(* Schneider Machine Expert - Basic project PLC_New_08_09, file version 2.7.0.0 *)
(* CompanyInformations: Name=Plast-O-Matick, Country=EEUU *)
(* ProjectInformations: Name=New project *)

HARDWARE
  Cpu 0: TM221CE16R
  ModuleExtensionObject 0: TM3AM6/G
  EthernetConfiguration: NetworkName=M221, IpAllocationMode=FixedAddress, IpAddress=192.168.1.235, SubnetMask=255.255.255.0
  SerialLineConfiguration: Baud=Baud19200, Parity=ParityNone, DataBits=DataBits8, StopBits=StopBits1, PhysicalMedium=PhysicalMediumRs485, TransmissionMode=TransmissionModeModbusRtu, SlaveId=1, Addressing=MasterAddressing
  MastTask: UsePeriodScanMode=false, PeriodScan=100
  FastTask: Period=255
  CpuBehavior: StartingMode=StartAsPreviousState, AutoSaveRamOnEeprom=true, WatchdogPeriod=250

SYMBOLS  (address, symbol, comment, settings)
  %MW432:X0 VLV03_04_POWER_ON
  %MW444:X0 VLV05_06_POWER_ON
  %MW117:X0 DATETIME_CHANGE
  %M0       VLV01_HMI_START
  %M1       VLV01_HMI_STP
  %M2       VLV01_CMD_OPN
  %M3       VLV01_TON_OPN_DN
  %M4       VLV01_COUNT_OPN_DN
  %M5       VLV01_RST_COUNT
  %M6       VLV01_ONS_STS_AUTOMATIC
  %M7       VLV01_CNF_OPN
  %M8       VLV01_CNF_CLS
  %M9       COPY_DATA
  %M10      VLV01_ONS_STP
  %M11      VLV01_SAVE_DATETIME
  %M12      VLV01_CMD_CLS
  %M13      VLV01_TON_CLS_DN
  %M14      VLV01_COUNT_CLS_DN
  %M15      VLV01_ALMD_CNF_OPN_DN
  %M16      VLV01_ALMD_CNF_CLS_DN
  %M17      VLV01_T_ALMD_CNF_OPN_DN
  %M19      VLV01_T_ALMD_CNF_CLS_DN
  %M20      PLC_HORARIOOFICINA
  %M21      HORARIOOFICINA_ACTIVE
  %M22      HMI_HORARIOOFICINA
  %M23      VLV01_STS_AUTOMATIC
  %M24      VLV01_HMI_STARTED
  %M25      VLV01_TON_SEG_RST
  %M26      VLV01_TON_SEG_DN
  %M27      VLV01_TON_MIN_DN
  %M28      VLV01_TON_HR_DN
  %M29      VLV2_ONS_STP
  %M30      VLV02_HMI_START
  %M31      VLV02_HMI_STP
  %M32      VLV02_CMD_OPN
  %M33      VLV02_TON_OPN_DN
  %M34      VLV02_COUNT_OPN_DN
  %M35      VLV02_RST_COUNT
  %M36      VLV02_ONS_STS_AUTOMATIC
  %M37      VLV02_CNF_OPN
  %M38      VLV02_CNF_CLS
  %M41      VLV02_SAVE_DATETIME
  %M42      VLV02_CMD_CLS
  %M43      VLV02_TON_CLS_DN
  %M44      VLV02_COUNT_CLS_DN
  %M45      VLV02_ALMD_CNF_OPN_DN
  %M46      VLV02_ALMD_CNF_CLS_DN
  %M47      VLV02_T_ALMD_CNF_OPN_DN
  %M49      VLV02_T_ALMD_CNF_CLS_DN
  %M50      VLV01_02_POWER_ON
  %M53      VLV02_STS_AUTOMATIC
  %M54      VLV02_HMI_STARTED
  %M55      VLV02_TON_SEG_RST
  %M56      VLV02_TON_SEG_DN
  %M57      VLV02_TON_MIN_DN
  %M58      VLV02_TON_HR_DN
  %M60      VLV03_HMI_START
  %M61      VLV03_HMI_STP
  %M62      VLV03_CMD_OPN
  %M63      VLV03_TON_OPN_DN
  %M64      VLV03_COUNT_OPN_DN
  %M65      VLV03_RST_COUNT
  %M66      VLV03_ONS_STR_AUTOMATIC
  %M67      VLV03_CNF_OPN
  %M68      VLV03_CNF_CLS
  %M70      VLV03_CLOSE_DATA1
  %M71      VLV03_SAVE_DATETIME
  %M72      VLV03_CMD_CLS
  %M73      VLV03_TON_CLS_DN
  %M74      VLV03_COUNT_CLS_DN
  %M75      VLV03_ALMD_CNF_OPN_DN
  %M76      VLV03_ALMD_CNF_CLS_DN
  %M77      VLV03_T_ALMD_CNF_OPN_DN
  %M78      VLV03_ONS_STP_AUTOMATIC
  %M79      VLV03_T_ALMD_CNF_CLS_DN
  %M83      VLV03_STS_AUTOMATIC
  %M84      VLV03_HMI_STARTED
  %M85      VLV03_TON_SEG_RST
  %M86      VLV03_TON_SEG_DN
  %M87      VLV03_TON_MIN_DN
  %M88      VLV03_TON_HR_DN
  %M90      VLV04_HMI_START
  %M91      VLV04_HMI_STP
  %M92      VLV04_CMD_OPN
  %M93      VLV04_TON_OPN_DN
  %M94      VLV04_COUNT_OPN_DN
  %M95      VLV04_RST_COUNT
  %M96      VLV04_ONS_STR_AUTOMATIC
  %M97      VLV04_CNF_OPN
  %M98      VLV04_CNF_CLS
  %M100     VLV04_CLOSE_DATA1
  %M101     VLV04_SAVE_DATETIME
  %M102     VLV04_CMD_CLS
  %M103     VLV04_TON_CLS_DN
  %M104     VLV04_COUNT_CLS_DN
  %M105     VLV04_ALMD_CNF_OPN_DN
  %M106     VLV04_ALMD_CNF_CLS_DN
  %M107     VLV04_T_ALMD_CNF_OPN_DN
  %M108     VLV04_ONS_STP_AUTOMATIC
  %M109     VLV04_T_ALMD_CNF_CLS_DN
  %M113     VLV04_STS_AUTOMATIC
  %M114     VLV04_HMI_STARTED
  %M115     VLV04_TON_SEG_RST
  %M116     VLV04_TON_SEG_DN
  %M117     VLV04_TON_MIN_DN
  %M118     VLV04_TON_HR_DN
  %M120     VLV05_HMI_START
  %M121     VLV05_HMI_STP
  %M122     VLV05_CMD_OPN
  %M123     VLV05_TON_OPN_DN
  %M124     VLV05_COUNT_OPN_DN
  %M125     VLV05_RST_COUNT
  %M126     VLV05_ONS_STS_AUTOMATIC
  %M127     VLV05_CNF_OPN
  %M128     VLV05_CNF_CLS
  %M131     VLV05_SAVE_DATETIME
  %M132     VLV05_CMD_CLS
  %M133     VLV05_TON_CLS_DN
  %M134     VLV05_COUNT_CLS_DN
  %M135     VLV05_ALMD_CNF_OPN_DN
  %M136     VLV05_ALMD_CNF_CLS_DN
  %M137     VLV05_T_ALMD_CNF_OPN_DN
  %M138     VLV05_ONS_STP_AUTOMATIC
  %M139     VLV05_T_ALMD_CNF_CLS_DN
  %M143     VLV05_STS_AUTOMATIC
  %M144     VLV05_HMI_STARTED
  %M145     VLV05_TON_SEG_RST
  %M146     VLV05_TON_SEG_DN
  %M147     VLV05_TON_MIN_DN
  %M148     VLV05_TON_HR_DN
  %M150     VLV06_HMI_START
  %M151     VLV06_HMI_STP
  %M152     VLV06_CMD_OPN
  %M153     VLV06_TON_OPN_DN
  %M154     VLV06_COUNT_OPN_DN
  %M155     VLV06_RST_COUNT
  %M156     VLV06_ONS_STS_AUTOMATIC
  %M157     VLV06_CNF_OPN
  %M158     VLV06_CNF_CLS
  %M161     VLV06_SAVE_DATETIME
  %M162     VLV06_CMD_CLS
  %M163     VLV06_TON_CLS_DN
  %M164     VLV06_COUNT_CLS_DN
  %M165     VLV06_ALMD_CNF_OPN_DN
  %M166     VLV06_ALMD_CNF_CLS_DN
  %M167     VLV06_T_ALMD_CNF_OPN_DN
  %M169     VLV06_T_ALMD_CNF_CLS_DN
  %M173     VLV06_STS_AUTOMATIC
  %M174     VLV06_HMI_STARTED
  %M175     VLV06_TON_SEG_RST
  %M176     VLV06_TON_SEG_DN
  %M177     VLV06_TON_MIN_DN
  %M178     VLV06_TON_HR_DN
  %M180     VLV07_HMI_START
  %M181     VLV07_HMI_STP
  %M182     VLV07_CMD_OPN
  %M183     VLV07_TON_OPN_DN
  %M184     VLV07_COUNT_OPN_DN
  %M185     VLV07_RST_COUNT
  %M186     VLV07_ONS_STS_AUTOMATIC
  %M187     VLV07_CNF_OPN
  %M188     VLV07_CNF_CLS
  %M191     VLV07_SAVE_DATETIME
  %M192     VLV07_CMD_CLS
  %M193     VLV07_TON_CLS_DN
  %M194     VLV07_COUNT_CLS_DN
  %M195     VLV07_ALMD_CNF_OPN_DN
  %M196     VLV07_ALMD_CNF_CLS_DN
  %M197     VLV07_T_ALMD_CNF_OPN_DN
  %M199     VLV07_T_ALMD_CNF_CLS_DN
  %M200     VLV07_SCHEDULE_ON
  %M203     VLV07_STS_AUTOMATIC
  %M204     VLV07_HMI_STARTED
  %M205     VLV07_TON_SEG_RST
  %M206     VLV07_TON_SEG_DN
  %M207     VLV07_TON_MIN_DN
  %M208     VLV07_TON_HR_DN
  %M220     VLV08_HMI_START
  %M221     VLV08_HMI_STP
  %M222     VLV08_HMI_STARTED
  %M223     VLV08_RST_COUNT
  %M224     VLV08_STS_AUTOMATIC
  %M225     VLV08_ONS_STR
  %M226     VLV08_ONS_STP_AUTOMATIC
  %M227     VLV08_ONS_STS_AUTOMATIC
  %M228     VLV08_ONS_01
  %M229     VLV08_CMD_OPN
  %M230     VLV08_CMD_CLS
  %M231     VLV08_CNF_OPN
  %M232     VLV08_CNF_CLS
  %M233     VLV08_TON_OPN_DN
  %M234     VLV08_TON_CLS_DN
  %M235     VLV08_TON_SEG_DN
  %M236     VLV08_TON_SEG_RST
  %M237     VLV08_TON_MIN_DN
  %M238     VLV08_TON_HR_DN
  %M239     VLV08_ALMD_CNF_OPN_DN
  %M240     VLV08_ALMD_CNF_CLS_DN
  %M241     VLV08_T_ALMD_CNF_OPN_DN
  %M242     VLV08_T_ALMD_CNF_CLS_DN
  %M243     VLV08_SAVE_DATETIME
  %M244     VLV08_T_CNF_OPN
  %M245     VLV08_T_CNF_CLS
  %M246     VLV08_MB_COMM_OK
  %M247     VLV08_MB_COMM_ERROR
  %M248     VLV08_MB_READ_ENABLE
  %M249     VLV08_MB_READ_TRIGGER
  %M250     VLV08_ONS_STR_AUTOMATIC
  %M251     VLV08_CLOSE_DATA1
  %M315     VLV09_HMI_START
  %M316     VLV09_HMI_STP
  %M317     VLV09_HMI_STARTED
  %M318     VLV09_RST_COUNT
  %M319     VLV09_STS_AUTOMATIC
  %M320     VLV09_ONS_STR
  %M321     VLV09_ONS_STP_AUTOMATIC
  %M322     VLV09_ONS_STS_AUTOMATIC
  %M323     VLV09_ONS_01
  %M324     VLV09_CMD_OPN
  %M325     VLV09_CMD_CLS
  %M326     VLV09_CNF_OPN
  %M327     VLV09_CNF_CLS
  %M328     VLV09_TON_OPN_DN
  %M329     VLV09_TON_CLS_DN
  %M330     VLV09_TON_SEG_DN
  %M331     VLV09_TON_SEG_RST
  %M332     VLV09_TON_MIN_DN
  %M333     VLV09_TON_HR_DN
  %M334     VLV09_ALMD_CNF_OPN_DN
  %M335     VLV09_ALMD_CNF_CLS_DN
  %M336     VLV09_T_ALMD_CNF_OPN_DN
  %M337     VLV09_T_ALMD_CNF_CLS_DN
  %M338     VLV09_SAVE_DATETIME
  %M339     VLV09_T_CNF_OPN
  %M340     VLV09_T_CNF_CLS
  %M341     VLV09_MB_COMM_OK
  %M342     VLV09_MB_COMM_ERROR
  %M343     VLV09_MB_READ_ENABLE
  %M344     VLV09_MB_READ_TRIGGER
  %S5       SB_TB100MS  "Time base of 100 ms generated by an internal clock"
  %S13      SB_FIRSTRUN  "Indicates the first controller cycle in RUN mode"
  %S50      SB_RTCUPDATE  "Set to 1, this bit allows to update the date and time"
  %SW51     SW_RTCHHMM  "RTC Function: contains in BCD HHMM: hour and minute"
  %SW52     SW_RTCMMDD  "RTC Function: contains in BCD MMDD: month and day"
  %SW53     SW_RTCCCYY  "RTC Function: contains in BCD CCYY: century and year"
  %MW0      VLV01_CNT_CLS_ACC
  %MW1      VLV01_CNT_OPN_ACC
  %MW2      VLV01_T_CNF_PRESET
  %MW3      VLV01_CNF_HR_PRESET
  %MW5      VLV01_RTC_HHMM
  %MW6      VLV01_RTC_MMDD
  %MW7      VLV01_RTC_YY
  %MW10     VLV02_CNT_CLS_ACC
  %MW11     VLV02_CNT_OPN_ACC
  %MW12     VLV02_T_CNF_PRESET  "timer1"
  %MW13     VLV02_CNF_HR_PRESET
  %MW15     VLV02_RTC_HHMM
  %MW16     VLV02_RTC_MMDD
  %MW17     VLV02_RTC_YY
  %MW18     VLV03_SP_ACTUAL
  %MW19     VLV03_CV_ACTUAL
  %MW20     VLV03_CNT_CLS_ACC
  %MW21     VLV03_CNT_OPN_ACC
  %MW22     VLV03_T_CNF_PRESET
  %MW23     VLV03_CNF_HR_PRESET
  %MW24     VLV03_SETPOINT_ALTO
  %MW25     VLV03_RTC_HHMM
  %MW26     VLV03_RTC_MMDD
  %MW27     VLV03_RTC_YY
  %MW28     VLV04_SP_ACTUAL
  %MW29     VLV04_CV_ACTUAL
  %MW30     VLV04_CNT_CLS_ACC
  %MW31     VLV04_CNT_OPN_ACC
  %MW32     VLV04_T_CNF_PRESET
  %MW33     VLV04_CNF_HR_PRESET
  %MW34     VLV04_SETPOINT_ALTO
  %MW35     VLV04_RTC_HHMM
  %MW36     VLV04_RTC_MMDD
  %MW37     VLV04_RTC_YY
  %MW40     VLV05_CNT_CLS_ACC
  %MW41     VLV05_CNT_OPN_ACC
  %MW42     VLV05_T_CNF_PRESET
  %MW43     VLV05_CNF_HR_PRESET
  %MW45     VLV05_RTC_HHMM
  %MW46     VLV05_RTC_MMDD
  %MW47     VLV05_RTC_YY
  %MW50     VLV06_CNT_CLS_ACC
  %MW51     VLV06_CNT_OPN_ACC
  %MW52     VLV06_T_CNF_PRESET
  %MW53     VLV06_CNF_HR_PRESET
  %MW55     VLV06_RTC_HHMM
  %MW56     VLV06_RTC_MMDD
  %MW57     VLV06_RTC_YY
  %MW60     VLV07_CNT_OPN_ACC
  %MW61     VLV07_CNT_CLS_ACC
  %MW63     VLV07_T_CICLO
  %MW64     VLV07_WORK_CICLE
  %MW68     VLV05_RTC_HHMM_OPEN
  %MW69     VLV05_RTC_MMDD_OPEN
  %MW70     VLV05_RTC_YY_OPEN
  %MW71     VLV05_RTC_HHMM_CLOSE
  %MW72     VLV05_RTC_MMDD_CLOSE
  %MW73     VLV05_RTC_YY_CLOSE
  %MW110    DAY
  %MW111    HOUR
  %MW112    MINUTES
  %MW113    MONTH
  %MW114    YEAR
  %MW115    SCRAP_MONTH
  %MW116    SCRAP_MINUTES
  %MW129    VLV07_SCHEDULE
  %MW130    VLV07_MONTH
  %MW131    VLV07_YR
  %MW132    VLV07_DY
  %MW133    VLV07_HR
  %MW134    VLV07_MIN
  %MW135    VLV07_OPEN_MONTH
  %MW136    VLV07_OPEN_YR
  %MW137    VLV07_OPEN_DY
  %MW138    VLV07_OPEN_HR
  %MW139    VLV07_OPEN_MIN
  %MW140    VLV07_CLOSE_MONTH
  %MW141    VLV07_CLOSE_YR
  %MW142    VLV07_CLOSE_DY
  %MW143    VLV07_CLOSE_HR
  %MW144    VLV07_CLOSE_MIN
  %MW145    VLV07_SCHED_HR
  %MW146    VLV07_SCHED_MIN
  %MW155    VLV01_CNF_OPN_W
  %MW156    VLV02_CNF_OPN_W
  %MW180    VLV08_SP_ACTUAL  "Setpoint actual VLV8"
  %MW181    VLV08_CV_ACTUAL  "Control value (salida analógica)"
  %MW182    VLV08_CNT_CLS_ACC  "Acumulador contador cierre"
  %MW183    VLV08_CNT_OPN_ACC  "Acumulador contador apertura"
  %MW184    VLV08_CNT_CLS_ACC2  "Acumulador cierre 2"
  %MW185    VLV08_CNT_OPN_ACC2  "Acumulador apertura 2"
  %MW186    VLV08_T_CNF_PRESET  "Tiempo configuración preset"
  %MW187    VLV08_CNF_HR_PRESET  "Horas configuración preset"
  %MW188    VLV08_RTC_HHMM  "RTC hora:minuto"
  %MW189    VLV08_RTC_MMDD  "RTC mes:día"
  %MW190    VLV08_RTC_YY  "RTC año"
  %MW191    VLV08_SETPOINT_ALTO  "Setpoint alto (límite superior)"
  %MW192      "Selector rango (0=0-20mA, 1=4-20mA)"
  %MW193    VLV08_WORK_CICLE  "Ciclo de trabajo (%)"
  %MW194    VLV08_T_CICLO  "Tiempo de ciclo (segundos)"
  %MW195    VLV08_MB_POSITION  "Posición Modbus (0-100%)"
  %MW196    VLV08_MB_COMM_OK_COUNT  "Contador comms exitosas"
  %MW197    VLV08_MB_ERROR_COUNT  "Contador errores comm"
  %MW210    VLV09_SP_ACTUAL
  %MW211    VLV09_CV_ACTUAL
  %MW212    VLV09_CNT_CLS_ACC
  %MW213    VLV09_CNT_OPN_ACC
  %MW214    VLV09_CNT_CLS_ACC2
  %MW215    VLV09_CNT_OPN_ACC2
  %MW216    VLV09_T_CNF_PRESET
  %MW217    VLV09_CNF_HR_PRESET
  %MW218    VLV09_RTC_HHMM
  %MW219    VLV09_RTC_MMDD
  %MW220    VLV09_RTC_YY
  %MW221    VLV09_SETPOINT_ALTO
  %MW222    VLV09_CLOSE_DATA1
  %MW223    VLV09_WORK_CICLE
  %MW224    VLV09_T_CICLO
  %MW225    VLV09_MB_POSITION
  %MW226    VLV09_MB_COMM_OK_COUNT
  %MW227    VLV09_MB_ERROR_COUNT
  %MD200    VLV01_CNT_OPN_ACC2
  %MD202    VLV01_CNT_CLS_ACC2
  %MD204    VLV02_CNT_OPN_ACC2
  %MD206    VLV02_CNT_CLS_ACC2
  %MD208    VLV03_CNT_OPN_ACC2
  %MD210    VLV03_CNT_CLS_ACC2
  %MD212    VLV04_CNT_OPN_ACC2
  %MD214    VLV04_CNT_CLS_ACC2
  %MD216    VLV05_CNT_OPN_ACC2
  %MD218    VLV05_CNT_CLS_ACC2
  %MD220    VLV06_CNT_OPN_ACC2
  %MD222    VLV06_CNT_CLS_ACC2
  %MD224    VLV07_CNT_OPN_ACC2
  %MD226    VLV07_CNT_CLS_ACC2
  %TM0      VLV01_TON_OPN  "timer1"  [Preset=600, Base=TenMilliSeconds]
  %TM1      VLV01_TON_SEG  [Preset=60, Base=OneSecond]
  %TM2      VLV01_TON_CLS  [Preset=600, Base=TenMilliSeconds]
  %TM3      VLV01_TON_ALMD_CNF_OPN  [Preset=400, Base=TenMilliSeconds]
  %TM4      VLV01_TON_ALMD_CNF_CLS  [Preset=500, Base=TenMilliSeconds]
  %TM5      VLV01_T_CNF_OPN  [Preset=400, Base=TenMilliSeconds]
  %TM6      VLV01_T_CNF_CLS  [Preset=400, Base=TenMilliSeconds]
  %TM7      VLV01_ONS_01  [Type=TP, Preset=50, Base=TenMilliSeconds]
  %TM8      NOVLV02_TON_SEG  [Preset=25, Base=TenMilliSeconds]
  %TM9      VLV03_ONS_STP  [Type=TP, Preset=100, Base=TenMilliSeconds]
  %TM10     VLV02_TON_OPN  [Preset=700, Base=TenMilliSeconds]
  %TM11     VLV02_TON_SEG  [Preset=60, Base=OneSecond, IsRetentive=true]
  %TM12     VLV02_TON_CLS  [Preset=500, Base=TenMilliSeconds]
  %TM13     VLV02_TON_ALMD_CNF_OPN  [Base=TenMilliSeconds]
  %TM14     VLV02_TON_ALMD_CNF_CLS  [Base=TenMilliSeconds]
  %TM15     VLV02_T_CNF_OPN  [Preset=250, Base=TenMilliSeconds]
  %TM16     VLV02_T_CNF_CLS  [Preset=250, Base=TenMilliSeconds]
  %TM17     VLV02_ONS  [Type=TP, Preset=50, Base=TenMilliSeconds]
  %TM18     VLV04_ONS_STP  [Type=TP, Preset=500, Base=TenMilliSeconds]
  %TM19     VLV05_ONS_STR  [Type=TP, Preset=500, Base=TenMilliSeconds]
  %TM20     VLV03_TON_OPN  [Preset=200, Base=TenMilliSeconds]
  %TM21     VLV03_TON_SEG  [Preset=60, Base=OneSecond]
  %TM22     VLV03_TON_CLS  [Preset=60, Base=TenMilliSeconds]
  %TM23     VLV03_TON_ALMD_CNF_OPN  [Preset=400, Base=TenMilliSeconds]
  %TM24     VLV03_TON_ALMD_CNF_CLS  [Preset=500, Base=TenMilliSeconds]
  %TM25     VLV03_T_CNF_OPN  [Preset=30, Base=TenMilliSeconds]
  %TM26     VLV03_T_CNF_CLS  [Preset=30, Base=TenMilliSeconds]
  %TM27     VLV03_ONS_01  [Type=TP, Preset=50, Base=TenMilliSeconds]
  %TM28       [Type=TP, Base=TenMilliSeconds]
  %TM29       [Preset=10, Base=OneSecond]
  %TM30     VLV04_TON_OPN  [Preset=300, Base=TenMilliSeconds]
  %TM31     VLV04_TON_SEG  [Preset=60, Base=OneSecond]
  %TM32     VLV04_TON_CLS  [Preset=300, Base=TenMilliSeconds]
  %TM33     VLV04_TON_ALMD_CNF_OPN  [Preset=300, Base=TenMilliSeconds]
  %TM34     VLV04_TON_ALMD_CNF_CLS  [Preset=300, Base=TenMilliSeconds]
  %TM35     VLV04_T_CNF_OPN  [Preset=10, Base=TenMilliSeconds]
  %TM36     VLV04_T_CNF_CLS  [Base=TenMilliSeconds]
  %TM37     VLV04_ONS  [Type=TP, Preset=50, Base=TenMilliSeconds]
  %TM38       [Type=TP, Preset=5, Base=OneSecond]
  %TM39       [Type=TP, Preset=6, Base=TenMilliSeconds]
  %TM40     VLV05_TON_OPN  [Preset=60, Base=TenMilliSeconds]
  %TM41     VLV05_TON_SEG  [Preset=60, Base=OneSecond]
  %TM42     VLV05_TON_CLS  [Preset=60, Base=TenMilliSeconds]
  %TM43     VLV05_TON_ALMD_CNF_OPN  [Preset=500, Base=TenMilliSeconds]
  %TM44     VLV05_TON_ALMD_CNF_CLS  [Preset=500, Base=TenMilliSeconds]
  %TM45     VLV05_T_CNF_OPN
  %TM46     VLV05_T_CNF_CLS
  %TM47     VLV05_ONS_01  [Type=TP, Preset=50, Base=TenMilliSeconds]
  %TM48       [Type=TP, Preset=50, Base=TenMilliSeconds]
  %TM49       [Type=TP, Preset=50, Base=TenMilliSeconds]
  %TM50     VLV06_TON_OPN  [Preset=200, Base=TenMilliSeconds]
  %TM51     VLV06_TON_SEG  [Preset=60, Base=OneSecond]
  %TM52     VLV06_TON_CLS  [Preset=300, Base=TenMilliSeconds]
  %TM53     VLV06_TON_ALMD_CNF_OPN  [Preset=300, Base=TenMilliSeconds]
  %TM54     VLV06_TON_ALMD_CNF_CLS  [Preset=300, Base=TenMilliSeconds]
  %TM55     VLV06_T_CNF_OPN
  %TM56     VLV06_T_CNF_CLS
  %TM57     VLV06_ONS  [Type=TP, Preset=50, Base=TenMilliSeconds]
  %TM58       [Preset=5, Base=OneSecond]
  %TM61       [Preset=60, Base=OneSecond]
  %TM76       [Preset=30, Base=TenMilliSeconds]
  %TM77       [Preset=30, Base=TenMilliSeconds]
  %TM78       [Preset=30, Base=TenMilliSeconds]
  %TM79       [Preset=30, Base=TenMilliSeconds]
  %TM80       [Type=TP, Preset=30, Base=TenMilliSeconds]
  %TM81       [Preset=30, Base=TenMilliSeconds]
  %TM87       [Type=TP, Preset=50, Base=TenMilliSeconds]
  %TM90       [Type=TP, Preset=50, Base=TenMilliSeconds]
  %TM91       [Type=TP, Preset=50, Base=TenMilliSeconds]
  %TM96       [Type=TP, Preset=50, Base=TenMilliSeconds]
  %TM100    VLV08_ONS_STP  [Type=TP, Preset=100, Base=TenMilliSeconds]
  %TM101    VLV08_ONS_02  [Type=TP, Preset=50, Base=TenMilliSeconds]
  %C0       VLV01_CNT_OPN
  %C1       VLV01_CNT_CLS
  %C2       VLV01_CNT_SEG  [Preset=1]
  %C3       VLV01_CNT_MIN  [Preset=60]
  %C4       VLV01_CNT_HR  [Preset=9]
  %C5       VLV02_CNT_SEG  [Preset=1]
  %C6       VLV02_CNT_MIN  [Preset=60]
  %C7       VLV02_CNT_HR  [Preset=8]
  %C8       VLV02_CNT_CLS
  %C9       VLV02_CNT_OPN
  %C10      VLV03_CNT_OPN  [Preset=60]
  %C11      VLV03_CNT_CLS
  %C12      VLV03_CNT_SEG  [Preset=1]
  %C13      VLV03_CNT_MIN  [Preset=60]
  %C14      VLV03_CNT_HR  [Preset=8]
  %C15      VLV04_CNT_SEG  [Preset=1]
  %C16      VLV04_CNT_MIN  [Preset=60]
  %C17      VLV04_CNT_HR  [Preset=60]
  %C18      VLV04_CNT_CLS  [Preset=60]
  %C19      VLV04_CNT_OPN
  %C20      VLV05_CNT_OPN
  %C21      VLV05_CNT_CLS
  %C22      VLV05_CNT_SEG  [Preset=1]
  %C23      VLV05_CNT_MIN  [Preset=60]
  %C24      VLV05_CNT_HR  [Preset=8]
  %C25      VLV06_CNT_SEG  [Preset=1]
  %C26      VLV06_CNT_MIN  [Preset=60]
  %C27      VLV06_CNT_HR  [Preset=9]
  %C28      VLV06_CNT_CLS
  %C29      VLV06_CNT_OPN
  %C30        [Preset=22]
  %C31        [Preset=20]
  %C32      VLV07_CNT_SEG  [Preset=1]
  %C33      VLV07_CNT_MIN  [Preset=60]
  %C34      VLV07_CNT_HR  [Preset=8]
  %C35        [Preset=5]
  %C36        [Preset=10]
  %C37        [Preset=10]
  %C40      VLV07_CNT_OPN
  %C41      VLV07_CNT_CLS
  %C50        [Preset=500]
  %C51        [Preset=500]
  %C52      VLV08_CNT_SEG  [Preset=500]
  %C53      VLV08_CNT_MIN
  %C54      VLV08_CNT_HR
  %C55      VLV08_CNT_OPN
  %C56      VLV08_CNT_CLS
  %C60      VLV09_CNT_OPN
  %C61      VLV09_CNT_CLS
  %C62      VLV09_CNT_SEG
  %C63      VLV09_CNT_MIN
  %C64      VLV09_CNT_HR
  %READ_VAR0   [Link(Value(FBComLinkParameterEnums=SerialLine1)), RemoteDeviceId(Value(int=1)), Timeout(Value(int=2)), ObjType(Value(FBComObjTypeParameterEnums=MW)), FirstObj(Value(int=1)), Quantity(Value(int=1)), IndexData(Value(int=59))]
  %READ_VAR1   [Link(Value(FBComLinkParameterEnums=SerialLine1)), RemoteDeviceId(Value(int=2)), Timeout(Value(int=2)), ObjType(Value(FBComObjTypeParameterEnums=MW)), FirstObj(Value(int=1)), Quantity(Value(int=1)), IndexData(Value(int=48))]
  %WRITE_VAR0   [Link(Value(FBComLinkParameterEnums=SerialLine1)), RemoteDeviceId(Value(int=1)), Timeout(Value(int=2)), ObjType(Value(FBComObjTypeParameterEnums=SINGLE_REG)), FirstObj(Value(int=2)), Quantity(Value(int=1)), IndexData(Value(int=90))]
  %WRITE_VAR1   [Link(Value(FBComLinkParameterEnums=SerialLine1)), RemoteDeviceId(Value(int=2)), Timeout(Value(int=2)), ObjType(Value(FBComObjTypeParameterEnums=SINGLE_REG)), FirstObj(Value(int=2)), Quantity(Value(int=1)), IndexData(Value(int=100))]
  %IW1.0    AI1  [Type=Type_0_10V, Scope=Scope_Customized, Minimum=0, Maximum=10000]
  %IW1.1    AI2  [Type=Type_0_20mA, Scope=Scope_Customized, Minimum=0, Maximum=20000]
  %QW1.0    AO1  [Type=Type_0_10V, Scope=Scope_Customized, Minimum=0, Maximum=10000]
  %QW1.1    AO2  [Type=Type_0_20mA, Scope=Scope_Customized, Minimum=0, Maximum=20000]

POU MAIN - TEST
  (* SectionNumber=1 *)

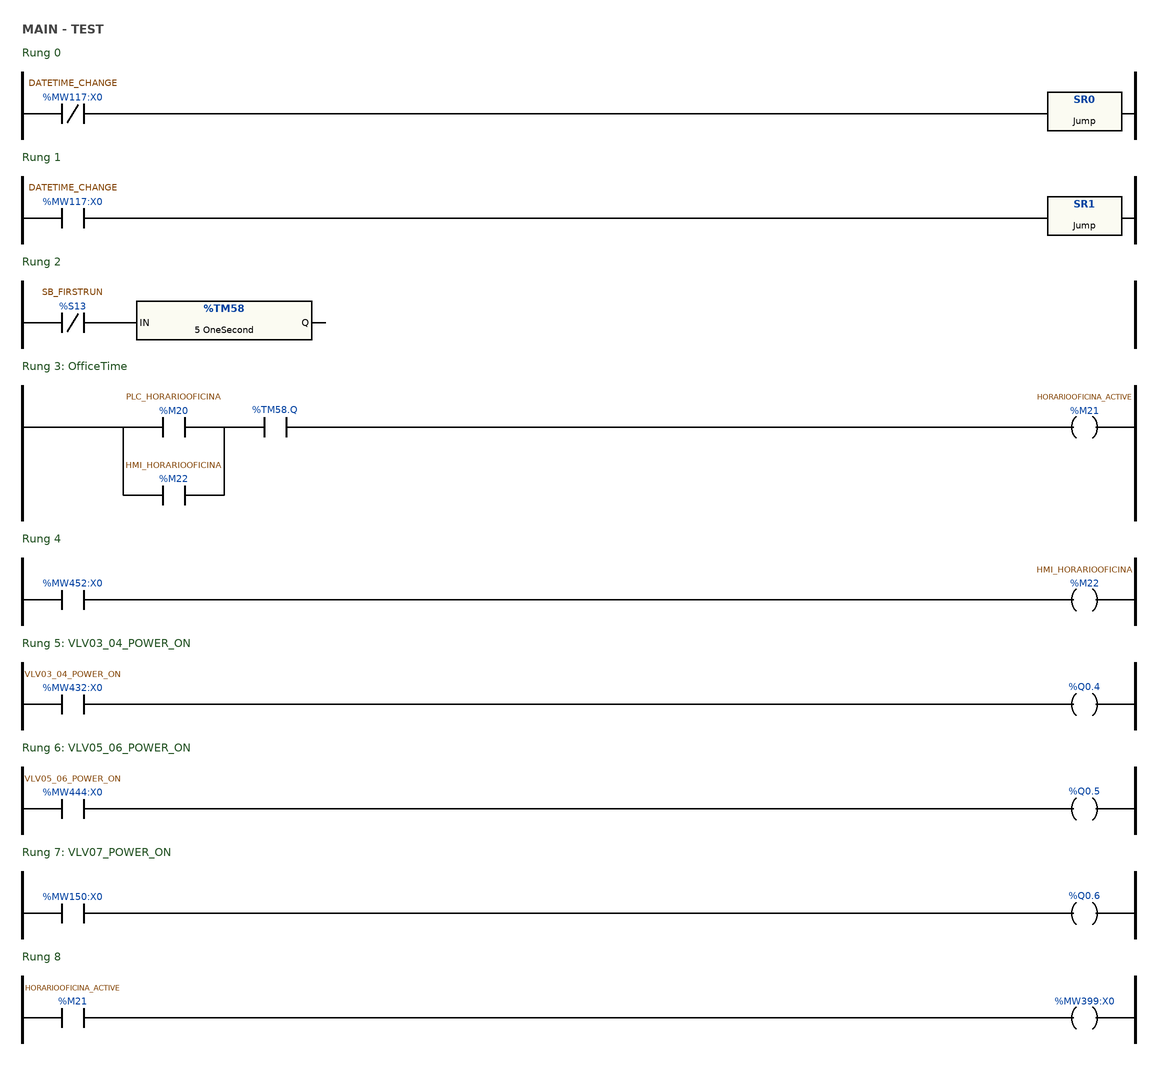

// Rung 0
  LDN %MW117:X0
  SR0
  // as ST:
  //   IF NOT %MW117:X0 THEN SR0(); END_IF;

// Rung 1
  LD %MW117:X0
  SR1
  // as ST:
  //   IF %MW117:X0 THEN SR1(); END_IF;

// Rung 2
  BLK %TM58
  LDN %S13                (* SB_FIRSTRUN *)
  IN
  END_BLK
  // as ST:
  //   %TM58(IN := NOT SB_FIRSTRUN);

// Rung 3: OfficeTime
  LD 1
  AND( %M20               (* PLC_HORARIOOFICINA *)
  OR %M22                 (* HMI_HORARIOOFICINA *)
  )
  AND %TM58.Q
  ST %M21                 (* HORARIOOFICINA_ACTIVE *)
  // as ST:
  //   HORARIOOFICINA_ACTIVE := (PLC_HORARIOOFICINA OR HMI_HORARIOOFICINA) AND %TM58.Q;

// Rung 4
  LD %MW452:X0
  ST %M22                 (* HMI_HORARIOOFICINA *)
  // as ST:
  //   HMI_HORARIOOFICINA := %MW452:X0;

// Rung 5: VLV03_04_POWER_ON
  LD %MW432:X0
  ST %Q0.4
  // as ST:
  //   %Q0.4 := %MW432:X0;

// Rung 6: VLV05_06_POWER_ON
  LD %MW444:X0
  ST %Q0.5
  // as ST:
  //   %Q0.5 := %MW444:X0;

// Rung 7: VLV07_POWER_ON
  LD %MW150:X0
  ST %Q0.6
  // as ST:
  //   %Q0.6 := %MW150:X0;

// Rung 8
  LD %M21                 (* HORARIOOFICINA_ACTIVE *)
  ST %MW399:X0
  // as ST:
  //   %MW399:X0 := HORARIOOFICINA_ACTIVE;

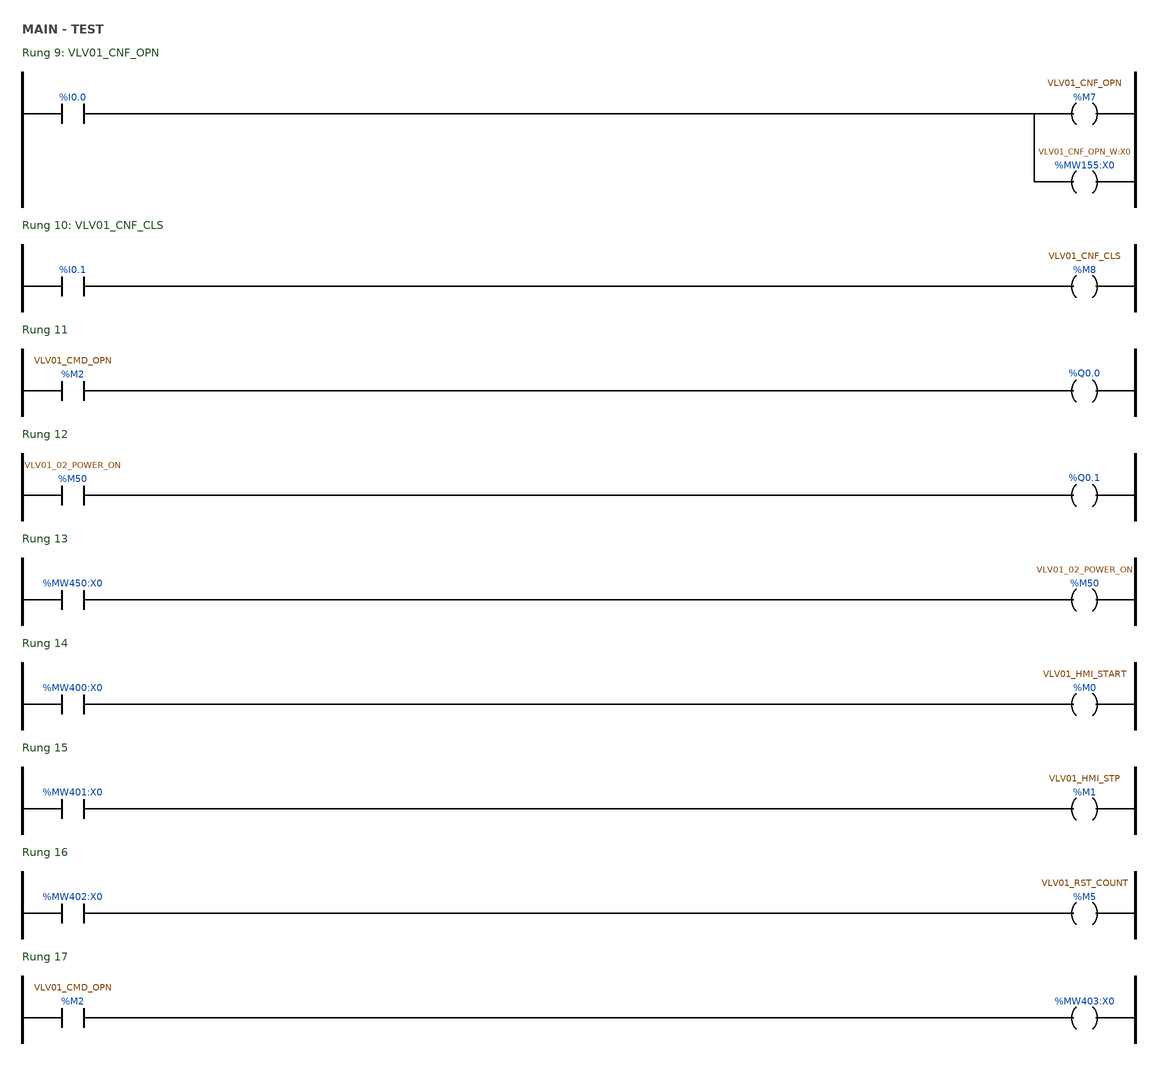

// Rung 9: VLV01_CNF_OPN
  LD %I0.0
  ST %M7                  (* VLV01_CNF_OPN *)
  ST %MW155:X0            (* VLV01_CNF_OPN_W *)
  // as ST:
  //   VLV01_CNF_OPN := %I0.0;
  //   VLV01_CNF_OPN_W:X0 := %I0.0;

// Rung 10: VLV01_CNF_CLS
  LD %I0.1
  ST %M8                  (* VLV01_CNF_CLS *)
  // as ST:
  //   VLV01_CNF_CLS := %I0.1;

// Rung 11
  LD %M2                  (* VLV01_CMD_OPN *)
  ST %Q0.0
  // as ST:
  //   %Q0.0 := VLV01_CMD_OPN;

// Rung 12
  LD %M50                 (* VLV01_02_POWER_ON *)
  ST %Q0.1
  // as ST:
  //   %Q0.1 := VLV01_02_POWER_ON;

// Rung 13
  LD %MW450:X0
  ST %M50                 (* VLV01_02_POWER_ON *)
  // as ST:
  //   VLV01_02_POWER_ON := %MW450:X0;

// Rung 14
  LD %MW400:X0
  ST %M0                  (* VLV01_HMI_START *)
  // as ST:
  //   VLV01_HMI_START := %MW400:X0;

// Rung 15
  LD %MW401:X0
  ST %M1                  (* VLV01_HMI_STP *)
  // as ST:
  //   VLV01_HMI_STP := %MW401:X0;

// Rung 16
  LD %MW402:X0
  ST %M5                  (* VLV01_RST_COUNT *)
  // as ST:
  //   VLV01_RST_COUNT := %MW402:X0;

// Rung 17
  LD %M2                  (* VLV01_CMD_OPN *)
  ST %MW403:X0
  // as ST:
  //   %MW403:X0 := VLV01_CMD_OPN;

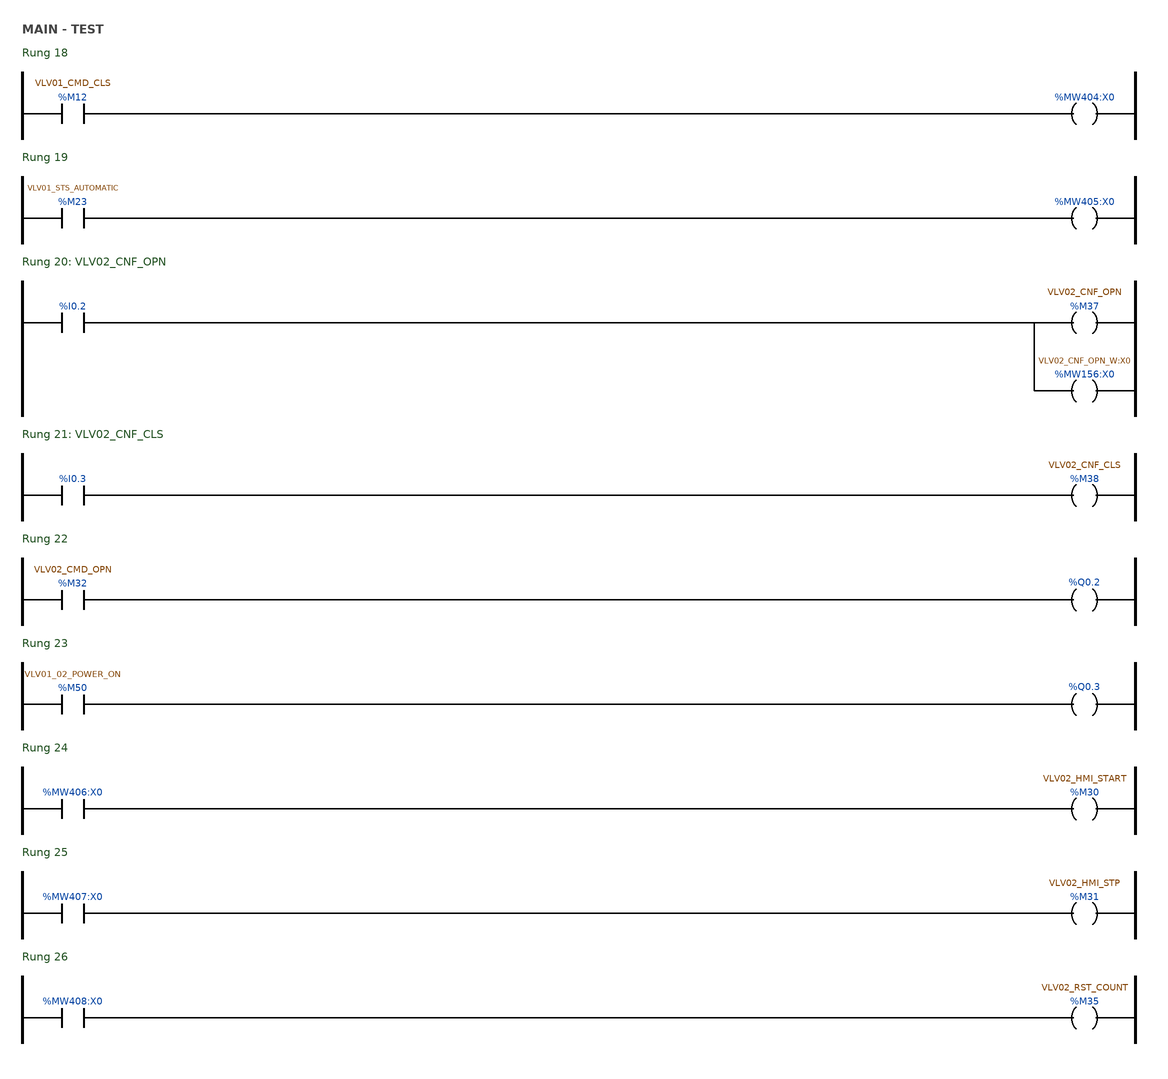

// Rung 18
  LD %M12                 (* VLV01_CMD_CLS *)
  ST %MW404:X0
  // as ST:
  //   %MW404:X0 := VLV01_CMD_CLS;

// Rung 19
  LD %M23                 (* VLV01_STS_AUTOMATIC *)
  ST %MW405:X0
  // as ST:
  //   %MW405:X0 := VLV01_STS_AUTOMATIC;

// Rung 20: VLV02_CNF_OPN
  LD %I0.2
  ST %M37                 (* VLV02_CNF_OPN *)
  ST %MW156:X0            (* VLV02_CNF_OPN_W *)
  // as ST:
  //   VLV02_CNF_OPN := %I0.2;
  //   VLV02_CNF_OPN_W:X0 := %I0.2;

// Rung 21: VLV02_CNF_CLS
  LD %I0.3
  ST %M38                 (* VLV02_CNF_CLS *)
  // as ST:
  //   VLV02_CNF_CLS := %I0.3;

// Rung 22
  LD %M32                 (* VLV02_CMD_OPN *)
  ST %Q0.2
  // as ST:
  //   %Q0.2 := VLV02_CMD_OPN;

// Rung 23
  LD %M50                 (* VLV01_02_POWER_ON *)
  ST %Q0.3
  // as ST:
  //   %Q0.3 := VLV01_02_POWER_ON;

// Rung 24
  LD %MW406:X0
  ST %M30                 (* VLV02_HMI_START *)
  // as ST:
  //   VLV02_HMI_START := %MW406:X0;

// Rung 25
  LD %MW407:X0
  ST %M31                 (* VLV02_HMI_STP *)
  // as ST:
  //   VLV02_HMI_STP := %MW407:X0;

// Rung 26
  LD %MW408:X0
  ST %M35                 (* VLV02_RST_COUNT *)
  // as ST:
  //   VLV02_RST_COUNT := %MW408:X0;

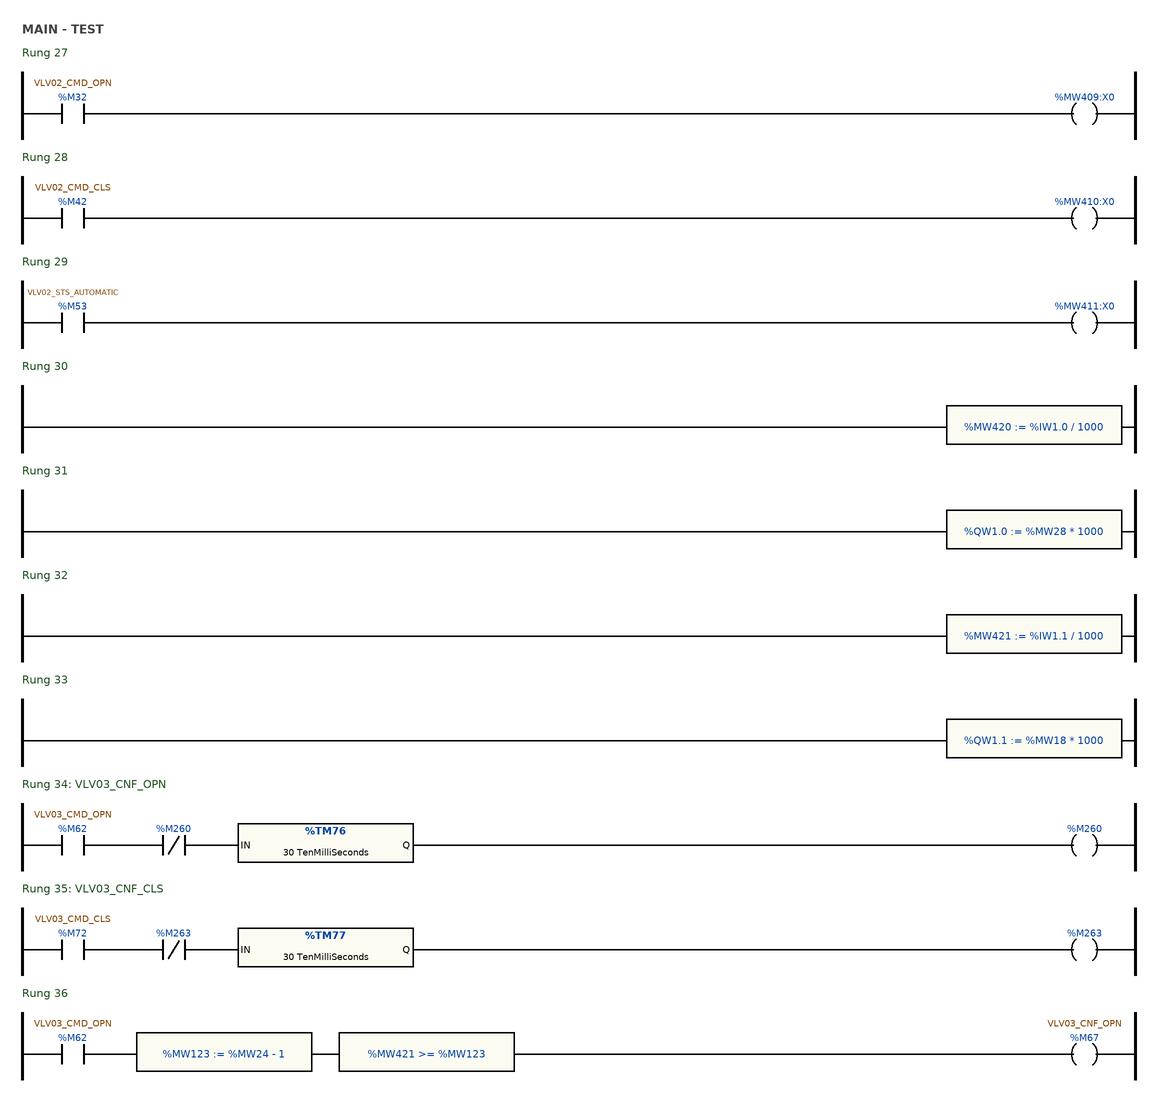

// Rung 27
  LD %M32                 (* VLV02_CMD_OPN *)
  ST %MW409:X0
  // as ST:
  //   %MW409:X0 := VLV02_CMD_OPN;

// Rung 28
  LD %M42                 (* VLV02_CMD_CLS *)
  ST %MW410:X0
  // as ST:
  //   %MW410:X0 := VLV02_CMD_CLS;

// Rung 29
  LD %M53                 (* VLV02_STS_AUTOMATIC *)
  ST %MW411:X0
  // as ST:
  //   %MW411:X0 := VLV02_STS_AUTOMATIC;

// Rung 30
  LD 1
  [ %MW420 := %IW1.0 / 1000 ](* AI1 *)
  // as ST:
  //   %MW420 := AI1 / 1000;

// Rung 31
  LD 1
  [ %QW1.0 := %MW28 * 1000 ](* AO1, VLV04_SP_ACTUAL *)
  // as ST:
  //   AO1 := VLV04_SP_ACTUAL * 1000;

// Rung 32
  LD 1
  [ %MW421 := %IW1.1 / 1000 ](* AI2 *)
  // as ST:
  //   %MW421 := AI2 / 1000;

// Rung 33
  LD 1
  [ %QW1.1 := %MW18 * 1000 ](* AO2, VLV03_SP_ACTUAL *)
  // as ST:
  //   AO2 := VLV03_SP_ACTUAL * 1000;

// Rung 34: VLV03_CNF_OPN
  BLK %TM76
  LD %M62                 (* VLV03_CMD_OPN *)
  ANDN %M260
  IN
  OUT_BLK
  LD Q
  ST %M260
  END_BLK
  // as ST:
  //   %TM76(IN := VLV03_CMD_OPN AND NOT %M260);
  //   %M260 := %TM76.Q;

// Rung 35: VLV03_CNF_CLS
  BLK %TM77
  LD %M72                 (* VLV03_CMD_CLS *)
  ANDN %M263
  IN
  OUT_BLK
  LD Q
  ST %M263
  END_BLK
  // as ST:
  //   %TM77(IN := VLV03_CMD_CLS AND NOT %M263);
  //   %M263 := %TM77.Q;

// Rung 36
  LD %M62                 (* VLV03_CMD_OPN *)
  OPER [ %MW123 := %MW24 - 1 ](* VLV03_SETPOINT_ALTO *)
  AND [ %MW421 >= %MW123 ]
  ST %M67                 (* VLV03_CNF_OPN *)
  // as ST:
  //   IF VLV03_CMD_OPN THEN %MW123 := VLV03_SETPOINT_ALTO - 1; END_IF;
  //   VLV03_CNF_OPN := VLV03_CMD_OPN AND %MW421 >= %MW123;

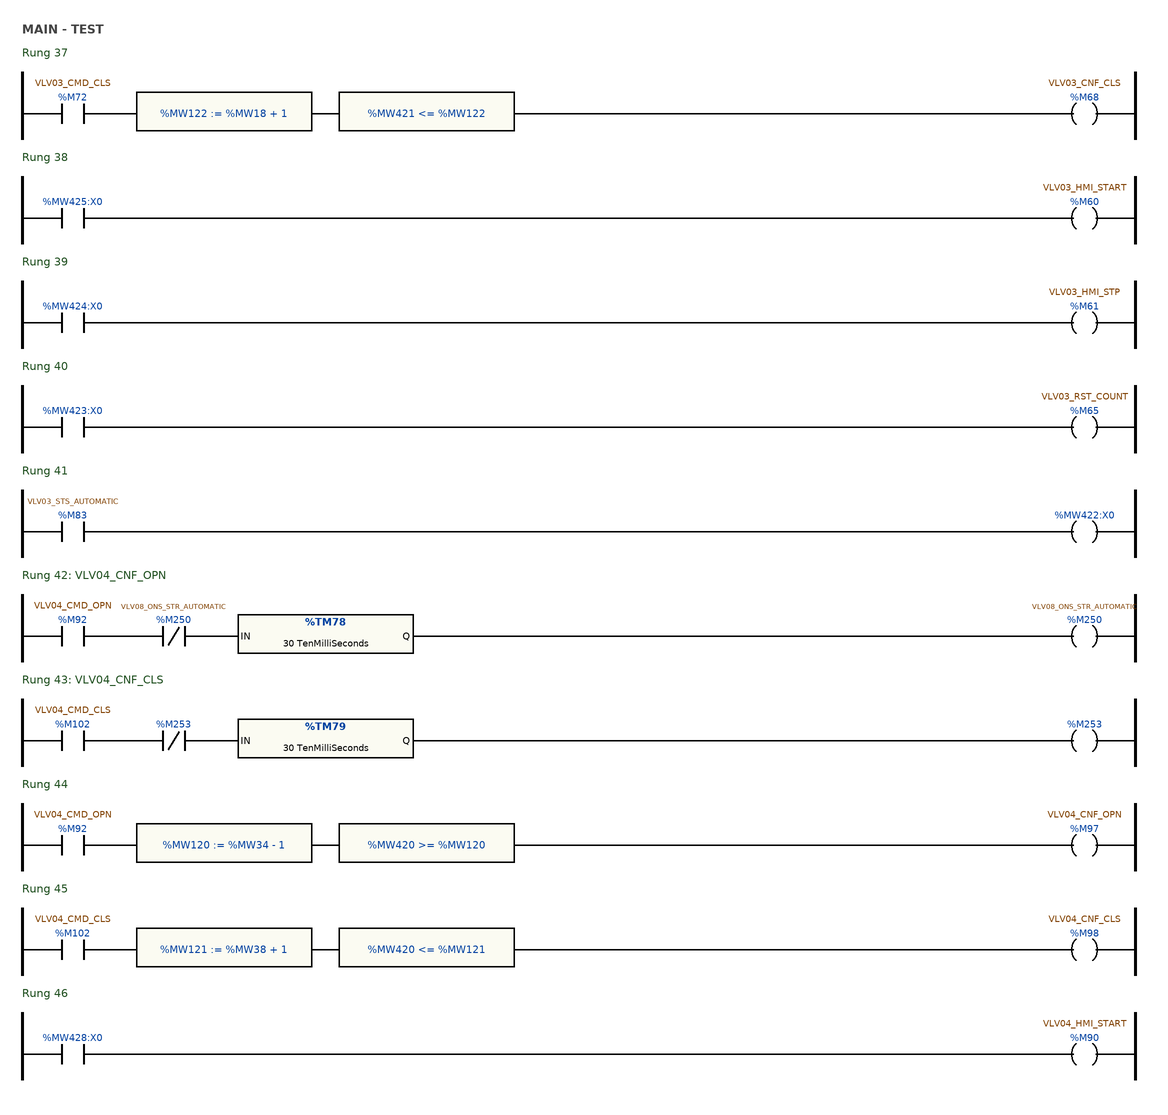

// Rung 37
  LD %M72                 (* VLV03_CMD_CLS *)
  OPER [ %MW122 := %MW18 + 1 ](* VLV03_SP_ACTUAL *)
  AND [ %MW421 <= %MW122 ]
  ST %M68                 (* VLV03_CNF_CLS *)
  // as ST:
  //   IF VLV03_CMD_CLS THEN %MW122 := VLV03_SP_ACTUAL + 1; END_IF;
  //   VLV03_CNF_CLS := VLV03_CMD_CLS AND %MW421 <= %MW122;

// Rung 38
  LD %MW425:X0
  ST %M60                 (* VLV03_HMI_START *)
  // as ST:
  //   VLV03_HMI_START := %MW425:X0;

// Rung 39
  LD %MW424:X0
  ST %M61                 (* VLV03_HMI_STP *)
  // as ST:
  //   VLV03_HMI_STP := %MW424:X0;

// Rung 40
  LD %MW423:X0
  ST %M65                 (* VLV03_RST_COUNT *)
  // as ST:
  //   VLV03_RST_COUNT := %MW423:X0;

// Rung 41
  LD %M83                 (* VLV03_STS_AUTOMATIC *)
  ST %MW422:X0
  // as ST:
  //   %MW422:X0 := VLV03_STS_AUTOMATIC;

// Rung 42: VLV04_CNF_OPN
  BLK %TM78
  LD %M92                 (* VLV04_CMD_OPN *)
  ANDN %M250              (* VLV08_ONS_STR_AUTOMATIC *)
  IN
  OUT_BLK
  LD Q
  ST %M250                (* VLV08_ONS_STR_AUTOMATIC *)
  END_BLK
  // as ST:
  //   %TM78(IN := VLV04_CMD_OPN AND NOT VLV08_ONS_STR_AUTOMATIC);
  //   VLV08_ONS_STR_AUTOMATIC := %TM78.Q;

// Rung 43: VLV04_CNF_CLS
  BLK %TM79
  LD %M102                (* VLV04_CMD_CLS *)
  ANDN %M253
  IN
  OUT_BLK
  LD Q
  ST %M253
  END_BLK
  // as ST:
  //   %TM79(IN := VLV04_CMD_CLS AND NOT %M253);
  //   %M253 := %TM79.Q;

// Rung 44
  LD %M92                 (* VLV04_CMD_OPN *)
  OPER [ %MW120 := %MW34 - 1 ](* VLV04_SETPOINT_ALTO *)
  AND [ %MW420 >= %MW120 ]
  ST %M97                 (* VLV04_CNF_OPN *)
  // as ST:
  //   IF VLV04_CMD_OPN THEN %MW120 := VLV04_SETPOINT_ALTO - 1; END_IF;
  //   VLV04_CNF_OPN := VLV04_CMD_OPN AND %MW420 >= %MW120;

// Rung 45
  LD %M102                (* VLV04_CMD_CLS *)
  OPER [ %MW121 := %MW38 + 1 ]
  AND [ %MW420 <= %MW121 ]
  ST %M98                 (* VLV04_CNF_CLS *)
  // as ST:
  //   IF VLV04_CMD_CLS THEN %MW121 := %MW38 + 1; END_IF;
  //   VLV04_CNF_CLS := VLV04_CMD_CLS AND %MW420 <= %MW121;

// Rung 46
  LD %MW428:X0
  ST %M90                 (* VLV04_HMI_START *)
  // as ST:
  //   VLV04_HMI_START := %MW428:X0;

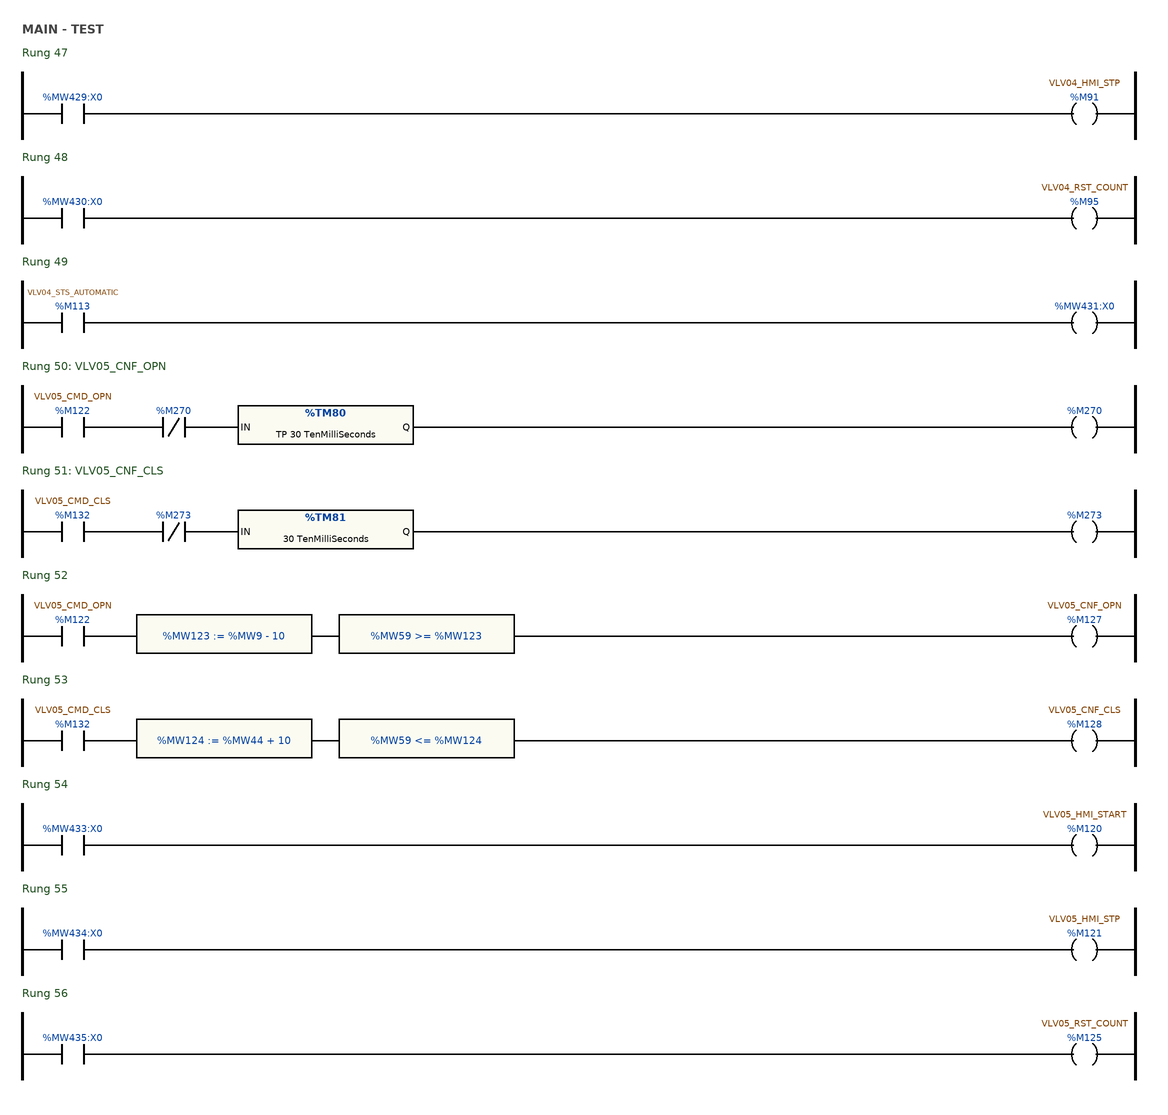

// Rung 47
  LD %MW429:X0
  ST %M91                 (* VLV04_HMI_STP *)
  // as ST:
  //   VLV04_HMI_STP := %MW429:X0;

// Rung 48
  LD %MW430:X0
  ST %M95                 (* VLV04_RST_COUNT *)
  // as ST:
  //   VLV04_RST_COUNT := %MW430:X0;

// Rung 49
  LD %M113                (* VLV04_STS_AUTOMATIC *)
  ST %MW431:X0
  // as ST:
  //   %MW431:X0 := VLV04_STS_AUTOMATIC;

// Rung 50: VLV05_CNF_OPN
  BLK %TM80
  LD %M122                (* VLV05_CMD_OPN *)
  ANDN %M270
  IN
  OUT_BLK
  LD Q
  ST %M270
  END_BLK
  // as ST:
  //   %TM80(IN := VLV05_CMD_OPN AND NOT %M270);
  //   %M270 := %TM80.Q;

// Rung 51: VLV05_CNF_CLS
  BLK %TM81
  LD %M132                (* VLV05_CMD_CLS *)
  ANDN %M273
  IN
  OUT_BLK
  LD Q
  ST %M273
  END_BLK
  // as ST:
  //   %TM81(IN := VLV05_CMD_CLS AND NOT %M273);
  //   %M273 := %TM81.Q;

// Rung 52
  LD %M122                (* VLV05_CMD_OPN *)
  OPER [ %MW123 := %MW9 - 10 ]
  AND [ %MW59 >= %MW123 ]
  ST %M127                (* VLV05_CNF_OPN *)
  // as ST:
  //   IF VLV05_CMD_OPN THEN %MW123 := %MW9 - 10; END_IF;
  //   VLV05_CNF_OPN := VLV05_CMD_OPN AND %MW59 >= %MW123;

// Rung 53
  LD %M132                (* VLV05_CMD_CLS *)
  OPER [ %MW124 := %MW44 + 10 ]
  AND [ %MW59 <= %MW124 ]
  ST %M128                (* VLV05_CNF_CLS *)
  // as ST:
  //   IF VLV05_CMD_CLS THEN %MW124 := %MW44 + 10; END_IF;
  //   VLV05_CNF_CLS := VLV05_CMD_CLS AND %MW59 <= %MW124;

// Rung 54
  LD %MW433:X0
  ST %M120                (* VLV05_HMI_START *)
  // as ST:
  //   VLV05_HMI_START := %MW433:X0;

// Rung 55
  LD %MW434:X0
  ST %M121                (* VLV05_HMI_STP *)
  // as ST:
  //   VLV05_HMI_STP := %MW434:X0;

// Rung 56
  LD %MW435:X0
  ST %M125                (* VLV05_RST_COUNT *)
  // as ST:
  //   VLV05_RST_COUNT := %MW435:X0;

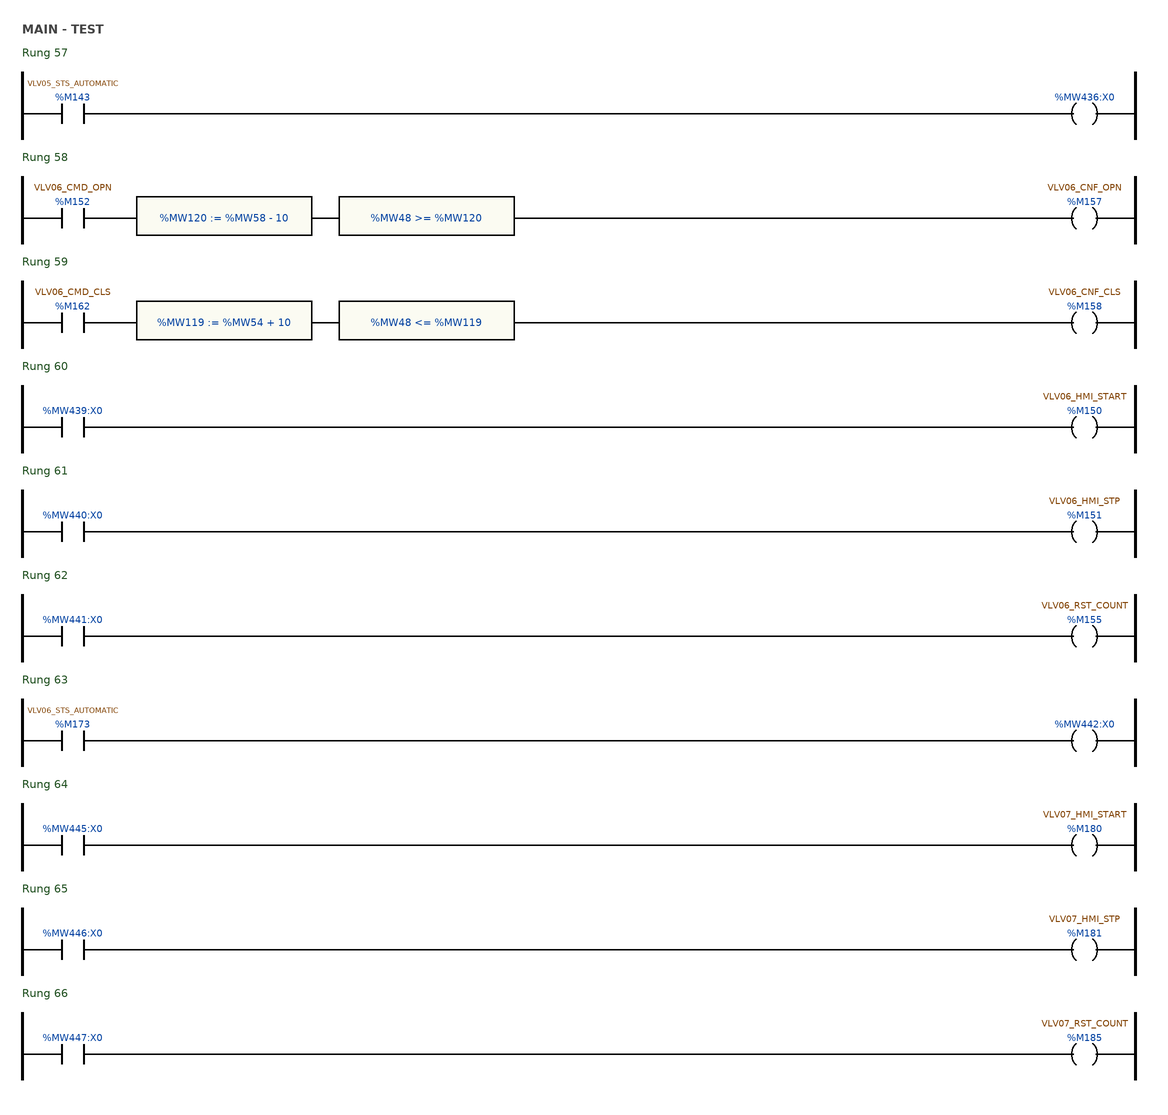

// Rung 57
  LD %M143                (* VLV05_STS_AUTOMATIC *)
  ST %MW436:X0
  // as ST:
  //   %MW436:X0 := VLV05_STS_AUTOMATIC;

// Rung 58
  LD %M152                (* VLV06_CMD_OPN *)
  OPER [ %MW120 := %MW58 - 10 ]
  AND [ %MW48 >= %MW120 ]
  ST %M157                (* VLV06_CNF_OPN *)
  // as ST:
  //   IF VLV06_CMD_OPN THEN %MW120 := %MW58 - 10; END_IF;
  //   VLV06_CNF_OPN := VLV06_CMD_OPN AND %MW48 >= %MW120;

// Rung 59
  LD %M162                (* VLV06_CMD_CLS *)
  OPER [ %MW119 := %MW54 + 10 ]
  AND [ %MW48 <= %MW119 ]
  ST %M158                (* VLV06_CNF_CLS *)
  // as ST:
  //   IF VLV06_CMD_CLS THEN %MW119 := %MW54 + 10; END_IF;
  //   VLV06_CNF_CLS := VLV06_CMD_CLS AND %MW48 <= %MW119;

// Rung 60
  LD %MW439:X0
  ST %M150                (* VLV06_HMI_START *)
  // as ST:
  //   VLV06_HMI_START := %MW439:X0;

// Rung 61
  LD %MW440:X0
  ST %M151                (* VLV06_HMI_STP *)
  // as ST:
  //   VLV06_HMI_STP := %MW440:X0;

// Rung 62
  LD %MW441:X0
  ST %M155                (* VLV06_RST_COUNT *)
  // as ST:
  //   VLV06_RST_COUNT := %MW441:X0;

// Rung 63
  LD %M173                (* VLV06_STS_AUTOMATIC *)
  ST %MW442:X0
  // as ST:
  //   %MW442:X0 := VLV06_STS_AUTOMATIC;

// Rung 64
  LD %MW445:X0
  ST %M180                (* VLV07_HMI_START *)
  // as ST:
  //   VLV07_HMI_START := %MW445:X0;

// Rung 65
  LD %MW446:X0
  ST %M181                (* VLV07_HMI_STP *)
  // as ST:
  //   VLV07_HMI_STP := %MW446:X0;

// Rung 66
  LD %MW447:X0
  ST %M185                (* VLV07_RST_COUNT *)
  // as ST:
  //   VLV07_RST_COUNT := %MW447:X0;

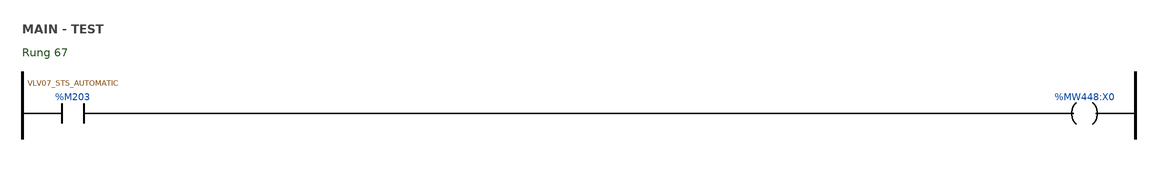

// Rung 67
  LD %M203                (* VLV07_STS_AUTOMATIC *)
  ST %MW448:X0
  // as ST:
  //   %MW448:X0 := VLV07_STS_AUTOMATIC;

POU VLV01_ON_OFF
  (* SectionNumber=2 *)

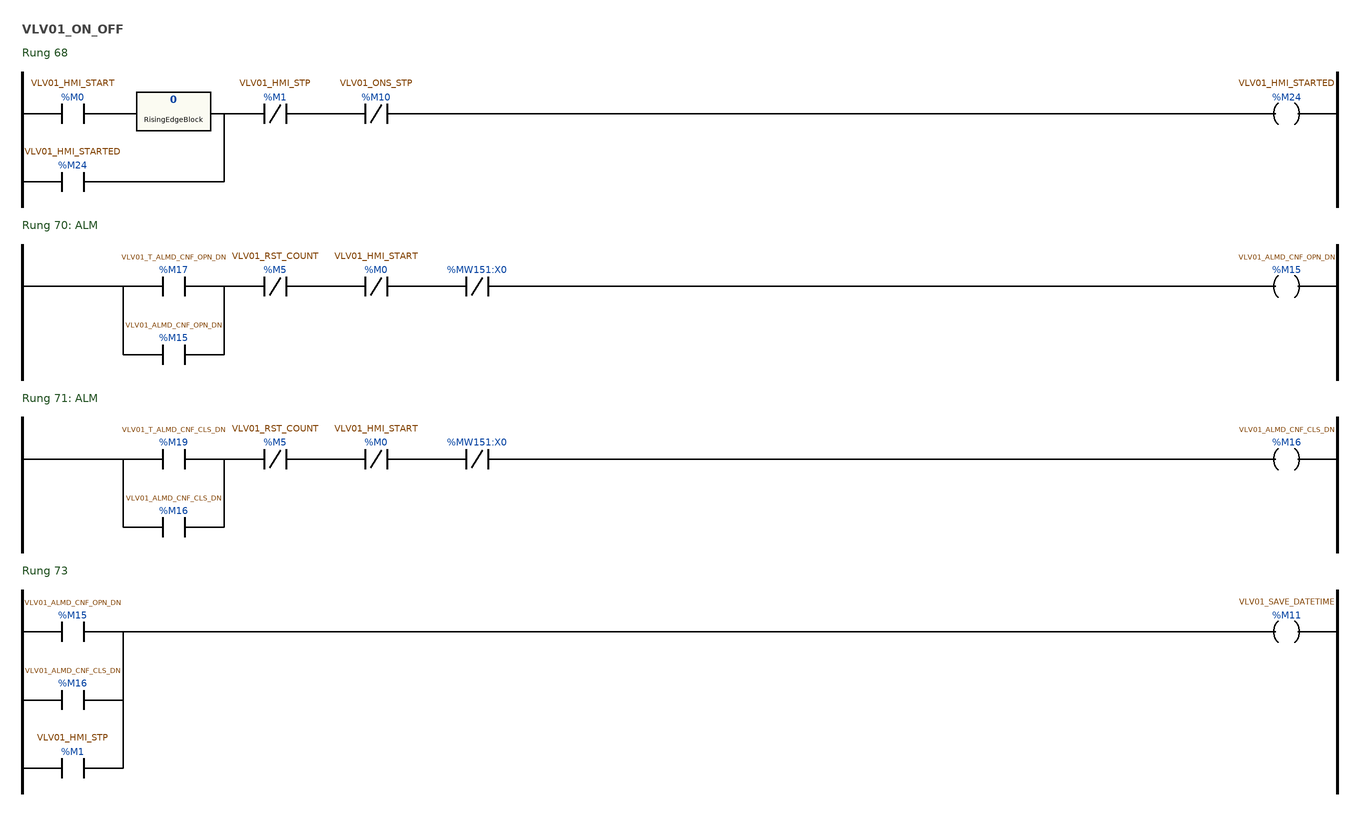

// Rung 68
  LD %M0                  (* VLV01_HMI_START *)
  RISING0
  OR %M24                 (* VLV01_HMI_STARTED *)
  ANDN %M1                (* VLV01_HMI_STP *)
  ANDN %M10               (* VLV01_ONS_STP *)
  ST %M24                 (* VLV01_HMI_STARTED *)
  // as ST:
  //   VLV01_HMI_STARTED := (RISING(VLV01_HMI_START) OR VLV01_HMI_STARTED) AND NOT VLV01_HMI_STP AND NOT VLV01_ONS_STP;

// Rung 69
  BLK %TM38
  LD %M1                  (* VLV01_HMI_STP *)
  OR(N %M23               (* VLV01_STS_AUTOMATIC *)
  RISING1
  )
  ANDN %M0                (* VLV01_HMI_START *)
  IN
  OUT_BLK
  LD Q
  ST %M10                 (* VLV01_ONS_STP *)
  END_BLK
  // as ST:
  //   %TM38(RISING1 := NOT VLV01_STS_AUTOMATIC, IN := (VLV01_HMI_STP OR NOT VLV01_STS_AUTOMATIC) AND NOT VLV01_HMI_START);
  //   VLV01_ONS_STP := %TM38.Q;
  (* the ladder stored for this rung does not match its IL; not drawn *)

// Rung 70: ALM
  LD 1
  AND( %M17               (* VLV01_T_ALMD_CNF_OPN_DN *)
  OR %M15                 (* VLV01_ALMD_CNF_OPN_DN *)
  )
  ANDN %M5                (* VLV01_RST_COUNT *)
  ANDN %M0                (* VLV01_HMI_START *)
  ANDN %MW151:X0
  ST %M15                 (* VLV01_ALMD_CNF_OPN_DN *)
  // as ST:
  //   VLV01_ALMD_CNF_OPN_DN := (VLV01_T_ALMD_CNF_OPN_DN OR VLV01_ALMD_CNF_OPN_DN) AND NOT VLV01_RST_COUNT AND NOT VLV01_HMI_START AND NOT %MW151:X0;

// Rung 71: ALM
  LD 1
  AND( %M19               (* VLV01_T_ALMD_CNF_CLS_DN *)
  OR %M16                 (* VLV01_ALMD_CNF_CLS_DN *)
  )
  ANDN %M5                (* VLV01_RST_COUNT *)
  ANDN %M0                (* VLV01_HMI_START *)
  ANDN %MW151:X0
  ST %M16                 (* VLV01_ALMD_CNF_CLS_DN *)
  // as ST:
  //   VLV01_ALMD_CNF_CLS_DN := (VLV01_T_ALMD_CNF_CLS_DN OR VLV01_ALMD_CNF_CLS_DN) AND NOT VLV01_RST_COUNT AND NOT VLV01_HMI_START AND NOT %MW151:X0;

// Rung 72: AUTM
  LD 1
  MULTIFB
  LD 1
  AND %M21                (* HORARIOOFICINA_ACTIVE *)
  AND %M24                (* VLV01_HMI_STARTED *)
  ANDN %M15               (* VLV01_ALMD_CNF_OPN_DN *)
  ANDN %M16               (* VLV01_ALMD_CNF_CLS_DN *)
  ANDN %M28               (* VLV01_TON_HR_DN *)
  ST %MW2509:X0
  LD %MW2509:X0
  ST %M23                 (* VLV01_STS_AUTOMATIC *)
  BLK %TM7                (* VLV01_ONS_01 *)
  LD %MW2509:X0
  IN
  OUT_BLK
  LD Q
  ST %M6                  (* VLV01_ONS_STS_AUTOMATIC *)
  END_BLK
  MULTIFB
  // as ST:
  //   %MW2509:X0 := HORARIOOFICINA_ACTIVE AND VLV01_HMI_STARTED AND NOT VLV01_ALMD_CNF_OPN_DN AND NOT VLV01_ALMD_CNF_CLS_DN AND NOT VLV01_TON_HR_DN;
  //   VLV01_STS_AUTOMATIC := %MW2509:X0;
  //   VLV01_ONS_01(IN := %MW2509:X0);
  //   VLV01_ONS_STS_AUTOMATIC := VLV01_ONS_01.Q;
  (* the ladder stored for this rung does not match its IL; not drawn *)

// Rung 73
  LD %M15                 (* VLV01_ALMD_CNF_OPN_DN *)
  OR %M16                 (* VLV01_ALMD_CNF_CLS_DN *)
  OR %M1                  (* VLV01_HMI_STP *)
  ST %M11                 (* VLV01_SAVE_DATETIME *)
  // as ST:
  //   VLV01_SAVE_DATETIME := VLV01_ALMD_CNF_OPN_DN OR VLV01_ALMD_CNF_CLS_DN OR VLV01_HMI_STP;

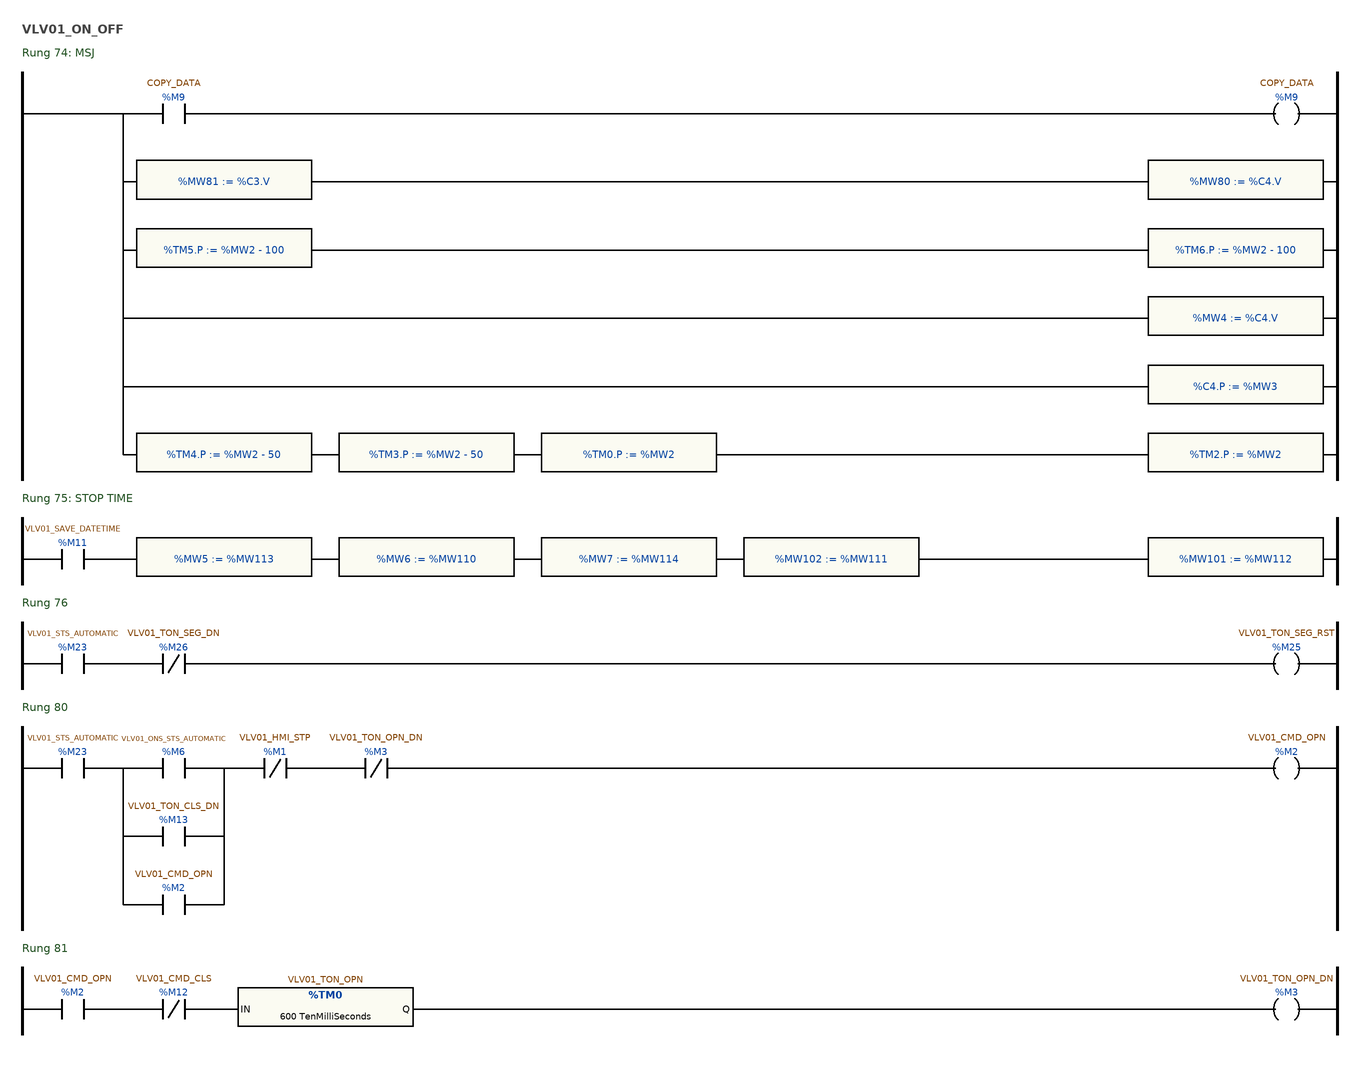

// Rung 74: MSJ
  LD 1
  MPS
  AND %M9                 (* COPY_DATA *)
  ST %M9                  (* COPY_DATA *)
  MRD
  OPER [ %MW81 := %C3.V ] (* VLV01_CNT_MIN *)
  [ %MW80 := %C4.V ]      (* VLV01_CNT_HR *)
  MRD
  OPER [ %TM5.P := %MW2 - 100 ](* VLV01_T_CNF_OPN, VLV01_T_CNF_PRESET *)
  [ %TM6.P := %MW2 - 100 ](* VLV01_T_CNF_CLS, VLV01_T_CNF_PRESET *)
  MRD
  [ %MW4 := %C4.V ]       (* VLV01_CNT_HR *)
  MRD
  [ %C4.P := %MW3 ]       (* VLV01_CNT_HR, VLV01_CNF_HR_PRESET *)
  MPP
  OPER [ %TM4.P := %MW2 - 50 ](* VLV01_TON_ALMD_CNF_CLS, VLV01_T_CNF_PRESET *)
  OPER [ %TM3.P := %MW2 - 50 ](* VLV01_TON_ALMD_CNF_OPN, VLV01_T_CNF_PRESET *)
  OPER [ %TM0.P := %MW2 ] (* VLV01_TON_OPN, VLV01_T_CNF_PRESET *)
  [ %TM2.P := %MW2 ]      (* VLV01_TON_CLS, VLV01_T_CNF_PRESET *)
  // as ST:
  //   COPY_DATA := COPY_DATA;
  //   %MW81 := VLV01_CNT_MIN.V;
  //   %MW80 := VLV01_CNT_HR.V;
  //   VLV01_T_CNF_OPN.P := VLV01_T_CNF_PRESET - 100;
  //   VLV01_T_CNF_CLS.P := VLV01_T_CNF_PRESET - 100;
  //   %MW4 := VLV01_CNT_HR.V;
  //   VLV01_CNT_HR.P := VLV01_CNF_HR_PRESET;
  //   VLV01_TON_ALMD_CNF_CLS.P := VLV01_T_CNF_PRESET - 50;
  //   VLV01_TON_ALMD_CNF_OPN.P := VLV01_T_CNF_PRESET - 50;
  //   VLV01_TON_OPN.P := VLV01_T_CNF_PRESET;
  //   VLV01_TON_CLS.P := VLV01_T_CNF_PRESET;

// Rung 75: STOP TIME
  LD %M11                 (* VLV01_SAVE_DATETIME *)
  OPER [ %MW5 := %MW113 ] (* VLV01_RTC_HHMM, MONTH *)
  OPER [ %MW6 := %MW110 ] (* VLV01_RTC_MMDD, DAY *)
  OPER [ %MW7 := %MW114 ] (* VLV01_RTC_YY, YEAR *)
  OPER [ %MW102 := %MW111 ](* HOUR *)
  [ %MW101 := %MW112 ]    (* MINUTES *)
  // as ST:
  //   IF VLV01_SAVE_DATETIME THEN VLV01_RTC_HHMM := MONTH; END_IF;
  //   IF VLV01_SAVE_DATETIME THEN VLV01_RTC_MMDD := DAY; END_IF;
  //   IF VLV01_SAVE_DATETIME THEN VLV01_RTC_YY := YEAR; END_IF;
  //   IF VLV01_SAVE_DATETIME THEN %MW102 := HOUR; END_IF;
  //   IF VLV01_SAVE_DATETIME THEN %MW101 := MINUTES; END_IF;

// Rung 76
  LD %M23                 (* VLV01_STS_AUTOMATIC *)
  ANDN %M26               (* VLV01_TON_SEG_DN *)
  ST %M25                 (* VLV01_TON_SEG_RST *)
  // as ST:
  //   VLV01_TON_SEG_RST := VLV01_STS_AUTOMATIC AND NOT VLV01_TON_SEG_DN;

// Rung 77
  BLK %C4                 (* VLV01_CNT_HR *)
  LD %M5                  (* VLV01_RST_COUNT *)
  OR( %M21                (* HORARIOOFICINA_ACTIVE *)
  RISING2
  )
  R
  LD %M27                 (* VLV01_TON_MIN_DN *)
  CU
  OUT_BLK
  LD D
  ST %M28                 (* VLV01_TON_HR_DN *)
  END_BLK
  // as ST:
  //   VLV01_CNT_HR(RISING2 := HORARIOOFICINA_ACTIVE, R := VLV01_RST_COUNT OR HORARIOOFICINA_ACTIVE, CU := VLV01_TON_MIN_DN);
  //   VLV01_TON_HR_DN := VLV01_CNT_HR.D;
  (* the ladder stored for this rung does not match its IL; not drawn *)

// Rung 78
  BLK %C3                 (* VLV01_CNT_MIN *)
  LD 1
  AND( %M5                (* VLV01_RST_COUNT *)
  OR %M27                 (* VLV01_TON_MIN_DN *)
  )
  OR( %M21                (* HORARIOOFICINA_ACTIVE *)
  RISING3
  )
  R
  LD %M26                 (* VLV01_TON_SEG_DN *)
  CU
  OUT_BLK
  LD D
  ST %M27                 (* VLV01_TON_MIN_DN *)
  END_BLK
  // as ST:
  //   VLV01_CNT_MIN(RISING3 := HORARIOOFICINA_ACTIVE, R := VLV01_RST_COUNT OR VLV01_TON_MIN_DN OR HORARIOOFICINA_ACTIVE, CU := VLV01_TON_SEG_DN);
  //   VLV01_TON_MIN_DN := VLV01_CNT_MIN.D;
  (* the ladder stored for this rung does not match its IL; not drawn *)

// Rung 79
  LD 1
  MULTIFB
  LD 1
  ST %MW2509:X1
  BLK %TM1                (* VLV01_TON_SEG *)
  LD %MW2509:X1
  AND %M23                (* VLV01_STS_AUTOMATIC *)
  AND %M25                (* VLV01_TON_SEG_RST *)
  IN
  OUT_BLK
  LD Q
  ST %MW2509:X0
  END_BLK
  BLK %C2                 (* VLV01_CNT_SEG *)
  LD %MW2509:X1
  AND( %M5                (* VLV01_RST_COUNT *)
  OR %M26                 (* VLV01_TON_SEG_DN *)
  )
  R
  LD %MW2509:X0
  CU
  OUT_BLK
  LD D
  ST %M26                 (* VLV01_TON_SEG_DN *)
  END_BLK
  MULTIFB
  // as ST:
  //   %MW2509:X1 := TRUE;
  //   VLV01_TON_SEG(IN := %MW2509:X1 AND VLV01_STS_AUTOMATIC AND VLV01_TON_SEG_RST);
  //   %MW2509:X0 := VLV01_TON_SEG.Q;
  //   VLV01_CNT_SEG(R := %MW2509:X1 AND (VLV01_RST_COUNT OR VLV01_TON_SEG_DN), CU := %MW2509:X0);
  //   VLV01_TON_SEG_DN := VLV01_CNT_SEG.D;
  (* the ladder stored for this rung does not match its IL; not drawn *)

// Rung 80
  LD %M23                 (* VLV01_STS_AUTOMATIC *)
  AND( %M6                (* VLV01_ONS_STS_AUTOMATIC *)
  OR %M13                 (* VLV01_TON_CLS_DN *)
  OR %M2                  (* VLV01_CMD_OPN *)
  )
  ANDN %M1                (* VLV01_HMI_STP *)
  ANDN %M3                (* VLV01_TON_OPN_DN *)
  ST %M2                  (* VLV01_CMD_OPN *)
  // as ST:
  //   VLV01_CMD_OPN := VLV01_STS_AUTOMATIC AND (VLV01_ONS_STS_AUTOMATIC OR VLV01_TON_CLS_DN OR VLV01_CMD_OPN) AND NOT VLV01_HMI_STP AND NOT VLV01_TON_OPN_DN;

// Rung 81
  BLK %TM0                (* VLV01_TON_OPN *)
  LD %M2                  (* VLV01_CMD_OPN *)
  ANDN %M12               (* VLV01_CMD_CLS *)
  IN
  OUT_BLK
  LD Q
  ST %M3                  (* VLV01_TON_OPN_DN *)
  END_BLK
  // as ST:
  //   VLV01_TON_OPN(IN := VLV01_CMD_OPN AND NOT VLV01_CMD_CLS);
  //   VLV01_TON_OPN_DN := VLV01_TON_OPN.Q;

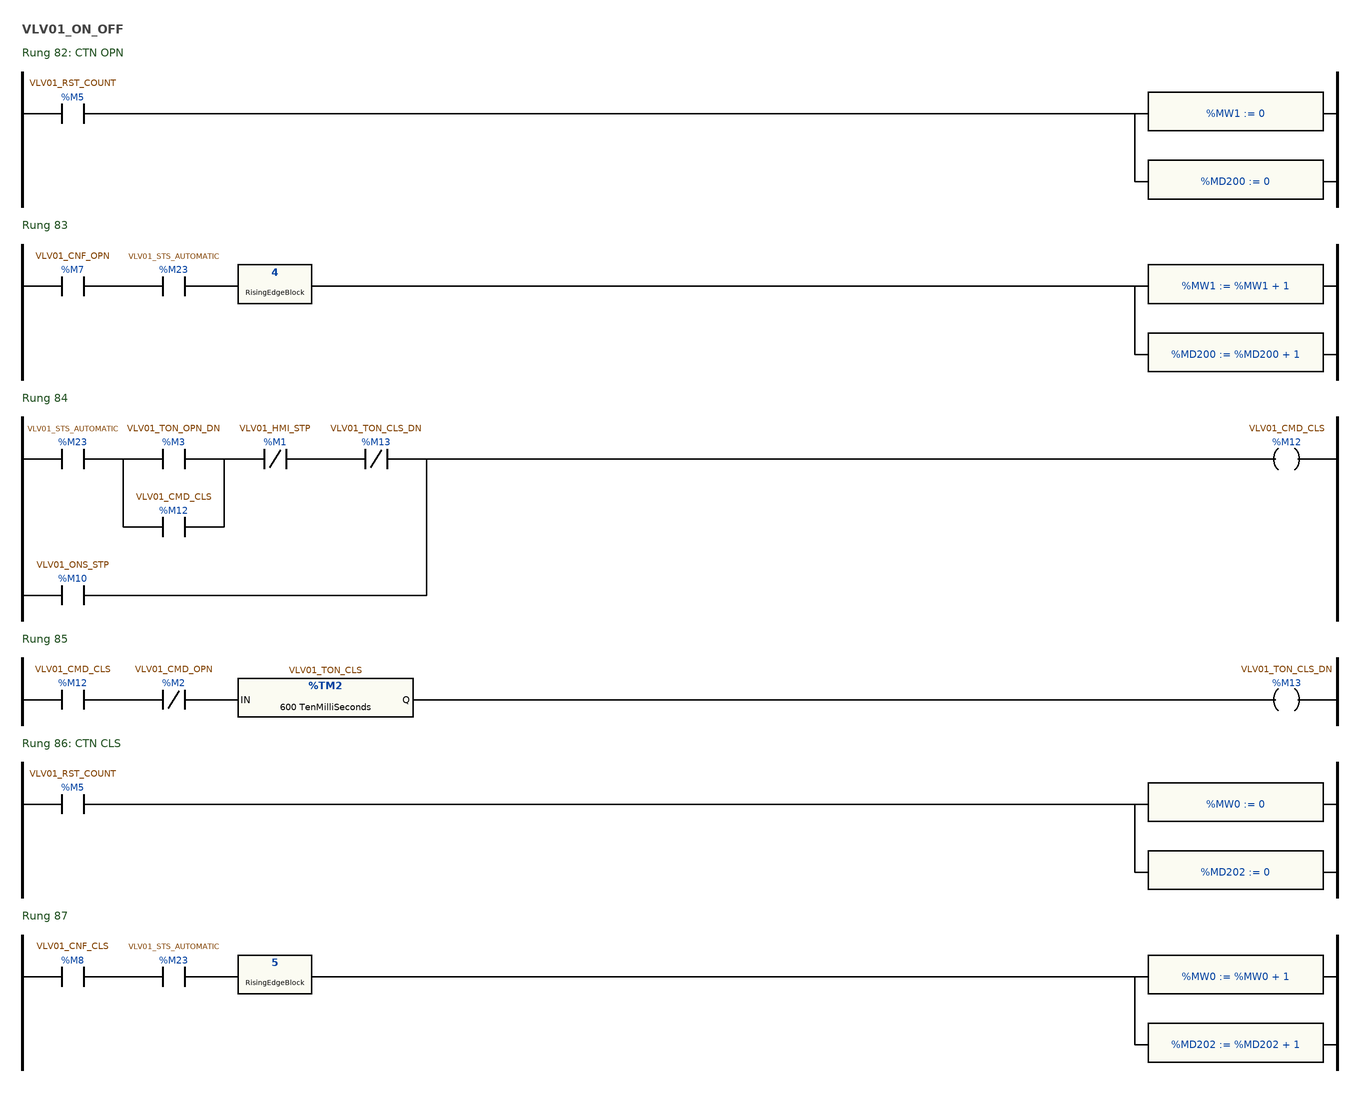

// Rung 82: CTN OPN
  LD %M5                  (* VLV01_RST_COUNT *)
  [ %MW1 := 0 ]           (* VLV01_CNT_OPN_ACC *)
  [ %MD200 := 0 ]         (* VLV01_CNT_OPN_ACC2 *)
  // as ST:
  //   IF VLV01_RST_COUNT THEN VLV01_CNT_OPN_ACC := 0; END_IF;
  //   IF VLV01_RST_COUNT THEN VLV01_CNT_OPN_ACC2 := 0; END_IF;

// Rung 83
  LD %M7                  (* VLV01_CNF_OPN *)
  AND %M23                (* VLV01_STS_AUTOMATIC *)
  RISING4
  [ %MW1 := %MW1 + 1 ]    (* VLV01_CNT_OPN_ACC, VLV01_CNT_OPN_ACC *)
  [ %MD200 := %MD200 + 1 ](* VLV01_CNT_OPN_ACC2, VLV01_CNT_OPN_ACC2 *)
  // as ST:
  //   IF RISING(VLV01_CNF_OPN AND VLV01_STS_AUTOMATIC) THEN VLV01_CNT_OPN_ACC := VLV01_CNT_OPN_ACC + 1; END_IF;
  //   IF RISING(VLV01_CNF_OPN AND VLV01_STS_AUTOMATIC) THEN VLV01_CNT_OPN_ACC2 := VLV01_CNT_OPN_ACC2 + 1; END_IF;

// Rung 84
  LD %M23                 (* VLV01_STS_AUTOMATIC *)
  AND( %M3                (* VLV01_TON_OPN_DN *)
  OR %M12                 (* VLV01_CMD_CLS *)
  )
  ANDN %M1                (* VLV01_HMI_STP *)
  ANDN %M13               (* VLV01_TON_CLS_DN *)
  OR %M10                 (* VLV01_ONS_STP *)
  ST %M12                 (* VLV01_CMD_CLS *)
  // as ST:
  //   VLV01_CMD_CLS := VLV01_STS_AUTOMATIC AND (VLV01_TON_OPN_DN OR VLV01_CMD_CLS) AND NOT VLV01_HMI_STP AND NOT VLV01_TON_CLS_DN OR VLV01_ONS_STP;

// Rung 85
  BLK %TM2                (* VLV01_TON_CLS *)
  LD %M12                 (* VLV01_CMD_CLS *)
  ANDN %M2                (* VLV01_CMD_OPN *)
  IN
  OUT_BLK
  LD Q
  ST %M13                 (* VLV01_TON_CLS_DN *)
  END_BLK
  // as ST:
  //   VLV01_TON_CLS(IN := VLV01_CMD_CLS AND NOT VLV01_CMD_OPN);
  //   VLV01_TON_CLS_DN := VLV01_TON_CLS.Q;

// Rung 86: CTN CLS
  LD %M5                  (* VLV01_RST_COUNT *)
  [ %MW0 := 0 ]           (* VLV01_CNT_CLS_ACC *)
  [ %MD202 := 0 ]         (* VLV01_CNT_CLS_ACC2 *)
  // as ST:
  //   IF VLV01_RST_COUNT THEN VLV01_CNT_CLS_ACC := 0; END_IF;
  //   IF VLV01_RST_COUNT THEN VLV01_CNT_CLS_ACC2 := 0; END_IF;

// Rung 87
  LD %M8                  (* VLV01_CNF_CLS *)
  AND %M23                (* VLV01_STS_AUTOMATIC *)
  RISING5
  [ %MW0 := %MW0 + 1 ]    (* VLV01_CNT_CLS_ACC, VLV01_CNT_CLS_ACC *)
  [ %MD202 := %MD202 + 1 ](* VLV01_CNT_CLS_ACC2, VLV01_CNT_CLS_ACC2 *)
  // as ST:
  //   IF RISING(VLV01_CNF_CLS AND VLV01_STS_AUTOMATIC) THEN VLV01_CNT_CLS_ACC := VLV01_CNT_CLS_ACC + 1; END_IF;
  //   IF RISING(VLV01_CNF_CLS AND VLV01_STS_AUTOMATIC) THEN VLV01_CNT_CLS_ACC2 := VLV01_CNT_CLS_ACC2 + 1; END_IF;

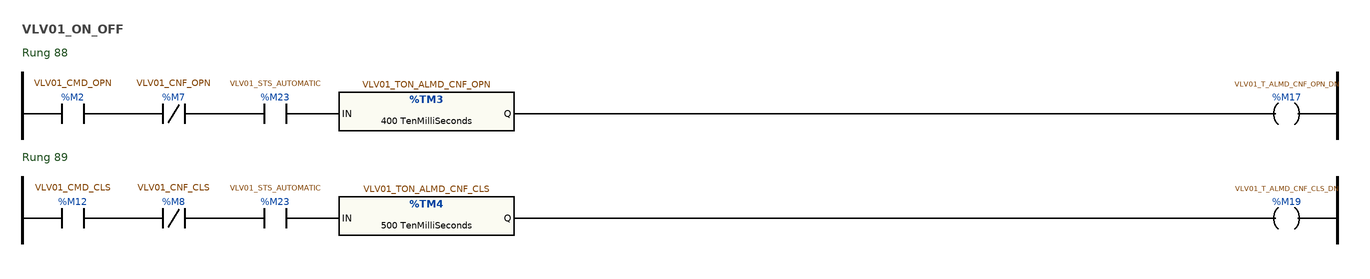

// Rung 88
  BLK %TM3                (* VLV01_TON_ALMD_CNF_OPN *)
  LD %M2                  (* VLV01_CMD_OPN *)
  ANDN %M7                (* VLV01_CNF_OPN *)
  AND %M23                (* VLV01_STS_AUTOMATIC *)
  IN
  OUT_BLK
  LD Q
  ST %M17                 (* VLV01_T_ALMD_CNF_OPN_DN *)
  END_BLK
  // as ST:
  //   VLV01_TON_ALMD_CNF_OPN(IN := VLV01_CMD_OPN AND NOT VLV01_CNF_OPN AND VLV01_STS_AUTOMATIC);
  //   VLV01_T_ALMD_CNF_OPN_DN := VLV01_TON_ALMD_CNF_OPN.Q;

// Rung 89
  BLK %TM4                (* VLV01_TON_ALMD_CNF_CLS *)
  LD %M12                 (* VLV01_CMD_CLS *)
  ANDN %M8                (* VLV01_CNF_CLS *)
  AND %M23                (* VLV01_STS_AUTOMATIC *)
  IN
  OUT_BLK
  LD Q
  ST %M19                 (* VLV01_T_ALMD_CNF_CLS_DN *)
  END_BLK
  // as ST:
  //   VLV01_TON_ALMD_CNF_CLS(IN := VLV01_CMD_CLS AND NOT VLV01_CNF_CLS AND VLV01_STS_AUTOMATIC);
  //   VLV01_T_ALMD_CNF_CLS_DN := VLV01_TON_ALMD_CNF_CLS.Q;

POU VLV02_ON_OFF
  (* SectionNumber=3 *)

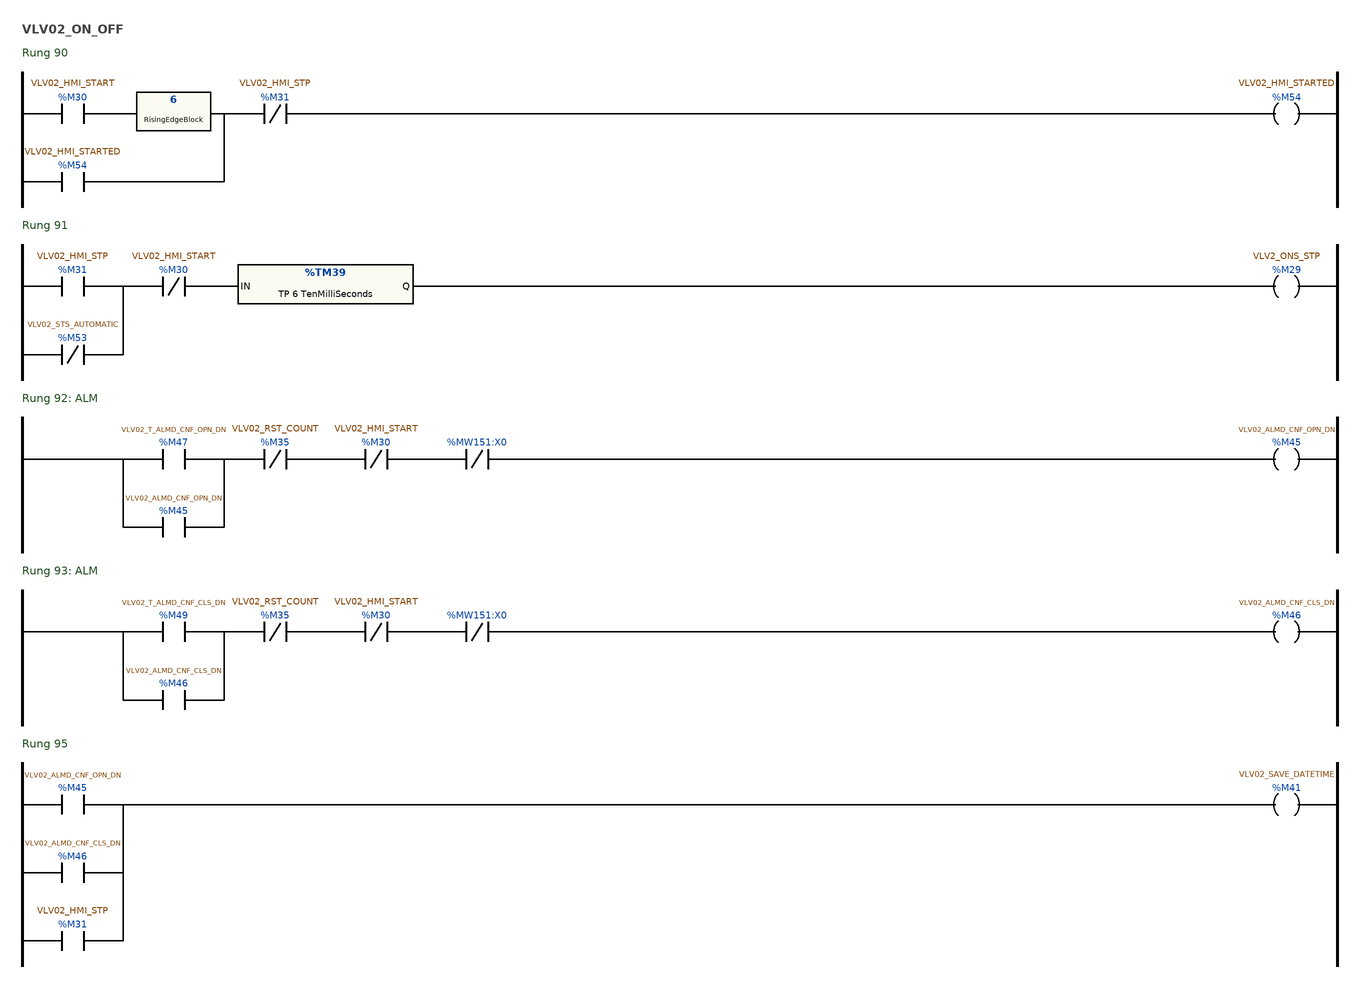

// Rung 90
  LD %M30                 (* VLV02_HMI_START *)
  RISING6
  OR %M54                 (* VLV02_HMI_STARTED *)
  ANDN %M31               (* VLV02_HMI_STP *)
  ST %M54                 (* VLV02_HMI_STARTED *)
  // as ST:
  //   VLV02_HMI_STARTED := (RISING(VLV02_HMI_START) OR VLV02_HMI_STARTED) AND NOT VLV02_HMI_STP;

// Rung 91
  BLK %TM39
  LD %M31                 (* VLV02_HMI_STP *)
  ORN %M53                (* VLV02_STS_AUTOMATIC *)
  ANDN %M30               (* VLV02_HMI_START *)
  IN
  OUT_BLK
  LD Q
  ST %M29                 (* VLV2_ONS_STP *)
  END_BLK
  // as ST:
  //   %TM39(IN := (VLV02_HMI_STP OR NOT VLV02_STS_AUTOMATIC) AND NOT VLV02_HMI_START);
  //   VLV2_ONS_STP := %TM39.Q;

// Rung 92: ALM
  LD 1
  AND( %M47               (* VLV02_T_ALMD_CNF_OPN_DN *)
  OR %M45                 (* VLV02_ALMD_CNF_OPN_DN *)
  )
  ANDN %M35               (* VLV02_RST_COUNT *)
  ANDN %M30               (* VLV02_HMI_START *)
  ANDN %MW151:X0
  ST %M45                 (* VLV02_ALMD_CNF_OPN_DN *)
  // as ST:
  //   VLV02_ALMD_CNF_OPN_DN := (VLV02_T_ALMD_CNF_OPN_DN OR VLV02_ALMD_CNF_OPN_DN) AND NOT VLV02_RST_COUNT AND NOT VLV02_HMI_START AND NOT %MW151:X0;

// Rung 93: ALM
  LD 1
  AND( %M49               (* VLV02_T_ALMD_CNF_CLS_DN *)
  OR %M46                 (* VLV02_ALMD_CNF_CLS_DN *)
  )
  ANDN %M35               (* VLV02_RST_COUNT *)
  ANDN %M30               (* VLV02_HMI_START *)
  ANDN %MW151:X0
  ST %M46                 (* VLV02_ALMD_CNF_CLS_DN *)
  // as ST:
  //   VLV02_ALMD_CNF_CLS_DN := (VLV02_T_ALMD_CNF_CLS_DN OR VLV02_ALMD_CNF_CLS_DN) AND NOT VLV02_RST_COUNT AND NOT VLV02_HMI_START AND NOT %MW151:X0;

// Rung 94
  LD 1
  MULTIFB
  LD 1
  AND %M21                (* HORARIOOFICINA_ACTIVE *)
  AND %M54                (* VLV02_HMI_STARTED *)
  ANDN %M45               (* VLV02_ALMD_CNF_OPN_DN *)
  ANDN %M46               (* VLV02_ALMD_CNF_CLS_DN *)
  ANDN %M58               (* VLV02_TON_HR_DN *)
  ST %MW2509:X0
  LD %MW2509:X0
  ST %M53                 (* VLV02_STS_AUTOMATIC *)
  BLK %TM17               (* VLV02_ONS *)
  LD %MW2509:X0
  IN
  OUT_BLK
  LD Q
  ST %M36                 (* VLV02_ONS_STS_AUTOMATIC *)
  END_BLK
  MULTIFB
  // as ST:
  //   %MW2509:X0 := HORARIOOFICINA_ACTIVE AND VLV02_HMI_STARTED AND NOT VLV02_ALMD_CNF_OPN_DN AND NOT VLV02_ALMD_CNF_CLS_DN AND NOT VLV02_TON_HR_DN;
  //   VLV02_STS_AUTOMATIC := %MW2509:X0;
  //   VLV02_ONS(IN := %MW2509:X0);
  //   VLV02_ONS_STS_AUTOMATIC := VLV02_ONS.Q;
  (* the ladder stored for this rung does not match its IL; not drawn *)

// Rung 95
  LD %M45                 (* VLV02_ALMD_CNF_OPN_DN *)
  OR %M46                 (* VLV02_ALMD_CNF_CLS_DN *)
  OR %M31                 (* VLV02_HMI_STP *)
  ST %M41                 (* VLV02_SAVE_DATETIME *)
  // as ST:
  //   VLV02_SAVE_DATETIME := VLV02_ALMD_CNF_OPN_DN OR VLV02_ALMD_CNF_CLS_DN OR VLV02_HMI_STP;

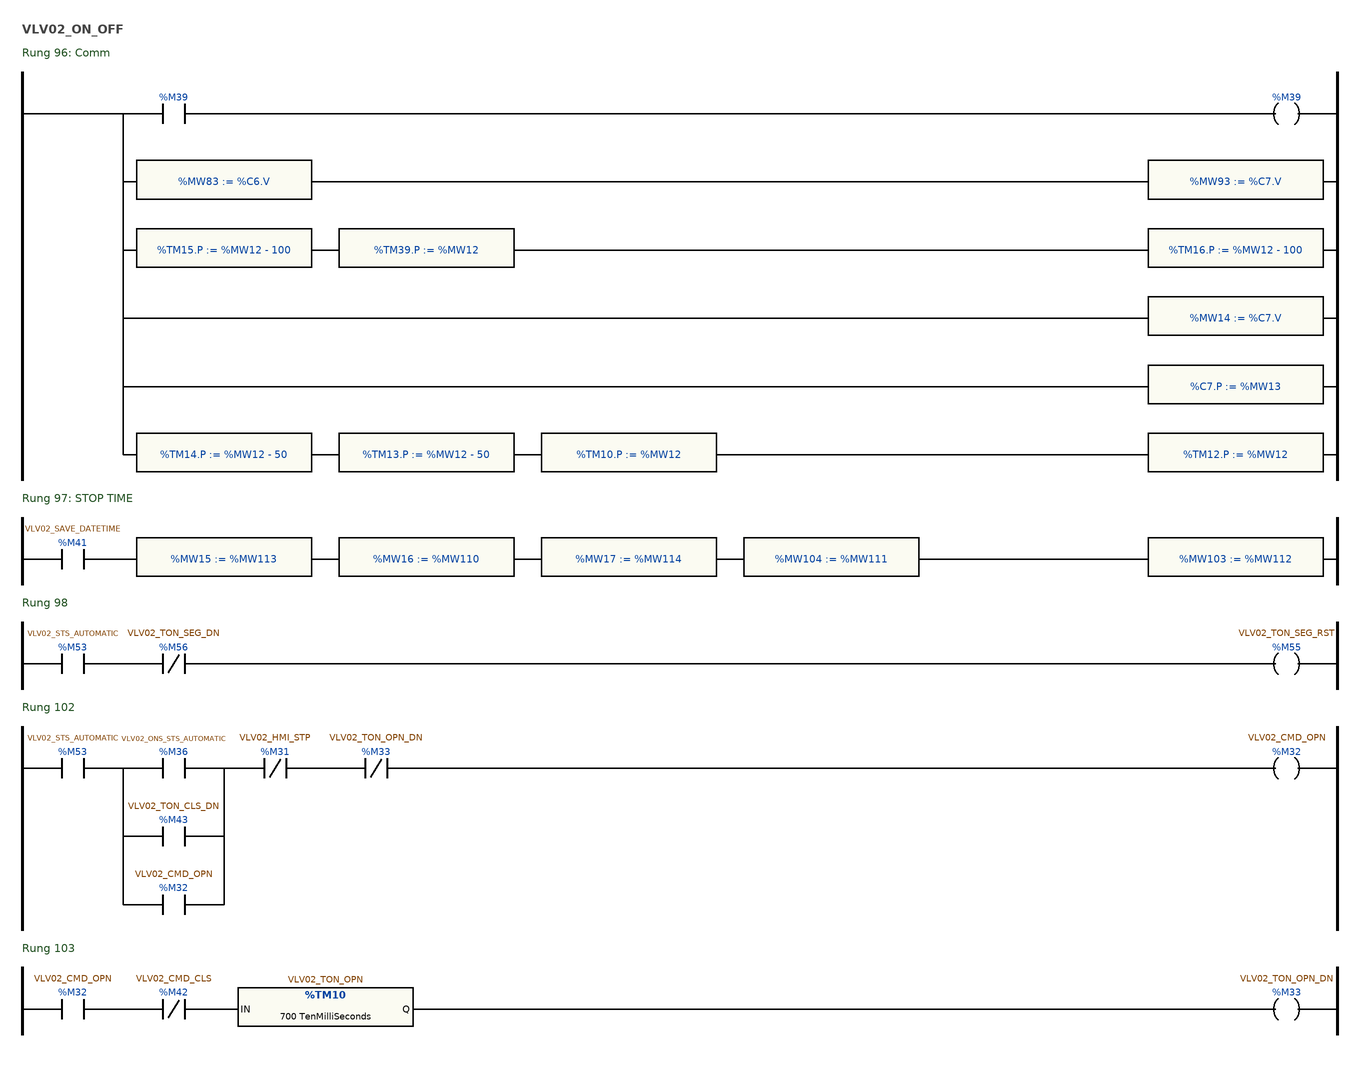

// Rung 96: Comm
  LD 1
  MPS
  AND %M39
  ST %M39
  MRD
  OPER [ %MW83 := %C6.V ] (* VLV02_CNT_MIN *)
  [ %MW93 := %C7.V ]      (* VLV02_CNT_HR *)
  MRD
  OPER [ %TM15.P := %MW12 - 100 ](* VLV02_T_CNF_OPN, VLV02_T_CNF_PRESET *)
  OPER [ %TM39.P := %MW12 ](* VLV02_T_CNF_PRESET *)
  [ %TM16.P := %MW12 - 100 ](* VLV02_T_CNF_CLS, VLV02_T_CNF_PRESET *)
  MRD
  [ %MW14 := %C7.V ]      (* VLV02_CNT_HR *)
  MRD
  [ %C7.P := %MW13 ]      (* VLV02_CNT_HR, VLV02_CNF_HR_PRESET *)
  MPP
  OPER [ %TM14.P := %MW12 - 50 ](* VLV02_TON_ALMD_CNF_CLS, VLV02_T_CNF_PRESET *)
  OPER [ %TM13.P := %MW12 - 50 ](* VLV02_TON_ALMD_CNF_OPN, VLV02_T_CNF_PRESET *)
  OPER [ %TM10.P := %MW12 ](* VLV02_TON_OPN, VLV02_T_CNF_PRESET *)
  [ %TM12.P := %MW12 ]    (* VLV02_TON_CLS, VLV02_T_CNF_PRESET *)
  // as ST:
  //   %M39 := %M39;
  //   %MW83 := VLV02_CNT_MIN.V;
  //   %MW93 := VLV02_CNT_HR.V;
  //   VLV02_T_CNF_OPN.P := VLV02_T_CNF_PRESET - 100;
  //   %TM39.P := VLV02_T_CNF_PRESET;
  //   VLV02_T_CNF_CLS.P := VLV02_T_CNF_PRESET - 100;
  //   %MW14 := VLV02_CNT_HR.V;
  //   VLV02_CNT_HR.P := VLV02_CNF_HR_PRESET;
  //   VLV02_TON_ALMD_CNF_CLS.P := VLV02_T_CNF_PRESET - 50;
  //   VLV02_TON_ALMD_CNF_OPN.P := VLV02_T_CNF_PRESET - 50;
  //   VLV02_TON_OPN.P := VLV02_T_CNF_PRESET;
  //   VLV02_TON_CLS.P := VLV02_T_CNF_PRESET;

// Rung 97: STOP TIME
  LD %M41                 (* VLV02_SAVE_DATETIME *)
  OPER [ %MW15 := %MW113 ](* VLV02_RTC_HHMM, MONTH *)
  OPER [ %MW16 := %MW110 ](* VLV02_RTC_MMDD, DAY *)
  OPER [ %MW17 := %MW114 ](* VLV02_RTC_YY, YEAR *)
  OPER [ %MW104 := %MW111 ](* HOUR *)
  [ %MW103 := %MW112 ]    (* MINUTES *)
  // as ST:
  //   IF VLV02_SAVE_DATETIME THEN VLV02_RTC_HHMM := MONTH; END_IF;
  //   IF VLV02_SAVE_DATETIME THEN VLV02_RTC_MMDD := DAY; END_IF;
  //   IF VLV02_SAVE_DATETIME THEN VLV02_RTC_YY := YEAR; END_IF;
  //   IF VLV02_SAVE_DATETIME THEN %MW104 := HOUR; END_IF;
  //   IF VLV02_SAVE_DATETIME THEN %MW103 := MINUTES; END_IF;

// Rung 98
  LD %M53                 (* VLV02_STS_AUTOMATIC *)
  ANDN %M56               (* VLV02_TON_SEG_DN *)
  ST %M55                 (* VLV02_TON_SEG_RST *)
  // as ST:
  //   VLV02_TON_SEG_RST := VLV02_STS_AUTOMATIC AND NOT VLV02_TON_SEG_DN;

// Rung 99
  BLK %C7                 (* VLV02_CNT_HR *)
  LD %M35                 (* VLV02_RST_COUNT *)
  OR( %M21                (* HORARIOOFICINA_ACTIVE *)
  RISING7
  )
  R
  LD %M57                 (* VLV02_TON_MIN_DN *)
  CU
  OUT_BLK
  LD D
  ST %M58                 (* VLV02_TON_HR_DN *)
  END_BLK
  // as ST:
  //   VLV02_CNT_HR(RISING7 := HORARIOOFICINA_ACTIVE, R := VLV02_RST_COUNT OR HORARIOOFICINA_ACTIVE, CU := VLV02_TON_MIN_DN);
  //   VLV02_TON_HR_DN := VLV02_CNT_HR.D;
  (* the ladder stored for this rung does not match its IL; not drawn *)

// Rung 100
  BLK %C6                 (* VLV02_CNT_MIN *)
  LD 1
  AND( %M35               (* VLV02_RST_COUNT *)
  OR %M57                 (* VLV02_TON_MIN_DN *)
  )
  OR( %M21                (* HORARIOOFICINA_ACTIVE *)
  RISING8
  )
  R
  LD %M56                 (* VLV02_TON_SEG_DN *)
  CU
  OUT_BLK
  LD D
  ST %M57                 (* VLV02_TON_MIN_DN *)
  END_BLK
  // as ST:
  //   VLV02_CNT_MIN(RISING8 := HORARIOOFICINA_ACTIVE, R := VLV02_RST_COUNT OR VLV02_TON_MIN_DN OR HORARIOOFICINA_ACTIVE, CU := VLV02_TON_SEG_DN);
  //   VLV02_TON_MIN_DN := VLV02_CNT_MIN.D;
  (* the ladder stored for this rung does not match its IL; not drawn *)

// Rung 101
  LD 1
  MULTIFB
  LD 1
  ST %MW2509:X1
  BLK %TM11               (* VLV02_TON_SEG *)
  LD %MW2509:X1
  AND %M53                (* VLV02_STS_AUTOMATIC *)
  AND %M55                (* VLV02_TON_SEG_RST *)
  IN
  OUT_BLK
  LD Q
  ST %MW2509:X0
  END_BLK
  BLK %C5                 (* VLV02_CNT_SEG *)
  LD %MW2509:X1
  AND( %M35               (* VLV02_RST_COUNT *)
  OR %M56                 (* VLV02_TON_SEG_DN *)
  )
  R
  LD %MW2509:X0
  CU
  OUT_BLK
  LD D
  ST %M56                 (* VLV02_TON_SEG_DN *)
  END_BLK
  MULTIFB
  // as ST:
  //   %MW2509:X1 := TRUE;
  //   VLV02_TON_SEG(IN := %MW2509:X1 AND VLV02_STS_AUTOMATIC AND VLV02_TON_SEG_RST);
  //   %MW2509:X0 := VLV02_TON_SEG.Q;
  //   VLV02_CNT_SEG(R := %MW2509:X1 AND (VLV02_RST_COUNT OR VLV02_TON_SEG_DN), CU := %MW2509:X0);
  //   VLV02_TON_SEG_DN := VLV02_CNT_SEG.D;
  (* the ladder stored for this rung does not match its IL; not drawn *)

// Rung 102
  LD %M53                 (* VLV02_STS_AUTOMATIC *)
  AND( %M36               (* VLV02_ONS_STS_AUTOMATIC *)
  OR %M43                 (* VLV02_TON_CLS_DN *)
  OR %M32                 (* VLV02_CMD_OPN *)
  )
  ANDN %M31               (* VLV02_HMI_STP *)
  ANDN %M33               (* VLV02_TON_OPN_DN *)
  ST %M32                 (* VLV02_CMD_OPN *)
  // as ST:
  //   VLV02_CMD_OPN := VLV02_STS_AUTOMATIC AND (VLV02_ONS_STS_AUTOMATIC OR VLV02_TON_CLS_DN OR VLV02_CMD_OPN) AND NOT VLV02_HMI_STP AND NOT VLV02_TON_OPN_DN;

// Rung 103
  BLK %TM10               (* VLV02_TON_OPN *)
  LD %M32                 (* VLV02_CMD_OPN *)
  ANDN %M42               (* VLV02_CMD_CLS *)
  IN
  OUT_BLK
  LD Q
  ST %M33                 (* VLV02_TON_OPN_DN *)
  END_BLK
  // as ST:
  //   VLV02_TON_OPN(IN := VLV02_CMD_OPN AND NOT VLV02_CMD_CLS);
  //   VLV02_TON_OPN_DN := VLV02_TON_OPN.Q;

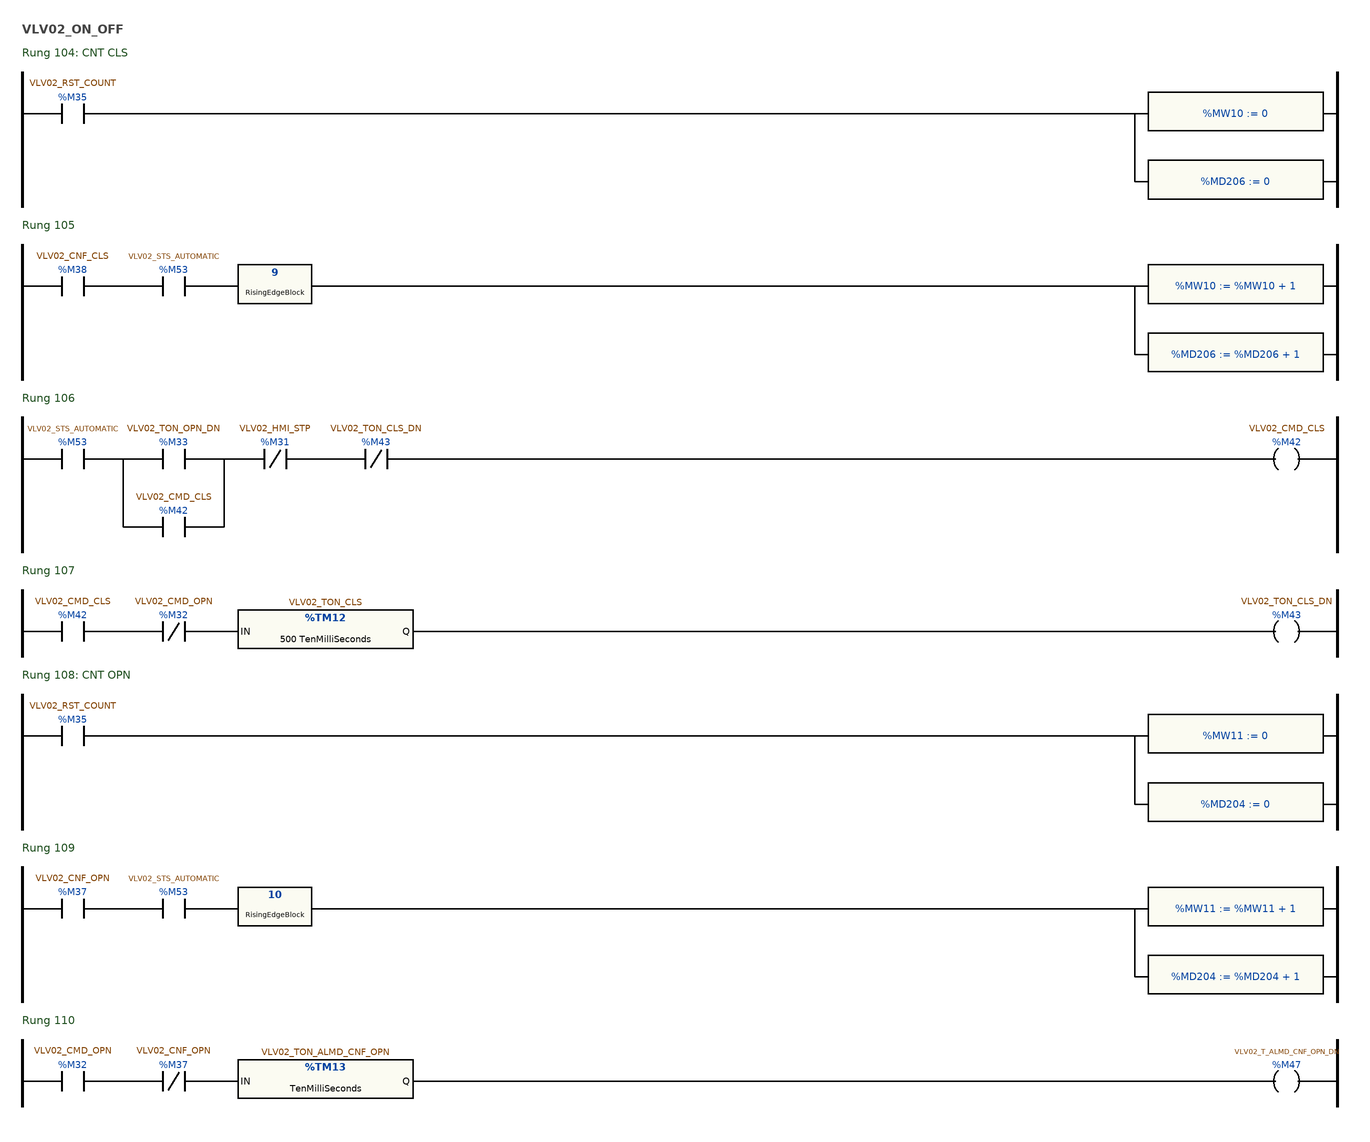

// Rung 104: CNT CLS
  LD %M35                 (* VLV02_RST_COUNT *)
  [ %MW10 := 0 ]          (* VLV02_CNT_CLS_ACC *)
  [ %MD206 := 0 ]         (* VLV02_CNT_CLS_ACC2 *)
  // as ST:
  //   IF VLV02_RST_COUNT THEN VLV02_CNT_CLS_ACC := 0; END_IF;
  //   IF VLV02_RST_COUNT THEN VLV02_CNT_CLS_ACC2 := 0; END_IF;

// Rung 105
  LD %M38                 (* VLV02_CNF_CLS *)
  AND %M53                (* VLV02_STS_AUTOMATIC *)
  RISING9
  [ %MW10 := %MW10 + 1 ]  (* VLV02_CNT_CLS_ACC, VLV02_CNT_CLS_ACC *)
  [ %MD206 := %MD206 + 1 ](* VLV02_CNT_CLS_ACC2, VLV02_CNT_CLS_ACC2 *)
  // as ST:
  //   IF RISING(VLV02_CNF_CLS AND VLV02_STS_AUTOMATIC) THEN VLV02_CNT_CLS_ACC := VLV02_CNT_CLS_ACC + 1; END_IF;
  //   IF RISING(VLV02_CNF_CLS AND VLV02_STS_AUTOMATIC) THEN VLV02_CNT_CLS_ACC2 := VLV02_CNT_CLS_ACC2 + 1; END_IF;

// Rung 106
  LD %M53                 (* VLV02_STS_AUTOMATIC *)
  AND( %M33               (* VLV02_TON_OPN_DN *)
  OR %M42                 (* VLV02_CMD_CLS *)
  )
  ANDN %M31               (* VLV02_HMI_STP *)
  ANDN %M43               (* VLV02_TON_CLS_DN *)
  ST %M42                 (* VLV02_CMD_CLS *)
  // as ST:
  //   VLV02_CMD_CLS := VLV02_STS_AUTOMATIC AND (VLV02_TON_OPN_DN OR VLV02_CMD_CLS) AND NOT VLV02_HMI_STP AND NOT VLV02_TON_CLS_DN;

// Rung 107
  BLK %TM12               (* VLV02_TON_CLS *)
  LD %M42                 (* VLV02_CMD_CLS *)
  ANDN %M32               (* VLV02_CMD_OPN *)
  IN
  OUT_BLK
  LD Q
  ST %M43                 (* VLV02_TON_CLS_DN *)
  END_BLK
  // as ST:
  //   VLV02_TON_CLS(IN := VLV02_CMD_CLS AND NOT VLV02_CMD_OPN);
  //   VLV02_TON_CLS_DN := VLV02_TON_CLS.Q;

// Rung 108: CNT OPN
  LD %M35                 (* VLV02_RST_COUNT *)
  [ %MW11 := 0 ]          (* VLV02_CNT_OPN_ACC *)
  [ %MD204 := 0 ]         (* VLV02_CNT_OPN_ACC2 *)
  // as ST:
  //   IF VLV02_RST_COUNT THEN VLV02_CNT_OPN_ACC := 0; END_IF;
  //   IF VLV02_RST_COUNT THEN VLV02_CNT_OPN_ACC2 := 0; END_IF;

// Rung 109
  LD %M37                 (* VLV02_CNF_OPN *)
  AND %M53                (* VLV02_STS_AUTOMATIC *)
  RISING10
  [ %MW11 := %MW11 + 1 ]  (* VLV02_CNT_OPN_ACC, VLV02_CNT_OPN_ACC *)
  [ %MD204 := %MD204 + 1 ](* VLV02_CNT_OPN_ACC2, VLV02_CNT_OPN_ACC2 *)
  // as ST:
  //   IF RISING(VLV02_CNF_OPN AND VLV02_STS_AUTOMATIC) THEN VLV02_CNT_OPN_ACC := VLV02_CNT_OPN_ACC + 1; END_IF;
  //   IF RISING(VLV02_CNF_OPN AND VLV02_STS_AUTOMATIC) THEN VLV02_CNT_OPN_ACC2 := VLV02_CNT_OPN_ACC2 + 1; END_IF;

// Rung 110
  BLK %TM13               (* VLV02_TON_ALMD_CNF_OPN *)
  LD %M32                 (* VLV02_CMD_OPN *)
  ANDN %M37               (* VLV02_CNF_OPN *)
  IN
  OUT_BLK
  LD Q
  ST %M47                 (* VLV02_T_ALMD_CNF_OPN_DN *)
  END_BLK
  // as ST:
  //   VLV02_TON_ALMD_CNF_OPN(IN := VLV02_CMD_OPN AND NOT VLV02_CNF_OPN);
  //   VLV02_T_ALMD_CNF_OPN_DN := VLV02_TON_ALMD_CNF_OPN.Q;

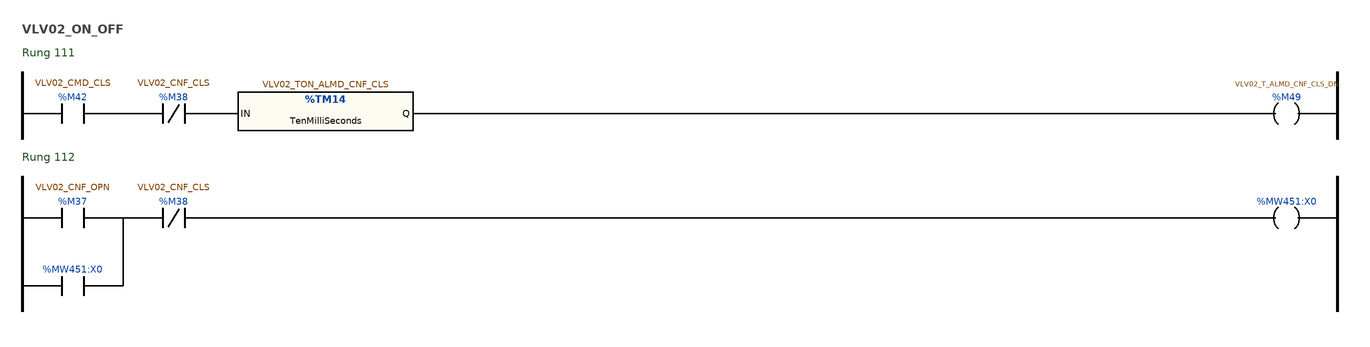

// Rung 111
  BLK %TM14               (* VLV02_TON_ALMD_CNF_CLS *)
  LD %M42                 (* VLV02_CMD_CLS *)
  ANDN %M38               (* VLV02_CNF_CLS *)
  IN
  OUT_BLK
  LD Q
  ST %M49                 (* VLV02_T_ALMD_CNF_CLS_DN *)
  END_BLK
  // as ST:
  //   VLV02_TON_ALMD_CNF_CLS(IN := VLV02_CMD_CLS AND NOT VLV02_CNF_CLS);
  //   VLV02_T_ALMD_CNF_CLS_DN := VLV02_TON_ALMD_CNF_CLS.Q;

// Rung 112
  LD %M37                 (* VLV02_CNF_OPN *)
  OR %MW451:X0
  ANDN %M38               (* VLV02_CNF_CLS *)
  ST %MW451:X0
  // as ST:
  //   %MW451:X0 := (VLV02_CNF_OPN OR %MW451:X0) AND NOT VLV02_CNF_CLS;

POU VLV03_ANALOG
  (* SectionNumber=4 *)

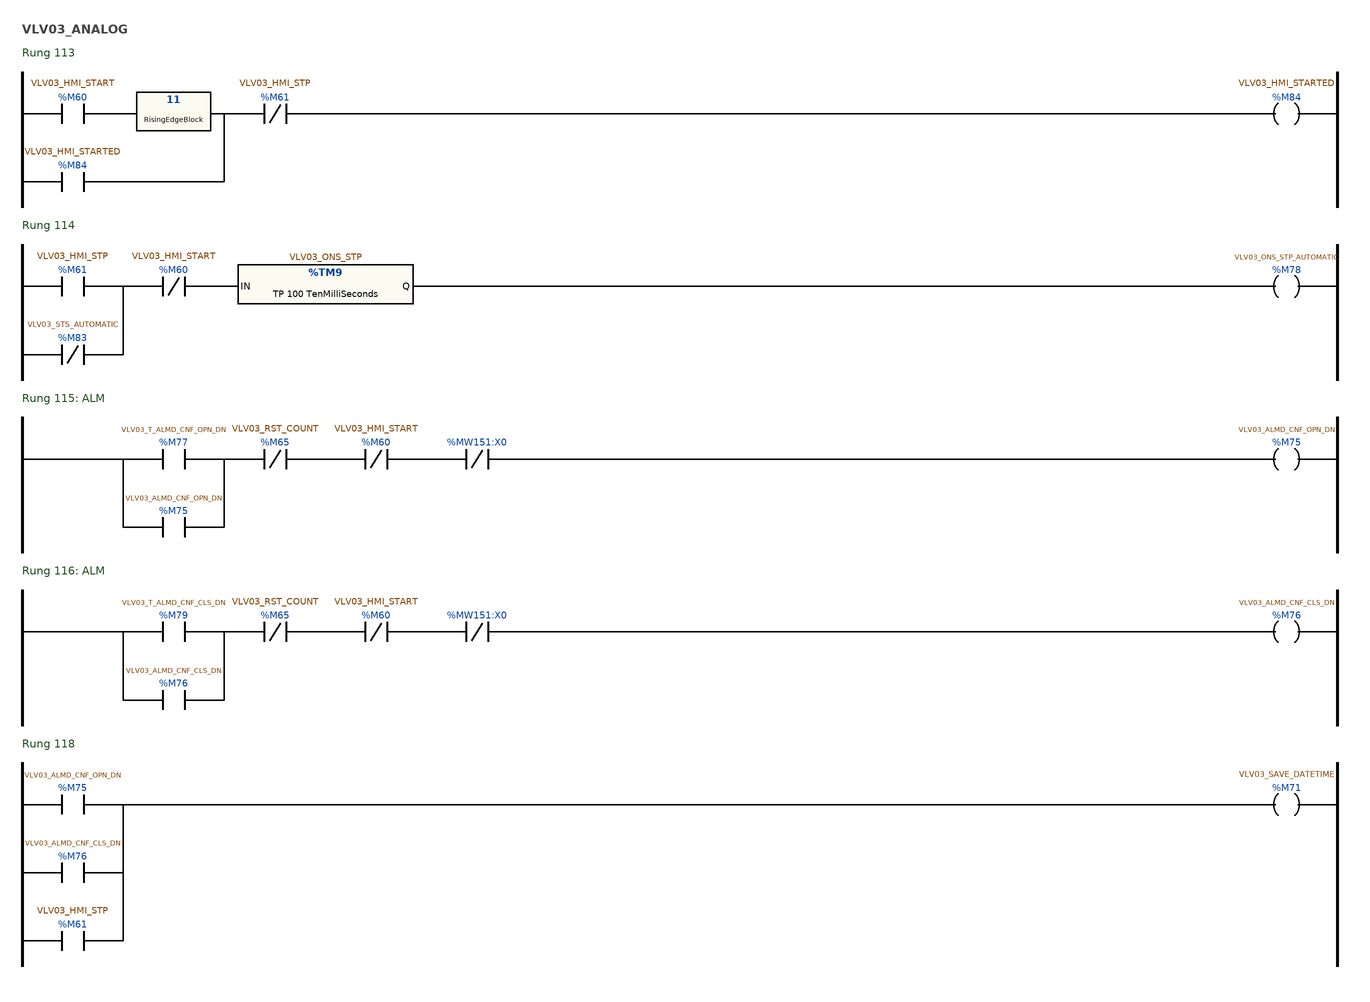

// Rung 113
  LD %M60                 (* VLV03_HMI_START *)
  RISING11
  OR %M84                 (* VLV03_HMI_STARTED *)
  ANDN %M61               (* VLV03_HMI_STP *)
  ST %M84                 (* VLV03_HMI_STARTED *)
  // as ST:
  //   VLV03_HMI_STARTED := (RISING(VLV03_HMI_START) OR VLV03_HMI_STARTED) AND NOT VLV03_HMI_STP;

// Rung 114
  BLK %TM9                (* VLV03_ONS_STP *)
  LD %M61                 (* VLV03_HMI_STP *)
  ORN %M83                (* VLV03_STS_AUTOMATIC *)
  ANDN %M60               (* VLV03_HMI_START *)
  IN
  OUT_BLK
  LD Q
  ST %M78                 (* VLV03_ONS_STP_AUTOMATIC *)
  END_BLK
  // as ST:
  //   VLV03_ONS_STP(IN := (VLV03_HMI_STP OR NOT VLV03_STS_AUTOMATIC) AND NOT VLV03_HMI_START);
  //   VLV03_ONS_STP_AUTOMATIC := VLV03_ONS_STP.Q;

// Rung 115: ALM
  LD 1
  AND( %M77               (* VLV03_T_ALMD_CNF_OPN_DN *)
  OR %M75                 (* VLV03_ALMD_CNF_OPN_DN *)
  )
  ANDN %M65               (* VLV03_RST_COUNT *)
  ANDN %M60               (* VLV03_HMI_START *)
  ANDN %MW151:X0
  ST %M75                 (* VLV03_ALMD_CNF_OPN_DN *)
  // as ST:
  //   VLV03_ALMD_CNF_OPN_DN := (VLV03_T_ALMD_CNF_OPN_DN OR VLV03_ALMD_CNF_OPN_DN) AND NOT VLV03_RST_COUNT AND NOT VLV03_HMI_START AND NOT %MW151:X0;

// Rung 116: ALM
  LD 1
  AND( %M79               (* VLV03_T_ALMD_CNF_CLS_DN *)
  OR %M76                 (* VLV03_ALMD_CNF_CLS_DN *)
  )
  ANDN %M65               (* VLV03_RST_COUNT *)
  ANDN %M60               (* VLV03_HMI_START *)
  ANDN %MW151:X0
  ST %M76                 (* VLV03_ALMD_CNF_CLS_DN *)
  // as ST:
  //   VLV03_ALMD_CNF_CLS_DN := (VLV03_T_ALMD_CNF_CLS_DN OR VLV03_ALMD_CNF_CLS_DN) AND NOT VLV03_RST_COUNT AND NOT VLV03_HMI_START AND NOT %MW151:X0;

// Rung 117
  LD 1
  MULTIFB
  LD 1
  AND %M21                (* HORARIOOFICINA_ACTIVE *)
  AND %M84                (* VLV03_HMI_STARTED *)
  ANDN %M75               (* VLV03_ALMD_CNF_OPN_DN *)
  ANDN %M76               (* VLV03_ALMD_CNF_CLS_DN *)
  AND %MW432:X0
  ANDN %M88               (* VLV03_TON_HR_DN *)
  ST %MW2509:X0
  LD %MW2509:X0
  ST %M83                 (* VLV03_STS_AUTOMATIC *)
  BLK %TM27               (* VLV03_ONS_01 *)
  LD %MW2509:X0
  IN
  OUT_BLK
  LD Q
  ST %M66                 (* VLV03_ONS_STR_AUTOMATIC *)
  END_BLK
  MULTIFB
  // as ST:
  //   %MW2509:X0 := HORARIOOFICINA_ACTIVE AND VLV03_HMI_STARTED AND NOT VLV03_ALMD_CNF_OPN_DN AND NOT VLV03_ALMD_CNF_CLS_DN AND %MW432:X0 AND NOT VLV03_TON_HR_DN;
  //   VLV03_STS_AUTOMATIC := %MW2509:X0;
  //   VLV03_ONS_01(IN := %MW2509:X0);
  //   VLV03_ONS_STR_AUTOMATIC := VLV03_ONS_01.Q;
  (* the ladder stored for this rung does not match its IL; not drawn *)

// Rung 118
  LD %M75                 (* VLV03_ALMD_CNF_OPN_DN *)
  OR %M76                 (* VLV03_ALMD_CNF_CLS_DN *)
  OR %M61                 (* VLV03_HMI_STP *)
  ST %M71                 (* VLV03_SAVE_DATETIME *)
  // as ST:
  //   VLV03_SAVE_DATETIME := VLV03_ALMD_CNF_OPN_DN OR VLV03_ALMD_CNF_CLS_DN OR VLV03_HMI_STP;

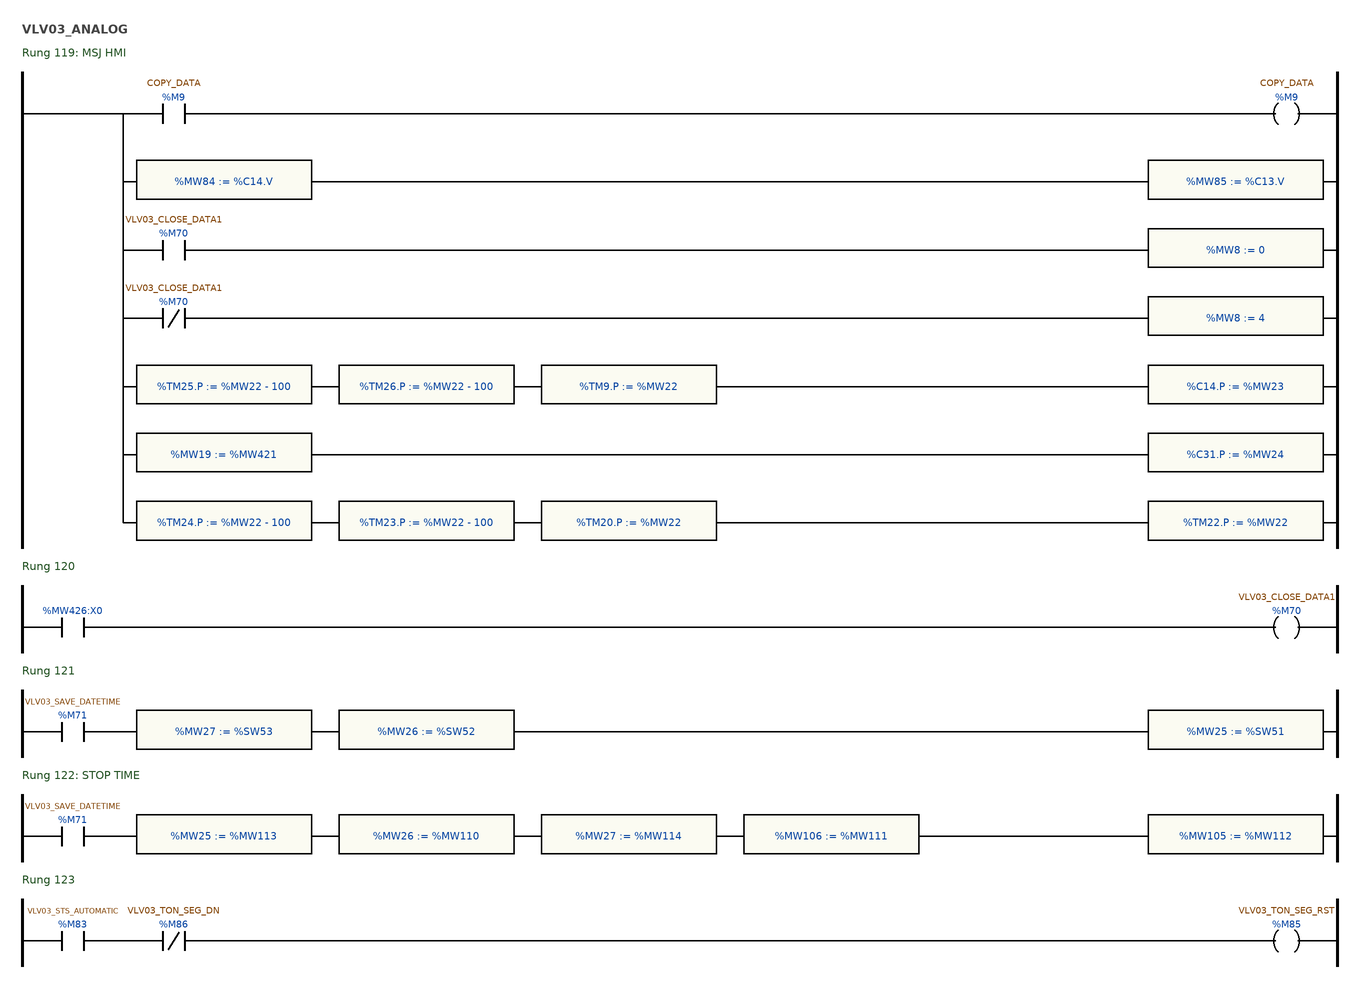

// Rung 119: MSJ HMI
  LD 1
  MPS
  AND %M9                 (* COPY_DATA *)
  ST %M9                  (* COPY_DATA *)
  MRD
  OPER [ %MW84 := %C14.V ](* VLV03_CNT_HR *)
  [ %MW85 := %C13.V ]     (* VLV03_CNT_MIN *)
  MRD
  AND %M70                (* VLV03_CLOSE_DATA1 *)
  [ %MW8 := 0 ]
  MRD
  ANDN %M70               (* VLV03_CLOSE_DATA1 *)
  [ %MW8 := 4 ]
  MRD
  OPER [ %TM25.P := %MW22 - 100 ](* VLV03_T_CNF_OPN, VLV03_T_CNF_PRESET *)
  OPER [ %TM26.P := %MW22 - 100 ](* VLV03_T_CNF_CLS, VLV03_T_CNF_PRESET *)
  OPER [ %TM9.P := %MW22 ](* VLV03_ONS_STP, VLV03_T_CNF_PRESET *)
  [ %C14.P := %MW23 ]     (* VLV03_CNT_HR, VLV03_CNF_HR_PRESET *)
  MRD
  OPER [ %MW19 := %MW421 ](* VLV03_CV_ACTUAL *)
  [ %C31.P := %MW24 ]     (* VLV03_SETPOINT_ALTO *)
  MPP
  OPER [ %TM24.P := %MW22 - 100 ](* VLV03_TON_ALMD_CNF_CLS, VLV03_T_CNF_PRESET *)
  OPER [ %TM23.P := %MW22 - 100 ](* VLV03_TON_ALMD_CNF_OPN, VLV03_T_CNF_PRESET *)
  OPER [ %TM20.P := %MW22 ](* VLV03_TON_OPN, VLV03_T_CNF_PRESET *)
  [ %TM22.P := %MW22 ]    (* VLV03_TON_CLS, VLV03_T_CNF_PRESET *)
  // as ST:
  //   COPY_DATA := COPY_DATA;
  //   %MW84 := VLV03_CNT_HR.V;
  //   %MW85 := VLV03_CNT_MIN.V;
  //   IF VLV03_CLOSE_DATA1 THEN %MW8 := 0; END_IF;
  //   IF NOT VLV03_CLOSE_DATA1 THEN %MW8 := 4; END_IF;
  //   VLV03_T_CNF_OPN.P := VLV03_T_CNF_PRESET - 100;
  //   VLV03_T_CNF_CLS.P := VLV03_T_CNF_PRESET - 100;
  //   VLV03_ONS_STP.P := VLV03_T_CNF_PRESET;
  //   VLV03_CNT_HR.P := VLV03_CNF_HR_PRESET;
  //   VLV03_CV_ACTUAL := %MW421;
  //   %C31.P := VLV03_SETPOINT_ALTO;
  //   VLV03_TON_ALMD_CNF_CLS.P := VLV03_T_CNF_PRESET - 100;
  //   VLV03_TON_ALMD_CNF_OPN.P := VLV03_T_CNF_PRESET - 100;
  //   VLV03_TON_OPN.P := VLV03_T_CNF_PRESET;
  //   VLV03_TON_CLS.P := VLV03_T_CNF_PRESET;

// Rung 120
  LD %MW426:X0
  ST %M70                 (* VLV03_CLOSE_DATA1 *)
  // as ST:
  //   VLV03_CLOSE_DATA1 := %MW426:X0;

// Rung 121
  LD %M71                 (* VLV03_SAVE_DATETIME *)
  OPER [ %MW27 := %SW53 ] (* VLV03_RTC_YY, SW_RTCCCYY *)
  OPER [ %MW26 := %SW52 ] (* VLV03_RTC_MMDD, SW_RTCMMDD *)
  [ %MW25 := %SW51 ]      (* VLV03_RTC_HHMM, SW_RTCHHMM *)
  // as ST:
  //   IF VLV03_SAVE_DATETIME THEN VLV03_RTC_YY := SW_RTCCCYY; END_IF;
  //   IF VLV03_SAVE_DATETIME THEN VLV03_RTC_MMDD := SW_RTCMMDD; END_IF;
  //   IF VLV03_SAVE_DATETIME THEN VLV03_RTC_HHMM := SW_RTCHHMM; END_IF;

// Rung 122: STOP TIME
  LD %M71                 (* VLV03_SAVE_DATETIME *)
  OPER [ %MW25 := %MW113 ](* VLV03_RTC_HHMM, MONTH *)
  OPER [ %MW26 := %MW110 ](* VLV03_RTC_MMDD, DAY *)
  OPER [ %MW27 := %MW114 ](* VLV03_RTC_YY, YEAR *)
  OPER [ %MW106 := %MW111 ](* HOUR *)
  [ %MW105 := %MW112 ]    (* MINUTES *)
  // as ST:
  //   IF VLV03_SAVE_DATETIME THEN VLV03_RTC_HHMM := MONTH; END_IF;
  //   IF VLV03_SAVE_DATETIME THEN VLV03_RTC_MMDD := DAY; END_IF;
  //   IF VLV03_SAVE_DATETIME THEN VLV03_RTC_YY := YEAR; END_IF;
  //   IF VLV03_SAVE_DATETIME THEN %MW106 := HOUR; END_IF;
  //   IF VLV03_SAVE_DATETIME THEN %MW105 := MINUTES; END_IF;

// Rung 123
  LD %M83                 (* VLV03_STS_AUTOMATIC *)
  ANDN %M86               (* VLV03_TON_SEG_DN *)
  ST %M85                 (* VLV03_TON_SEG_RST *)
  // as ST:
  //   VLV03_TON_SEG_RST := VLV03_STS_AUTOMATIC AND NOT VLV03_TON_SEG_DN;

// Rung 124
  BLK %C14                (* VLV03_CNT_HR *)
  LD %M65                 (* VLV03_RST_COUNT *)
  OR( %M21                (* HORARIOOFICINA_ACTIVE *)
  RISING12
  )
  R
  LD %M87                 (* VLV03_TON_MIN_DN *)
  CU
  OUT_BLK
  LD D
  ST %M88                 (* VLV03_TON_HR_DN *)
  END_BLK
  // as ST:
  //   VLV03_CNT_HR(RISING12 := HORARIOOFICINA_ACTIVE, R := VLV03_RST_COUNT OR HORARIOOFICINA_ACTIVE, CU := VLV03_TON_MIN_DN);
  //   VLV03_TON_HR_DN := VLV03_CNT_HR.D;
  (* the ladder stored for this rung does not match its IL; not drawn *)

// Rung 125
  BLK %C13                (* VLV03_CNT_MIN *)
  LD 1
  AND( %M65               (* VLV03_RST_COUNT *)
  OR %M87                 (* VLV03_TON_MIN_DN *)
  )
  OR( %M21                (* HORARIOOFICINA_ACTIVE *)
  RISING13
  )
  R
  LD %M86                 (* VLV03_TON_SEG_DN *)
  CU
  OUT_BLK
  LD D
  ST %M87                 (* VLV03_TON_MIN_DN *)
  END_BLK
  // as ST:
  //   VLV03_CNT_MIN(RISING13 := HORARIOOFICINA_ACTIVE, R := VLV03_RST_COUNT OR VLV03_TON_MIN_DN OR HORARIOOFICINA_ACTIVE, CU := VLV03_TON_SEG_DN);
  //   VLV03_TON_MIN_DN := VLV03_CNT_MIN.D;
  (* the ladder stored for this rung does not match its IL; not drawn *)

// Rung 126
  LD 1
  MULTIFB
  LD 1
  ST %MW2509:X1
  BLK %TM21               (* VLV03_TON_SEG *)
  LD %MW2509:X1
  AND %M83                (* VLV03_STS_AUTOMATIC *)
  AND %M85                (* VLV03_TON_SEG_RST *)
  IN
  OUT_BLK
  LD Q
  ST %MW2509:X0
  END_BLK
  BLK %C12                (* VLV03_CNT_SEG *)
  LD %MW2509:X1
  AND( %M65               (* VLV03_RST_COUNT *)
  OR %M86                 (* VLV03_TON_SEG_DN *)
  )
  R
  LD %MW2509:X0
  CU
  OUT_BLK
  LD D
  ST %M86                 (* VLV03_TON_SEG_DN *)
  END_BLK
  MULTIFB
  // as ST:
  //   %MW2509:X1 := TRUE;
  //   VLV03_TON_SEG(IN := %MW2509:X1 AND VLV03_STS_AUTOMATIC AND VLV03_TON_SEG_RST);
  //   %MW2509:X0 := VLV03_TON_SEG.Q;
  //   VLV03_CNT_SEG(R := %MW2509:X1 AND (VLV03_RST_COUNT OR VLV03_TON_SEG_DN), CU := %MW2509:X0);
  //   VLV03_TON_SEG_DN := VLV03_CNT_SEG.D;
  (* the ladder stored for this rung does not match its IL; not drawn *)

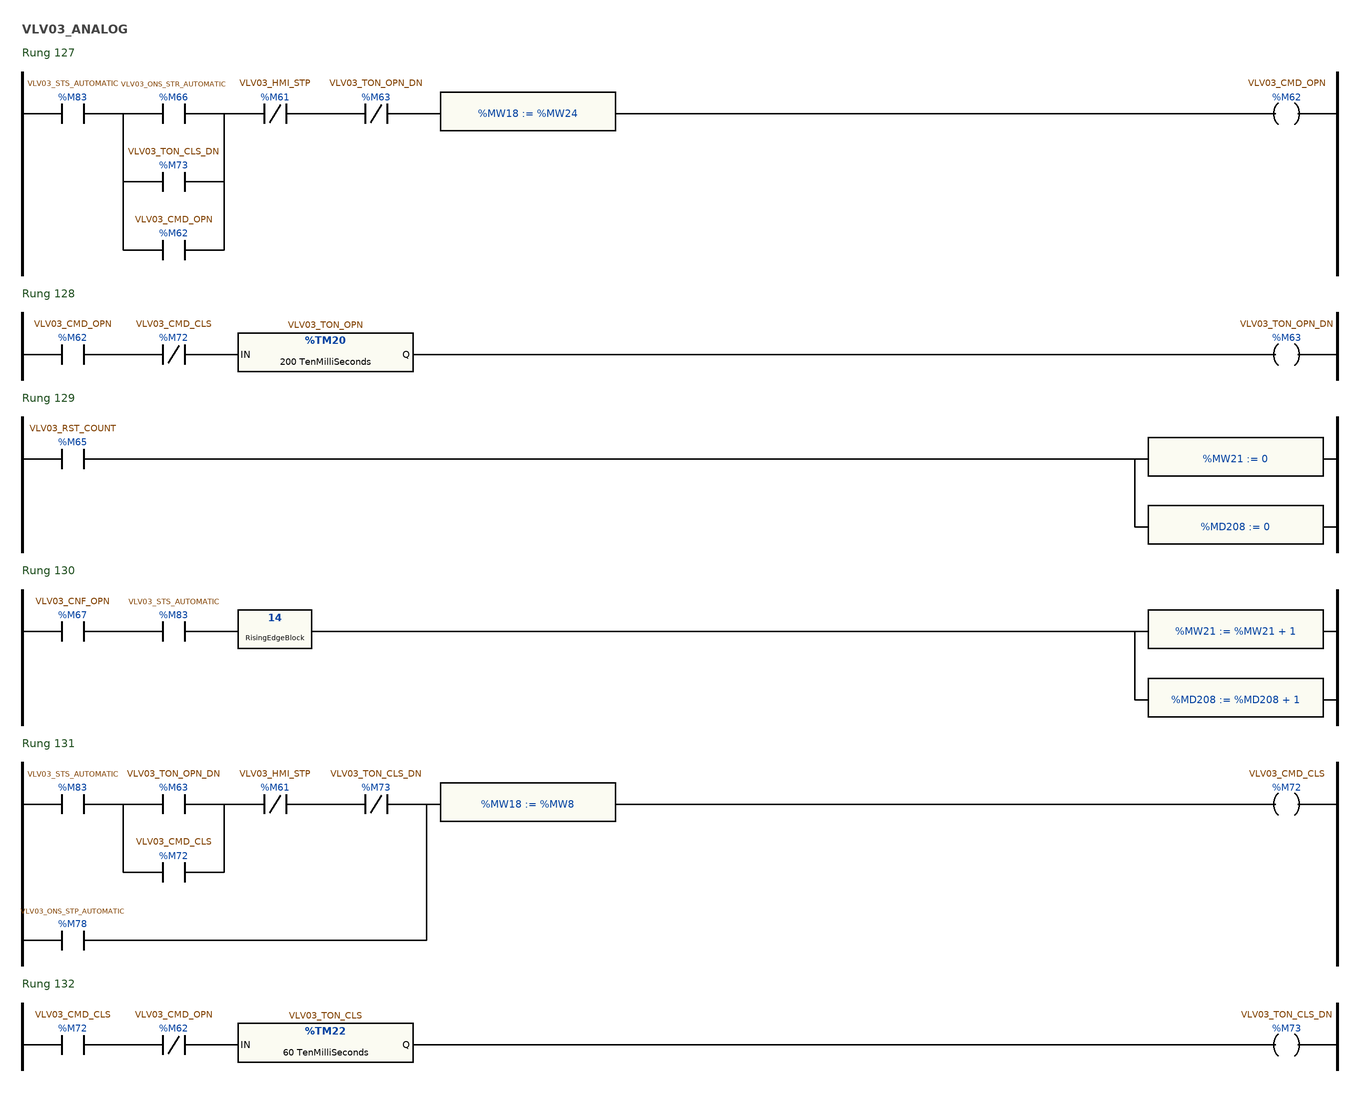

// Rung 127
  LD %M83                 (* VLV03_STS_AUTOMATIC *)
  AND( %M66               (* VLV03_ONS_STR_AUTOMATIC *)
  OR %M73                 (* VLV03_TON_CLS_DN *)
  OR %M62                 (* VLV03_CMD_OPN *)
  )
  ANDN %M61               (* VLV03_HMI_STP *)
  ANDN %M63               (* VLV03_TON_OPN_DN *)
  OPER [ %MW18 := %MW24 ] (* VLV03_SP_ACTUAL, VLV03_SETPOINT_ALTO *)
  ST %M62                 (* VLV03_CMD_OPN *)
  // as ST:
  //   IF VLV03_STS_AUTOMATIC AND (VLV03_ONS_STR_AUTOMATIC OR VLV03_TON_CLS_DN OR VLV03_CMD_OPN) AND NOT VLV03_HMI_STP AND NOT VLV03_TON_OPN_DN THEN VLV03_SP_ACTUAL := VLV03_SETPOINT_ALTO; END_IF;
  //   VLV03_CMD_OPN := VLV03_STS_AUTOMATIC AND (VLV03_ONS_STR_AUTOMATIC OR VLV03_TON_CLS_DN OR VLV03_CMD_OPN) AND NOT VLV03_HMI_STP AND NOT VLV03_TON_OPN_DN;

// Rung 128
  BLK %TM20               (* VLV03_TON_OPN *)
  LD %M62                 (* VLV03_CMD_OPN *)
  ANDN %M72               (* VLV03_CMD_CLS *)
  IN
  OUT_BLK
  LD Q
  ST %M63                 (* VLV03_TON_OPN_DN *)
  END_BLK
  // as ST:
  //   VLV03_TON_OPN(IN := VLV03_CMD_OPN AND NOT VLV03_CMD_CLS);
  //   VLV03_TON_OPN_DN := VLV03_TON_OPN.Q;

// Rung 129
  LD %M65                 (* VLV03_RST_COUNT *)
  [ %MW21 := 0 ]          (* VLV03_CNT_OPN_ACC *)
  [ %MD208 := 0 ]         (* VLV03_CNT_OPN_ACC2 *)
  // as ST:
  //   IF VLV03_RST_COUNT THEN VLV03_CNT_OPN_ACC := 0; END_IF;
  //   IF VLV03_RST_COUNT THEN VLV03_CNT_OPN_ACC2 := 0; END_IF;

// Rung 130
  LD %M67                 (* VLV03_CNF_OPN *)
  AND %M83                (* VLV03_STS_AUTOMATIC *)
  RISING14
  [ %MW21 := %MW21 + 1 ]  (* VLV03_CNT_OPN_ACC, VLV03_CNT_OPN_ACC *)
  [ %MD208 := %MD208 + 1 ](* VLV03_CNT_OPN_ACC2, VLV03_CNT_OPN_ACC2 *)
  // as ST:
  //   IF RISING(VLV03_CNF_OPN AND VLV03_STS_AUTOMATIC) THEN VLV03_CNT_OPN_ACC := VLV03_CNT_OPN_ACC + 1; END_IF;
  //   IF RISING(VLV03_CNF_OPN AND VLV03_STS_AUTOMATIC) THEN VLV03_CNT_OPN_ACC2 := VLV03_CNT_OPN_ACC2 + 1; END_IF;

// Rung 131
  LD %M83                 (* VLV03_STS_AUTOMATIC *)
  AND( %M63               (* VLV03_TON_OPN_DN *)
  OR %M72                 (* VLV03_CMD_CLS *)
  )
  ANDN %M61               (* VLV03_HMI_STP *)
  ANDN %M73               (* VLV03_TON_CLS_DN *)
  OR %M78                 (* VLV03_ONS_STP_AUTOMATIC *)
  OPER [ %MW18 := %MW8 ]  (* VLV03_SP_ACTUAL *)
  ST %M72                 (* VLV03_CMD_CLS *)
  // as ST:
  //   IF VLV03_STS_AUTOMATIC AND (VLV03_TON_OPN_DN OR VLV03_CMD_CLS) AND NOT VLV03_HMI_STP AND NOT VLV03_TON_CLS_DN OR VLV03_ONS_STP_AUTOMATIC THEN VLV03_SP_ACTUAL := %MW8; END_IF;
  //   VLV03_CMD_CLS := VLV03_STS_AUTOMATIC AND (VLV03_TON_OPN_DN OR VLV03_CMD_CLS) AND NOT VLV03_HMI_STP AND NOT VLV03_TON_CLS_DN OR VLV03_ONS_STP_AUTOMATIC;

// Rung 132
  BLK %TM22               (* VLV03_TON_CLS *)
  LD %M72                 (* VLV03_CMD_CLS *)
  ANDN %M62               (* VLV03_CMD_OPN *)
  IN
  OUT_BLK
  LD Q
  ST %M73                 (* VLV03_TON_CLS_DN *)
  END_BLK
  // as ST:
  //   VLV03_TON_CLS(IN := VLV03_CMD_CLS AND NOT VLV03_CMD_OPN);
  //   VLV03_TON_CLS_DN := VLV03_TON_CLS.Q;

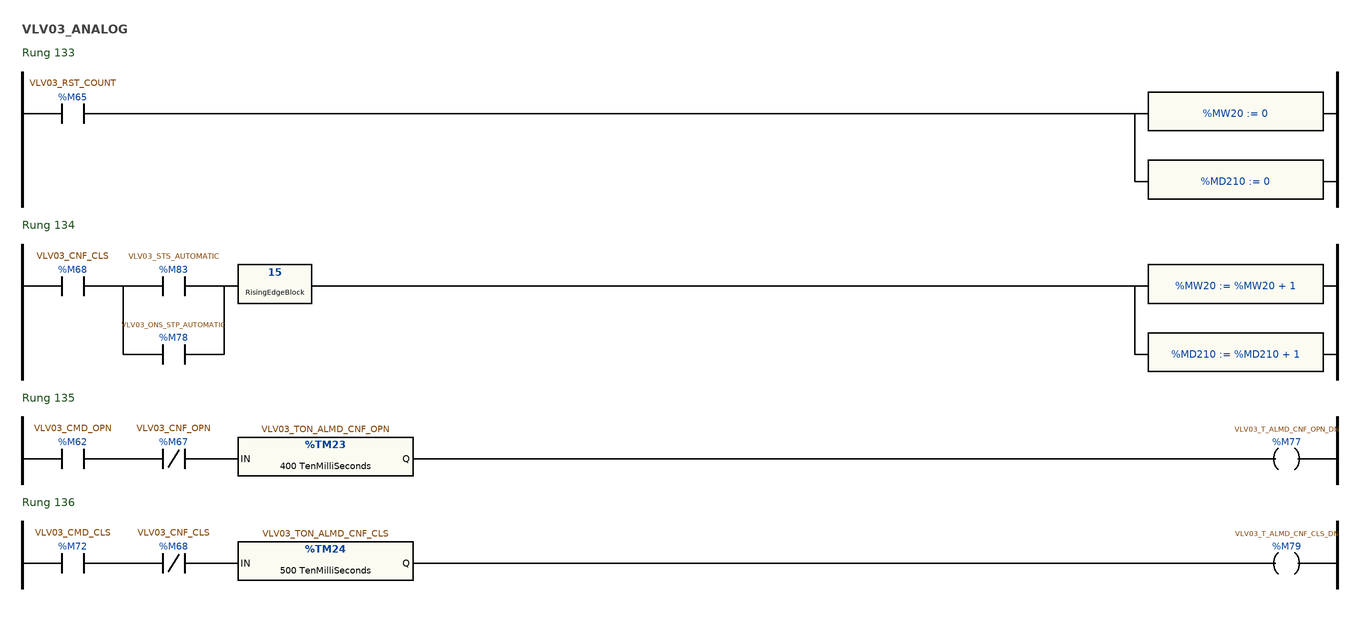

// Rung 133
  LD %M65                 (* VLV03_RST_COUNT *)
  [ %MW20 := 0 ]          (* VLV03_CNT_CLS_ACC *)
  [ %MD210 := 0 ]         (* VLV03_CNT_CLS_ACC2 *)
  // as ST:
  //   IF VLV03_RST_COUNT THEN VLV03_CNT_CLS_ACC := 0; END_IF;
  //   IF VLV03_RST_COUNT THEN VLV03_CNT_CLS_ACC2 := 0; END_IF;

// Rung 134
  LD %M68                 (* VLV03_CNF_CLS *)
  AND( %M83               (* VLV03_STS_AUTOMATIC *)
  OR %M78                 (* VLV03_ONS_STP_AUTOMATIC *)
  )
  RISING15
  [ %MW20 := %MW20 + 1 ]  (* VLV03_CNT_CLS_ACC, VLV03_CNT_CLS_ACC *)
  [ %MD210 := %MD210 + 1 ](* VLV03_CNT_CLS_ACC2, VLV03_CNT_CLS_ACC2 *)
  // as ST:
  //   IF RISING(VLV03_CNF_CLS AND (VLV03_STS_AUTOMATIC OR VLV03_ONS_STP_AUTOMATIC)) THEN VLV03_CNT_CLS_ACC := VLV03_CNT_CLS_ACC + 1; END_IF;
  //   IF RISING(VLV03_CNF_CLS AND (VLV03_STS_AUTOMATIC OR VLV03_ONS_STP_AUTOMATIC)) THEN VLV03_CNT_CLS_ACC2 := VLV03_CNT_CLS_ACC2 + 1; END_IF;

// Rung 135
  BLK %TM23               (* VLV03_TON_ALMD_CNF_OPN *)
  LD %M62                 (* VLV03_CMD_OPN *)
  ANDN %M67               (* VLV03_CNF_OPN *)
  IN
  OUT_BLK
  LD Q
  ST %M77                 (* VLV03_T_ALMD_CNF_OPN_DN *)
  END_BLK
  // as ST:
  //   VLV03_TON_ALMD_CNF_OPN(IN := VLV03_CMD_OPN AND NOT VLV03_CNF_OPN);
  //   VLV03_T_ALMD_CNF_OPN_DN := VLV03_TON_ALMD_CNF_OPN.Q;

// Rung 136
  BLK %TM24               (* VLV03_TON_ALMD_CNF_CLS *)
  LD %M72                 (* VLV03_CMD_CLS *)
  ANDN %M68               (* VLV03_CNF_CLS *)
  IN
  OUT_BLK
  LD Q
  ST %M79                 (* VLV03_T_ALMD_CNF_CLS_DN *)
  END_BLK
  // as ST:
  //   VLV03_TON_ALMD_CNF_CLS(IN := VLV03_CMD_CLS AND NOT VLV03_CNF_CLS);
  //   VLV03_T_ALMD_CNF_CLS_DN := VLV03_TON_ALMD_CNF_CLS.Q;

POU VLV04_ANALOG
  (* SectionNumber=5 *)

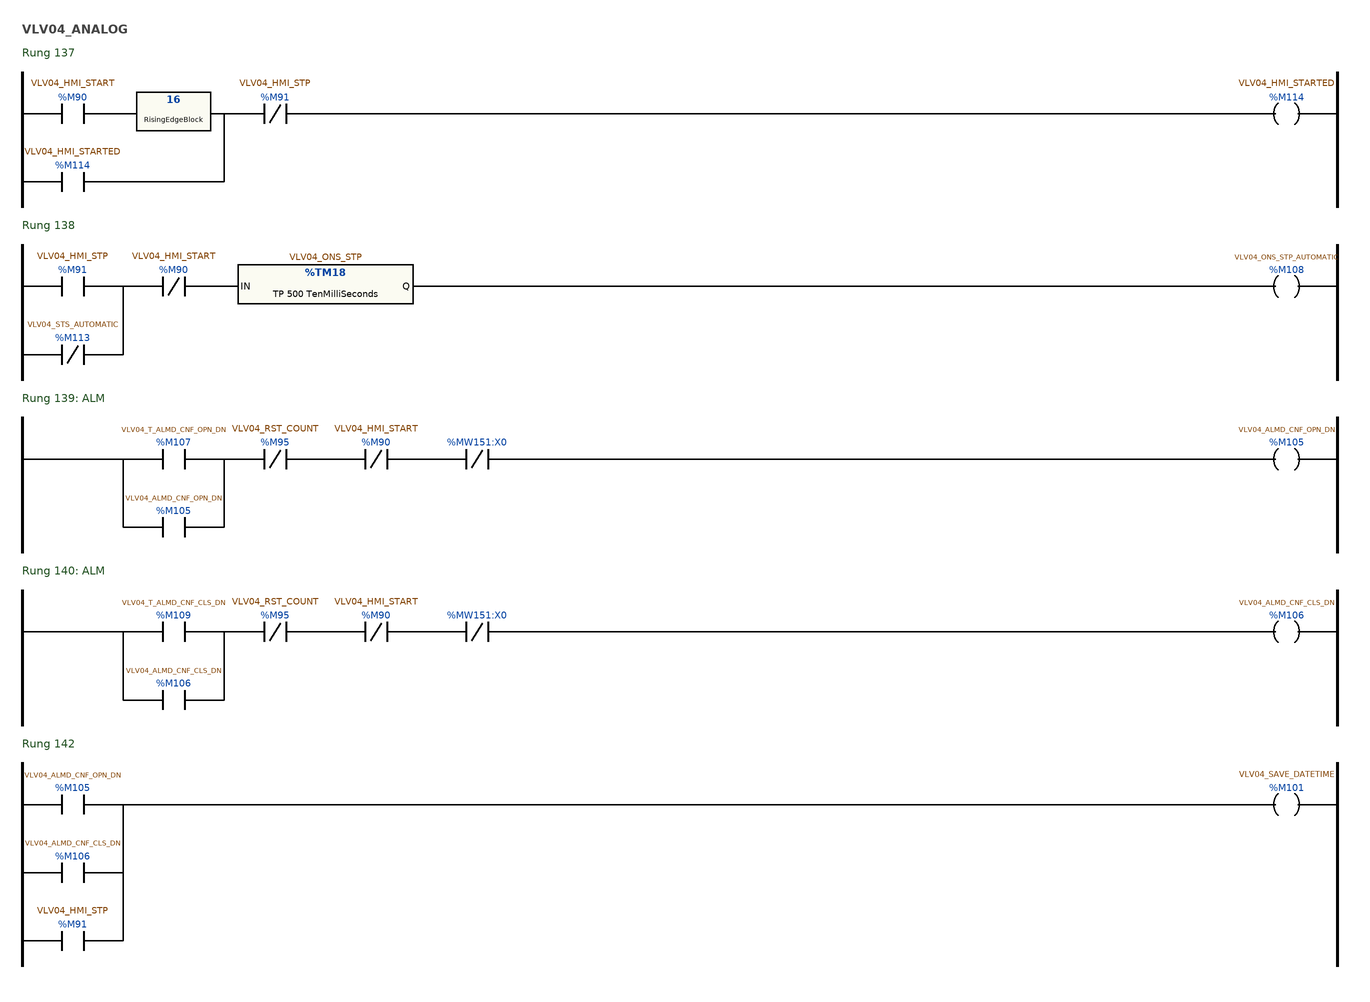

// Rung 137
  LD %M90                 (* VLV04_HMI_START *)
  RISING16
  OR %M114                (* VLV04_HMI_STARTED *)
  ANDN %M91               (* VLV04_HMI_STP *)
  ST %M114                (* VLV04_HMI_STARTED *)
  // as ST:
  //   VLV04_HMI_STARTED := (RISING(VLV04_HMI_START) OR VLV04_HMI_STARTED) AND NOT VLV04_HMI_STP;

// Rung 138
  BLK %TM18               (* VLV04_ONS_STP *)
  LD %M91                 (* VLV04_HMI_STP *)
  ORN %M113               (* VLV04_STS_AUTOMATIC *)
  ANDN %M90               (* VLV04_HMI_START *)
  IN
  OUT_BLK
  LD Q
  ST %M108                (* VLV04_ONS_STP_AUTOMATIC *)
  END_BLK
  // as ST:
  //   VLV04_ONS_STP(IN := (VLV04_HMI_STP OR NOT VLV04_STS_AUTOMATIC) AND NOT VLV04_HMI_START);
  //   VLV04_ONS_STP_AUTOMATIC := VLV04_ONS_STP.Q;

// Rung 139: ALM
  LD 1
  AND( %M107              (* VLV04_T_ALMD_CNF_OPN_DN *)
  OR %M105                (* VLV04_ALMD_CNF_OPN_DN *)
  )
  ANDN %M95               (* VLV04_RST_COUNT *)
  ANDN %M90               (* VLV04_HMI_START *)
  ANDN %MW151:X0
  ST %M105                (* VLV04_ALMD_CNF_OPN_DN *)
  // as ST:
  //   VLV04_ALMD_CNF_OPN_DN := (VLV04_T_ALMD_CNF_OPN_DN OR VLV04_ALMD_CNF_OPN_DN) AND NOT VLV04_RST_COUNT AND NOT VLV04_HMI_START AND NOT %MW151:X0;

// Rung 140: ALM
  LD 1
  AND( %M109              (* VLV04_T_ALMD_CNF_CLS_DN *)
  OR %M106                (* VLV04_ALMD_CNF_CLS_DN *)
  )
  ANDN %M95               (* VLV04_RST_COUNT *)
  ANDN %M90               (* VLV04_HMI_START *)
  ANDN %MW151:X0
  ST %M106                (* VLV04_ALMD_CNF_CLS_DN *)
  // as ST:
  //   VLV04_ALMD_CNF_CLS_DN := (VLV04_T_ALMD_CNF_CLS_DN OR VLV04_ALMD_CNF_CLS_DN) AND NOT VLV04_RST_COUNT AND NOT VLV04_HMI_START AND NOT %MW151:X0;

// Rung 141
  LD 1
  MULTIFB
  LD 1
  AND %M21                (* HORARIOOFICINA_ACTIVE *)
  AND %M114               (* VLV04_HMI_STARTED *)
  ANDN %M105              (* VLV04_ALMD_CNF_OPN_DN *)
  ANDN %M106              (* VLV04_ALMD_CNF_CLS_DN *)
  AND %MW432:X0
  ANDN %M118              (* VLV04_TON_HR_DN *)
  ST %MW2509:X0
  LD %MW2509:X0
  ST %M113                (* VLV04_STS_AUTOMATIC *)
  BLK %TM37               (* VLV04_ONS *)
  LD %MW2509:X0
  IN
  OUT_BLK
  LD Q
  ST %M96                 (* VLV04_ONS_STR_AUTOMATIC *)
  END_BLK
  MULTIFB
  // as ST:
  //   %MW2509:X0 := HORARIOOFICINA_ACTIVE AND VLV04_HMI_STARTED AND NOT VLV04_ALMD_CNF_OPN_DN AND NOT VLV04_ALMD_CNF_CLS_DN AND %MW432:X0 AND NOT VLV04_TON_HR_DN;
  //   VLV04_STS_AUTOMATIC := %MW2509:X0;
  //   VLV04_ONS(IN := %MW2509:X0);
  //   VLV04_ONS_STR_AUTOMATIC := VLV04_ONS.Q;
  (* the ladder stored for this rung does not match its IL; not drawn *)

// Rung 142
  LD %M105                (* VLV04_ALMD_CNF_OPN_DN *)
  OR %M106                (* VLV04_ALMD_CNF_CLS_DN *)
  OR %M91                 (* VLV04_HMI_STP *)
  ST %M101                (* VLV04_SAVE_DATETIME *)
  // as ST:
  //   VLV04_SAVE_DATETIME := VLV04_ALMD_CNF_OPN_DN OR VLV04_ALMD_CNF_CLS_DN OR VLV04_HMI_STP;

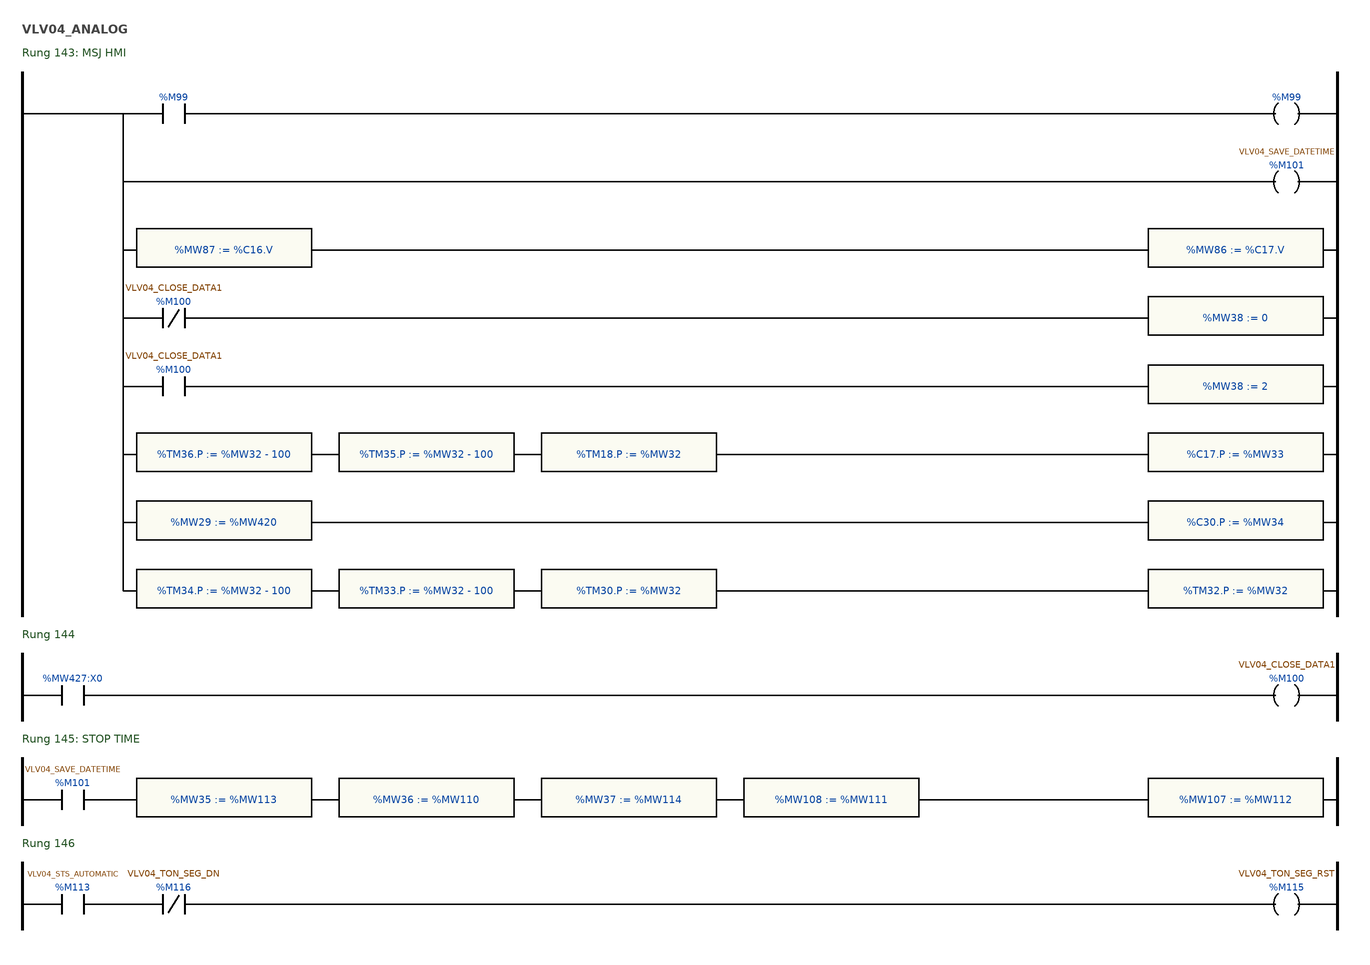

// Rung 143: MSJ HMI
  LD 1
  MPS
  AND %M99
  ST %M99
  MRD
  ST %M101                (* VLV04_SAVE_DATETIME *)
  MRD
  OPER [ %MW87 := %C16.V ](* VLV04_CNT_MIN *)
  [ %MW86 := %C17.V ]     (* VLV04_CNT_HR *)
  MRD
  ANDN %M100              (* VLV04_CLOSE_DATA1 *)
  [ %MW38 := 0 ]
  MRD
  AND %M100               (* VLV04_CLOSE_DATA1 *)
  [ %MW38 := 2 ]
  MRD
  OPER [ %TM36.P := %MW32 - 100 ](* VLV04_T_CNF_CLS, VLV04_T_CNF_PRESET *)
  OPER [ %TM35.P := %MW32 - 100 ](* VLV04_T_CNF_OPN, VLV04_T_CNF_PRESET *)
  OPER [ %TM18.P := %MW32 ](* VLV04_ONS_STP, VLV04_T_CNF_PRESET *)
  [ %C17.P := %MW33 ]     (* VLV04_CNT_HR, VLV04_CNF_HR_PRESET *)
  MRD
  OPER [ %MW29 := %MW420 ](* VLV04_CV_ACTUAL *)
  [ %C30.P := %MW34 ]     (* VLV04_SETPOINT_ALTO *)
  MPP
  OPER [ %TM34.P := %MW32 - 100 ](* VLV04_TON_ALMD_CNF_CLS, VLV04_T_CNF_PRESET *)
  OPER [ %TM33.P := %MW32 - 100 ](* VLV04_TON_ALMD_CNF_OPN, VLV04_T_CNF_PRESET *)
  OPER [ %TM30.P := %MW32 ](* VLV04_TON_OPN, VLV04_T_CNF_PRESET *)
  [ %TM32.P := %MW32 ]    (* VLV04_TON_CLS, VLV04_T_CNF_PRESET *)
  // as ST:
  //   %M99 := %M99;
  //   VLV04_SAVE_DATETIME := TRUE;
  //   %MW87 := VLV04_CNT_MIN.V;
  //   %MW86 := VLV04_CNT_HR.V;
  //   IF NOT VLV04_CLOSE_DATA1 THEN %MW38 := 0; END_IF;
  //   IF VLV04_CLOSE_DATA1 THEN %MW38 := 2; END_IF;
  //   VLV04_T_CNF_CLS.P := VLV04_T_CNF_PRESET - 100;
  //   VLV04_T_CNF_OPN.P := VLV04_T_CNF_PRESET - 100;
  //   VLV04_ONS_STP.P := VLV04_T_CNF_PRESET;
  //   VLV04_CNT_HR.P := VLV04_CNF_HR_PRESET;
  //   VLV04_CV_ACTUAL := %MW420;
  //   %C30.P := VLV04_SETPOINT_ALTO;
  //   VLV04_TON_ALMD_CNF_CLS.P := VLV04_T_CNF_PRESET - 100;
  //   VLV04_TON_ALMD_CNF_OPN.P := VLV04_T_CNF_PRESET - 100;
  //   VLV04_TON_OPN.P := VLV04_T_CNF_PRESET;
  //   VLV04_TON_CLS.P := VLV04_T_CNF_PRESET;

// Rung 144
  LD %MW427:X0
  ST %M100                (* VLV04_CLOSE_DATA1 *)
  // as ST:
  //   VLV04_CLOSE_DATA1 := %MW427:X0;

// Rung 145: STOP TIME
  LD %M101                (* VLV04_SAVE_DATETIME *)
  OPER [ %MW35 := %MW113 ](* VLV04_RTC_HHMM, MONTH *)
  OPER [ %MW36 := %MW110 ](* VLV04_RTC_MMDD, DAY *)
  OPER [ %MW37 := %MW114 ](* VLV04_RTC_YY, YEAR *)
  OPER [ %MW108 := %MW111 ](* HOUR *)
  [ %MW107 := %MW112 ]    (* MINUTES *)
  // as ST:
  //   IF VLV04_SAVE_DATETIME THEN VLV04_RTC_HHMM := MONTH; END_IF;
  //   IF VLV04_SAVE_DATETIME THEN VLV04_RTC_MMDD := DAY; END_IF;
  //   IF VLV04_SAVE_DATETIME THEN VLV04_RTC_YY := YEAR; END_IF;
  //   IF VLV04_SAVE_DATETIME THEN %MW108 := HOUR; END_IF;
  //   IF VLV04_SAVE_DATETIME THEN %MW107 := MINUTES; END_IF;

// Rung 146
  LD %M113                (* VLV04_STS_AUTOMATIC *)
  ANDN %M116              (* VLV04_TON_SEG_DN *)
  ST %M115                (* VLV04_TON_SEG_RST *)
  // as ST:
  //   VLV04_TON_SEG_RST := VLV04_STS_AUTOMATIC AND NOT VLV04_TON_SEG_DN;

// Rung 147
  BLK %C17                (* VLV04_CNT_HR *)
  LD %M95                 (* VLV04_RST_COUNT *)
  OR( %M21                (* HORARIOOFICINA_ACTIVE *)
  RISING17
  )
  R
  LD %M117                (* VLV04_TON_MIN_DN *)
  CU
  OUT_BLK
  LD D
  ST %M118                (* VLV04_TON_HR_DN *)
  END_BLK
  // as ST:
  //   VLV04_CNT_HR(RISING17 := HORARIOOFICINA_ACTIVE, R := VLV04_RST_COUNT OR HORARIOOFICINA_ACTIVE, CU := VLV04_TON_MIN_DN);
  //   VLV04_TON_HR_DN := VLV04_CNT_HR.D;
  (* the ladder stored for this rung does not match its IL; not drawn *)

// Rung 148
  BLK %C16                (* VLV04_CNT_MIN *)
  LD 1
  AND( %M95               (* VLV04_RST_COUNT *)
  OR %M117                (* VLV04_TON_MIN_DN *)
  )
  OR( %M21                (* HORARIOOFICINA_ACTIVE *)
  RISING18
  )
  R
  LD %M116                (* VLV04_TON_SEG_DN *)
  CU
  OUT_BLK
  LD D
  ST %M117                (* VLV04_TON_MIN_DN *)
  END_BLK
  // as ST:
  //   VLV04_CNT_MIN(RISING18 := HORARIOOFICINA_ACTIVE, R := VLV04_RST_COUNT OR VLV04_TON_MIN_DN OR HORARIOOFICINA_ACTIVE, CU := VLV04_TON_SEG_DN);
  //   VLV04_TON_MIN_DN := VLV04_CNT_MIN.D;
  (* the ladder stored for this rung does not match its IL; not drawn *)

// Rung 149
  LD 1
  MULTIFB
  LD 1
  ST %MW2509:X1
  BLK %TM31               (* VLV04_TON_SEG *)
  LD %MW2509:X1
  AND %M113               (* VLV04_STS_AUTOMATIC *)
  AND %M115               (* VLV04_TON_SEG_RST *)
  IN
  OUT_BLK
  LD Q
  ST %MW2509:X0
  END_BLK
  BLK %C15                (* VLV04_CNT_SEG *)
  LD %MW2509:X1
  AND( %M95               (* VLV04_RST_COUNT *)
  OR %M116                (* VLV04_TON_SEG_DN *)
  )
  R
  LD %MW2509:X0
  CU
  OUT_BLK
  LD D
  ST %M116                (* VLV04_TON_SEG_DN *)
  END_BLK
  MULTIFB
  // as ST:
  //   %MW2509:X1 := TRUE;
  //   VLV04_TON_SEG(IN := %MW2509:X1 AND VLV04_STS_AUTOMATIC AND VLV04_TON_SEG_RST);
  //   %MW2509:X0 := VLV04_TON_SEG.Q;
  //   VLV04_CNT_SEG(R := %MW2509:X1 AND (VLV04_RST_COUNT OR VLV04_TON_SEG_DN), CU := %MW2509:X0);
  //   VLV04_TON_SEG_DN := VLV04_CNT_SEG.D;
  (* the ladder stored for this rung does not match its IL; not drawn *)

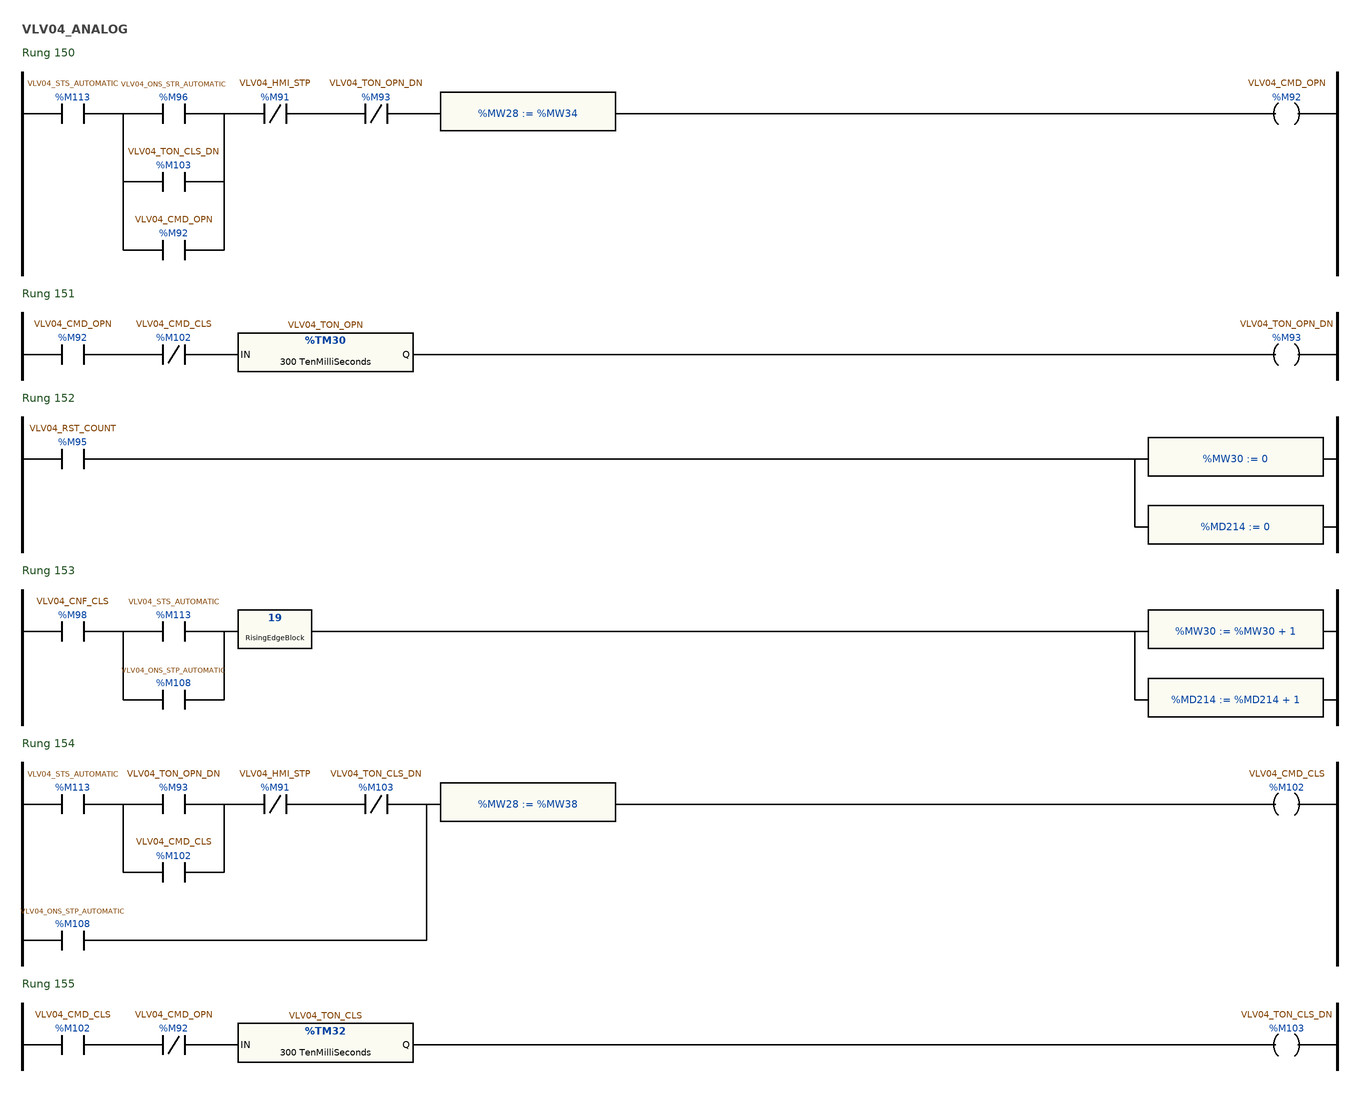

// Rung 150
  LD %M113                (* VLV04_STS_AUTOMATIC *)
  AND( %M96               (* VLV04_ONS_STR_AUTOMATIC *)
  OR %M103                (* VLV04_TON_CLS_DN *)
  OR %M92                 (* VLV04_CMD_OPN *)
  )
  ANDN %M91               (* VLV04_HMI_STP *)
  ANDN %M93               (* VLV04_TON_OPN_DN *)
  OPER [ %MW28 := %MW34 ] (* VLV04_SP_ACTUAL, VLV04_SETPOINT_ALTO *)
  ST %M92                 (* VLV04_CMD_OPN *)
  // as ST:
  //   IF VLV04_STS_AUTOMATIC AND (VLV04_ONS_STR_AUTOMATIC OR VLV04_TON_CLS_DN OR VLV04_CMD_OPN) AND NOT VLV04_HMI_STP AND NOT VLV04_TON_OPN_DN THEN VLV04_SP_ACTUAL := VLV04_SETPOINT_ALTO; END_IF;
  //   VLV04_CMD_OPN := VLV04_STS_AUTOMATIC AND (VLV04_ONS_STR_AUTOMATIC OR VLV04_TON_CLS_DN OR VLV04_CMD_OPN) AND NOT VLV04_HMI_STP AND NOT VLV04_TON_OPN_DN;

// Rung 151
  BLK %TM30               (* VLV04_TON_OPN *)
  LD %M92                 (* VLV04_CMD_OPN *)
  ANDN %M102              (* VLV04_CMD_CLS *)
  IN
  OUT_BLK
  LD Q
  ST %M93                 (* VLV04_TON_OPN_DN *)
  END_BLK
  // as ST:
  //   VLV04_TON_OPN(IN := VLV04_CMD_OPN AND NOT VLV04_CMD_CLS);
  //   VLV04_TON_OPN_DN := VLV04_TON_OPN.Q;

// Rung 152
  LD %M95                 (* VLV04_RST_COUNT *)
  [ %MW30 := 0 ]          (* VLV04_CNT_CLS_ACC *)
  [ %MD214 := 0 ]         (* VLV04_CNT_CLS_ACC2 *)
  // as ST:
  //   IF VLV04_RST_COUNT THEN VLV04_CNT_CLS_ACC := 0; END_IF;
  //   IF VLV04_RST_COUNT THEN VLV04_CNT_CLS_ACC2 := 0; END_IF;

// Rung 153
  LD %M98                 (* VLV04_CNF_CLS *)
  AND( %M113              (* VLV04_STS_AUTOMATIC *)
  OR %M108                (* VLV04_ONS_STP_AUTOMATIC *)
  )
  RISING19
  [ %MW30 := %MW30 + 1 ]  (* VLV04_CNT_CLS_ACC, VLV04_CNT_CLS_ACC *)
  [ %MD214 := %MD214 + 1 ](* VLV04_CNT_CLS_ACC2, VLV04_CNT_CLS_ACC2 *)
  // as ST:
  //   IF RISING(VLV04_CNF_CLS AND (VLV04_STS_AUTOMATIC OR VLV04_ONS_STP_AUTOMATIC)) THEN VLV04_CNT_CLS_ACC := VLV04_CNT_CLS_ACC + 1; END_IF;
  //   IF RISING(VLV04_CNF_CLS AND (VLV04_STS_AUTOMATIC OR VLV04_ONS_STP_AUTOMATIC)) THEN VLV04_CNT_CLS_ACC2 := VLV04_CNT_CLS_ACC2 + 1; END_IF;

// Rung 154
  LD %M113                (* VLV04_STS_AUTOMATIC *)
  AND( %M93               (* VLV04_TON_OPN_DN *)
  OR %M102                (* VLV04_CMD_CLS *)
  )
  ANDN %M91               (* VLV04_HMI_STP *)
  ANDN %M103              (* VLV04_TON_CLS_DN *)
  OR %M108                (* VLV04_ONS_STP_AUTOMATIC *)
  OPER [ %MW28 := %MW38 ] (* VLV04_SP_ACTUAL *)
  ST %M102                (* VLV04_CMD_CLS *)
  // as ST:
  //   IF VLV04_STS_AUTOMATIC AND (VLV04_TON_OPN_DN OR VLV04_CMD_CLS) AND NOT VLV04_HMI_STP AND NOT VLV04_TON_CLS_DN OR VLV04_ONS_STP_AUTOMATIC THEN VLV04_SP_ACTUAL := %MW38; END_IF;
  //   VLV04_CMD_CLS := VLV04_STS_AUTOMATIC AND (VLV04_TON_OPN_DN OR VLV04_CMD_CLS) AND NOT VLV04_HMI_STP AND NOT VLV04_TON_CLS_DN OR VLV04_ONS_STP_AUTOMATIC;

// Rung 155
  BLK %TM32               (* VLV04_TON_CLS *)
  LD %M102                (* VLV04_CMD_CLS *)
  ANDN %M92               (* VLV04_CMD_OPN *)
  IN
  OUT_BLK
  LD Q
  ST %M103                (* VLV04_TON_CLS_DN *)
  END_BLK
  // as ST:
  //   VLV04_TON_CLS(IN := VLV04_CMD_CLS AND NOT VLV04_CMD_OPN);
  //   VLV04_TON_CLS_DN := VLV04_TON_CLS.Q;

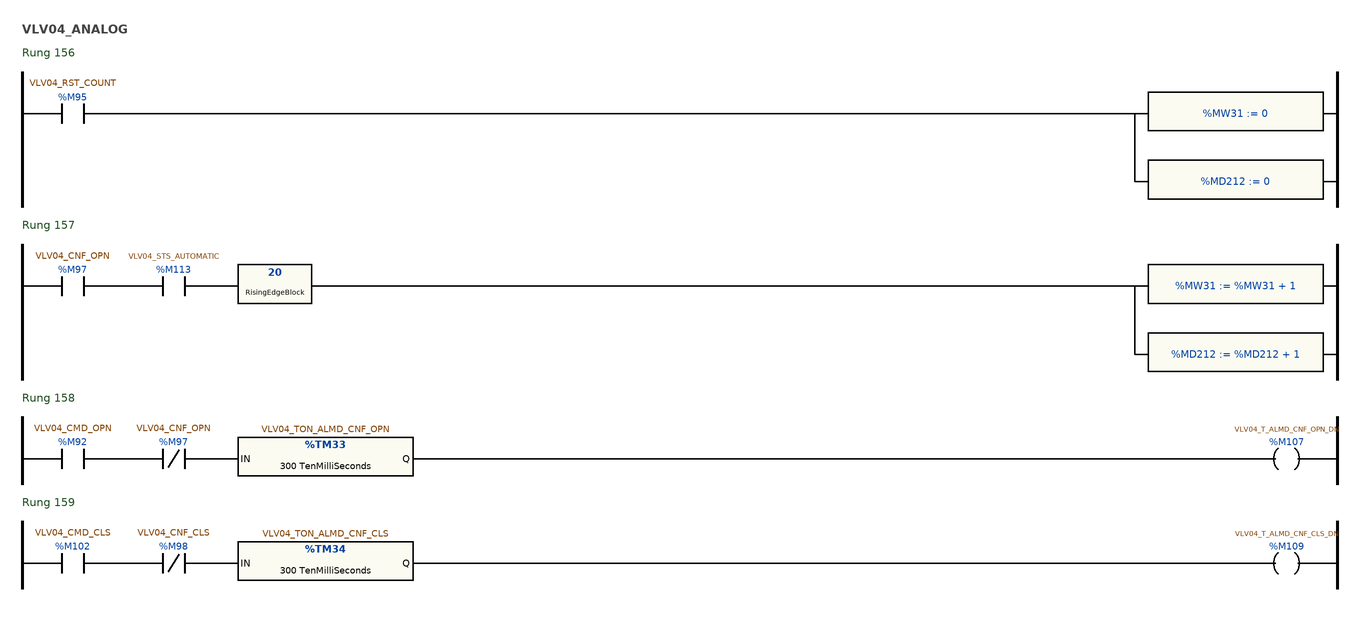

// Rung 156
  LD %M95                 (* VLV04_RST_COUNT *)
  [ %MW31 := 0 ]          (* VLV04_CNT_OPN_ACC *)
  [ %MD212 := 0 ]         (* VLV04_CNT_OPN_ACC2 *)
  // as ST:
  //   IF VLV04_RST_COUNT THEN VLV04_CNT_OPN_ACC := 0; END_IF;
  //   IF VLV04_RST_COUNT THEN VLV04_CNT_OPN_ACC2 := 0; END_IF;

// Rung 157
  LD %M97                 (* VLV04_CNF_OPN *)
  AND %M113               (* VLV04_STS_AUTOMATIC *)
  RISING20
  [ %MW31 := %MW31 + 1 ]  (* VLV04_CNT_OPN_ACC, VLV04_CNT_OPN_ACC *)
  [ %MD212 := %MD212 + 1 ](* VLV04_CNT_OPN_ACC2, VLV04_CNT_OPN_ACC2 *)
  // as ST:
  //   IF RISING(VLV04_CNF_OPN AND VLV04_STS_AUTOMATIC) THEN VLV04_CNT_OPN_ACC := VLV04_CNT_OPN_ACC + 1; END_IF;
  //   IF RISING(VLV04_CNF_OPN AND VLV04_STS_AUTOMATIC) THEN VLV04_CNT_OPN_ACC2 := VLV04_CNT_OPN_ACC2 + 1; END_IF;

// Rung 158
  BLK %TM33               (* VLV04_TON_ALMD_CNF_OPN *)
  LD %M92                 (* VLV04_CMD_OPN *)
  ANDN %M97               (* VLV04_CNF_OPN *)
  IN
  OUT_BLK
  LD Q
  ST %M107                (* VLV04_T_ALMD_CNF_OPN_DN *)
  END_BLK
  // as ST:
  //   VLV04_TON_ALMD_CNF_OPN(IN := VLV04_CMD_OPN AND NOT VLV04_CNF_OPN);
  //   VLV04_T_ALMD_CNF_OPN_DN := VLV04_TON_ALMD_CNF_OPN.Q;

// Rung 159
  BLK %TM34               (* VLV04_TON_ALMD_CNF_CLS *)
  LD %M102                (* VLV04_CMD_CLS *)
  ANDN %M98               (* VLV04_CNF_CLS *)
  IN
  OUT_BLK
  LD Q
  ST %M109                (* VLV04_T_ALMD_CNF_CLS_DN *)
  END_BLK
  // as ST:
  //   VLV04_TON_ALMD_CNF_CLS(IN := VLV04_CMD_CLS AND NOT VLV04_CNF_CLS);
  //   VLV04_T_ALMD_CNF_CLS_DN := VLV04_TON_ALMD_CNF_CLS.Q;

POU VLV05_MODBUSS
  (* SectionNumber=6 *)

